        PUBLISH_1 : PUBLISH_1(ID := opc_ua[WRITE;%opcuaFolderTestWithNodeIdString1%]);
        E_CTU : E_CTU(PV := UINT#3);
        folderTest2SameFolder1String : TEST_CONDITION;
        SUBSCRIBE_1_1 : SUBSCRIBE_1(ID := opc_ua[READ;%opcuaFolderTestWithNodeIdString1%]);
        BOOL2BOOL_1_1_1_1_2 : DINT2DINT;
        folderTest2DifferentFolder1String : TEST_CONDITION;
        SUBSCRIBE_2_2 : SUBSCRIBE_2(ID := opc_ua[READ;%opcuaFolderTestWithNodeIdString2%]);
        SUBSCRIBE_2_1_1 : SUBSCRIBE_2(ID := opc_ua[READ;%opcuaFolderTestWithNodeIdString3%]);
        BOOL2BOOL_1_3 : DINT2DINT;
        BOOL2BOOL_3 : DINT2DINT;
        folderTestDirectUnderString : TEST_CONDITION;
      END_FBS
      EVENT_CONNECTIONS
        BOOL2BOOL_2.CNF TO BOOL2BOOL_1_2.REQ;
        BOOL2BOOL_1_2.CNF TO BOOL2BOOL_1_1_2.REQ;
        BOOL2BOOL_1_1_3.CNF TO F_EQ_1_2.REQ;
        F_EQ_1_2.CNF TO folderTest2SameFolder1String.REQ;
        BOOL2BOOL_3.CNF TO F_EQ_2.REQ;
        F_EQ_2.CNF TO folderTestDirectUnderString.REQ;
        PUBLISH_2_1.INITO TO PUBLISH_2.INIT;
        PUBLISH_2_1.CNF TO PUBLISH_2.REQ;
        PUBLISH_2.INITO TO PUBLISH_1.INIT;
        PUBLISH_2.CNF TO PUBLISH_1.REQ;
        F_EQ_1_1_2.CNF TO folderTest2SameFolder2String.REQ;
        F_EQ_1_1_1_1_1.CNF TO folderTest2DifferentFolder2String.REQ;
        E_CTU.CUO TO E_PERMIT.EI;
        BOOL2BOOL_1_1_1_1_2.CNF TO F_EQ_1_1_1_2.REQ;
        F_EQ_1_1_1_2.CNF TO folderTest2DifferentFolder1String.REQ;
        folderTest2DifferentFolder1String.CNF TO F_EQ_1_1_1_1_1.REQ;
        BOOL2BOOL_1_1_1_1_1.CNF TO PUBLISH_2_1.REQ;
        BOOL2BOOL_1_1_2.CNF TO BOOL2BOOL_1_1_1_2.REQ;
        BOOL2BOOL_1_1_1_2.CNF TO BOOL2BOOL_1_1_1_1_1.REQ;
        SUBSCRIBE_2_1_1.IND TO BOOL2BOOL_1_1_1_3.REQ;
        BOOL2BOOL_1_1_1_3.CNF TO BOOL2BOOL_1_1_1_1_2.REQ;
        BOOL2BOOL_1_3.CNF TO BOOL2BOOL_1_1_3.REQ;
        folderTest2SameFolder1String.CNF TO F_EQ_1_1_2.REQ;
        SUBSCRIBE_1_1.INITO TO SUBSCRIBE_2_2.INIT;
        SUBSCRIBE_1_1.IND TO BOOL2BOOL_3.REQ;
        SUBSCRIBE_2_2.INITO TO SUBSCRIBE_2_1_1.INIT;
        SUBSCRIBE_2_2.IND TO BOOL2BOOL_1_3.REQ;
        PUBLISH_1.INITO TO INITO;
        INIT TO SUBSCRIBE_1_1.INIT;
        folderTestDirectUnderString.CNF TO E_CTU.CU;
        folderTest2SameFolder2String.CNF TO E_CTU.CU;
        folderTest2DifferentFolder2String.CNF TO E_CTU.CU;
        E_PERMIT.EO TO CNF;
        REQ TO BOOL2BOOL_2.REQ;
        SUBSCRIBE_2_1_1.INITO TO PUBLISH_2_1.INIT;
      END_CONNECTIONS
      DATA_CONNECTIONS
        BOOL2BOOL_1_2.OUT TO PUBLISH_2.SD_1;
        BOOL2BOOL_1_3.OUT TO F_EQ_1_2.IN1;
        F_EQ_1_2.OUT TO folderTest2SameFolder1String.check;
        BOOL2BOOL_3.OUT TO F_EQ_2.IN1;
        F_EQ_2.OUT TO folderTestDirectUnderString.check;
        BOOL2BOOL_1_1_2.OUT TO PUBLISH_2.SD_2;
        F_EQ_1_1_2.OUT TO folderTest2SameFolder2String.check;
        F_EQ_1_1_1_1_1.OUT TO folderTest2DifferentFolder2String.check;
        E_CTU.Q TO E_PERMIT.PERMIT;
        BOOL2BOOL_1_1_1_3.OUT TO F_EQ_1_1_1_2.IN1;
        F_EQ_1_1_1_2.OUT TO folderTest2DifferentFolder1String.check;
        BOOL2BOOL_1_1_1_1_2.OUT TO F_EQ_1_1_1_1_1.IN1;
        BOOL2BOOL_1_1_1_2.OUT TO PUBLISH_2_1.SD_1;
        BOOL2BOOL_1_1_1_1_1.OUT TO PUBLISH_2_1.SD_2;
        BOOL2BOOL_2.OUT TO PUBLISH_1.SD_1;
        SUBSCRIBE_2_1_1.RD_1 TO BOOL2BOOL_1_1_1_3.IN;
        SUBSCRIBE_2_2.RD_2 TO BOOL2BOOL_1_1_3.IN;
        BOOL2BOOL_1_1_3.OUT TO F_EQ_1_1_2.IN1;
        SUBSCRIBE_1_1.RD_1 TO BOOL2BOOL_3.IN;
        SUBSCRIBE_2_1_1.RD_2 TO BOOL2BOOL_1_1_1_1_2.IN;
        SUBSCRIBE_2_2.RD_1 TO BOOL2BOOL_1_3.IN;
        QI TO SUBSCRIBE_1_1.QI;
        QI TO SUBSCRIBE_2_2.QI;
        QI TO SUBSCRIBE_2_1_1.QI;
        QI TO PUBLISH_1.QI;
        QI TO PUBLISH_2.QI;
        QI TO PUBLISH_2_1.QI;
      END_CONNECTIONS
    END_SUBAPPLICATION
    SUBAPPLICATION foldersWithNodeByteStringId_1
      EVENT_INPUT
        INIT;
        REQ;
      END_EVENT
      EVENT_OUTPUT
        INITO;
        CNF;
      END_EVENT
      VAR_INPUT
        QI : BOOL;
      END_VAR
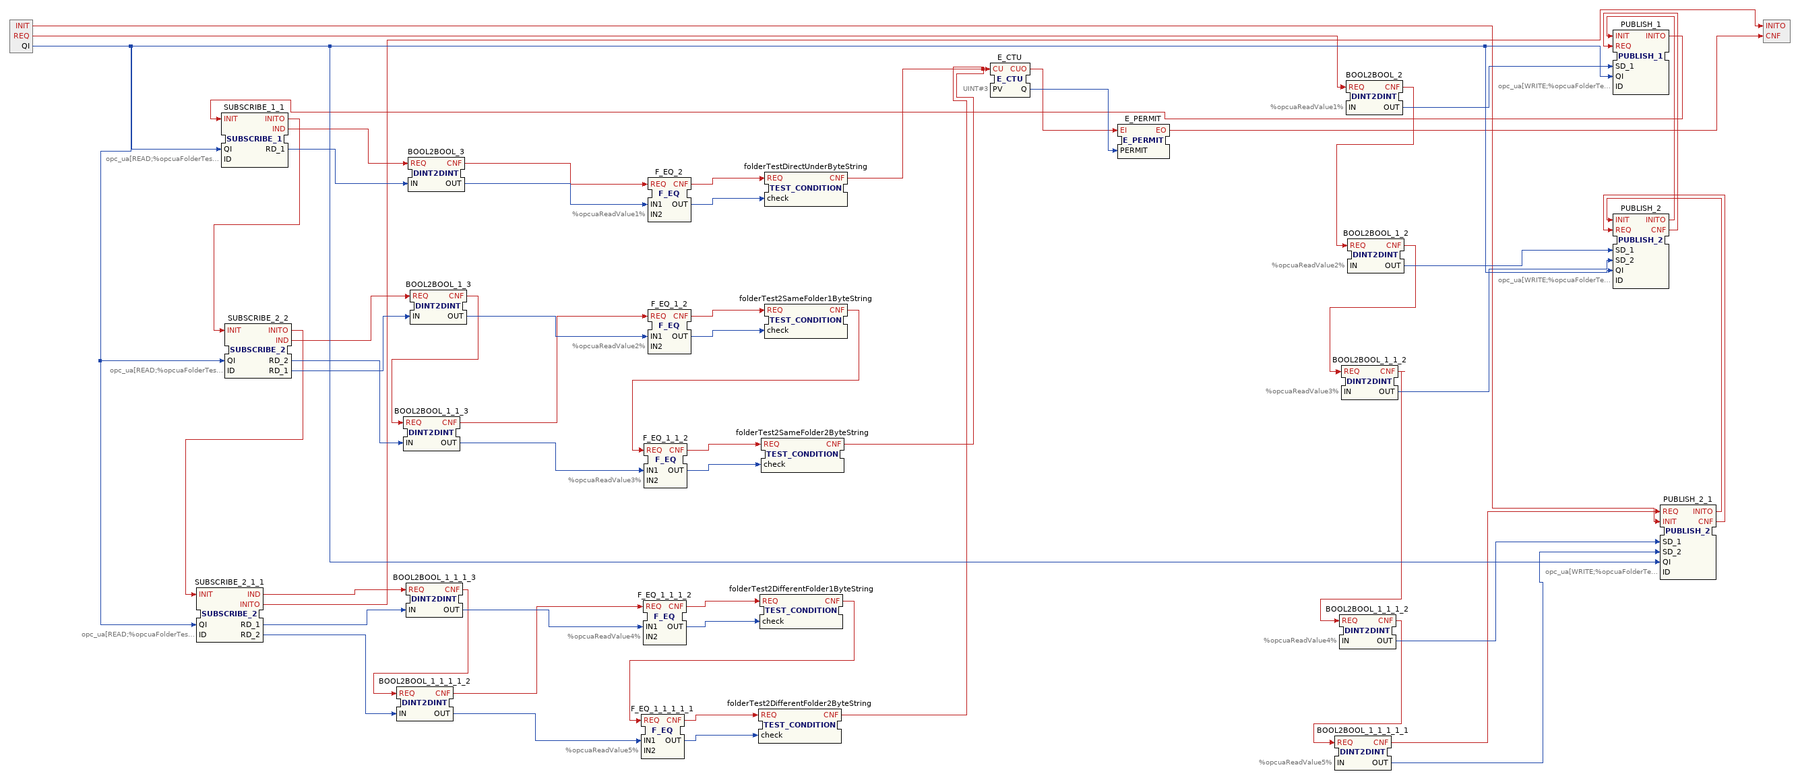
      [picture p23: application OpcUaLocalWorking.foldersWithNodeByteStringId_1]
      FBS
        BOOL2BOOL_1_2 : DINT2DINT(IN := %opcuaReadValue2%);
        F_EQ_1_2 : F_EQ(IN2 := %opcuaReadValue2%);
        F_EQ_2 : F_EQ(IN2 := %opcuaReadValue1%);
        PUBLISH_2 : PUBLISH_2(ID := opc_ua[WRITE;%opcuaFolderTestWithNodeIdByteString2%]);
        folderTest2SameFolder2ByteString : TEST_CONDITION;
        folderTest2DifferentFolder2ByteString : TEST_CONDITION;
        E_PERMIT : E_PERMIT;
        F_EQ_1_1_1_2 : F_EQ(IN2 := %opcuaReadValue4%);
        F_EQ_1_1_1_1_1 : F_EQ(IN2 := %opcuaReadValue5%);
        PUBLISH_2_1 : PUBLISH_2(ID := opc_ua[WRITE;%opcuaFolderTestWithNodeIdByteString3%]);
        BOOL2BOOL_1_1_2 : DINT2DINT(IN := %opcuaReadValue3%);
        BOOL2BOOL_1_1_1_1_1 : DINT2DINT(IN := %opcuaReadValue5%);
        BOOL2BOOL_2 : DINT2DINT(IN := %opcuaReadValue1%);
        BOOL2BOOL_1_1_1_3 : DINT2DINT;
        BOOL2BOOL_1_1_3 : DINT2DINT;
        BOOL2BOOL_1_1_1_2 : DINT2DINT(IN := %opcuaReadValue4%);
        F_EQ_1_1_2 : F_EQ(IN2 := %opcuaReadValue3%);
        PUBLISH_1 : PUBLISH_1(ID := opc_ua[WRITE;%opcuaFolderTestWithNodeIdByteString1%]);
        E_CTU : E_CTU(PV := UINT#3);
        folderTest2SameFolder1ByteString : TEST_CONDITION;
        SUBSCRIBE_1_1 : SUBSCRIBE_1(ID := opc_ua[READ;%opcuaFolderTestWithNodeIdByteString1%]);
        BOOL2BOOL_1_1_1_1_2 : DINT2DINT;
        folderTest2DifferentFolder1ByteString : TEST_CONDITION;
        SUBSCRIBE_2_2 : SUBSCRIBE_2(ID := opc_ua[READ;%opcuaFolderTestWithNodeIdByteString2%]);
        SUBSCRIBE_2_1_1 : SUBSCRIBE_2(ID := opc_ua[READ;%opcuaFolderTestWithNodeIdByteString3%]);
        BOOL2BOOL_1_3 : DINT2DINT;
        BOOL2BOOL_3 : DINT2DINT;
        folderTestDirectUnderByteString : TEST_CONDITION;
      END_FBS
      EVENT_CONNECTIONS
        BOOL2BOOL_2.CNF TO BOOL2BOOL_1_2.REQ;
        BOOL2BOOL_1_2.CNF TO BOOL2BOOL_1_1_2.REQ;
        BOOL2BOOL_1_1_3.CNF TO F_EQ_1_2.REQ;
        F_EQ_1_2.CNF TO folderTest2SameFolder1ByteString.REQ;
        BOOL2BOOL_3.CNF TO F_EQ_2.REQ;
        F_EQ_2.CNF TO folderTestDirectUnderByteString.REQ;
        PUBLISH_2_1.INITO TO PUBLISH_2.INIT;
        PUBLISH_2_1.CNF TO PUBLISH_2.REQ;
        PUBLISH_2.INITO TO PUBLISH_1.INIT;
        PUBLISH_2.CNF TO PUBLISH_1.REQ;
        F_EQ_1_1_2.CNF TO folderTest2SameFolder2ByteString.REQ;
        F_EQ_1_1_1_1_1.CNF TO folderTest2DifferentFolder2ByteString.REQ;
        E_CTU.CUO TO E_PERMIT.EI;
        BOOL2BOOL_1_1_1_1_2.CNF TO F_EQ_1_1_1_2.REQ;
        F_EQ_1_1_1_2.CNF TO folderTest2DifferentFolder1ByteString.REQ;
        folderTest2DifferentFolder1ByteString.CNF TO F_EQ_1_1_1_1_1.REQ;
        BOOL2BOOL_1_1_1_1_1.CNF TO PUBLISH_2_1.REQ;
        BOOL2BOOL_1_1_2.CNF TO BOOL2BOOL_1_1_1_2.REQ;
        BOOL2BOOL_1_1_1_2.CNF TO BOOL2BOOL_1_1_1_1_1.REQ;
        SUBSCRIBE_2_1_1.IND TO BOOL2BOOL_1_1_1_3.REQ;
        BOOL2BOOL_1_1_1_3.CNF TO BOOL2BOOL_1_1_1_1_2.REQ;
        BOOL2BOOL_1_3.CNF TO BOOL2BOOL_1_1_3.REQ;
        folderTest2SameFolder1ByteString.CNF TO F_EQ_1_1_2.REQ;
        SUBSCRIBE_1_1.INITO TO SUBSCRIBE_2_2.INIT;
        SUBSCRIBE_1_1.IND TO BOOL2BOOL_3.REQ;
        SUBSCRIBE_2_2.INITO TO SUBSCRIBE_2_1_1.INIT;
        SUBSCRIBE_2_2.IND TO BOOL2BOOL_1_3.REQ;
        folderTestDirectUnderByteString.CNF TO E_CTU.CU;
        folderTest2SameFolder2ByteString.CNF TO E_CTU.CU;
        folderTest2DifferentFolder2ByteString.CNF TO E_CTU.CU;
        E_PERMIT.EO TO CNF;
        REQ TO BOOL2BOOL_2.REQ;
        INIT TO PUBLISH_2_1.INIT;
        PUBLISH_1.INITO TO SUBSCRIBE_1_1.INIT;
        SUBSCRIBE_2_1_1.INITO TO INITO;
      END_CONNECTIONS
      DATA_CONNECTIONS
        BOOL2BOOL_1_2.OUT TO PUBLISH_2.SD_1;
        BOOL2BOOL_1_3.OUT TO F_EQ_1_2.IN1;
        F_EQ_1_2.OUT TO folderTest2SameFolder1ByteString.check;
        BOOL2BOOL_3.OUT TO F_EQ_2.IN1;
        F_EQ_2.OUT TO folderTestDirectUnderByteString.check;
        BOOL2BOOL_1_1_2.OUT TO PUBLISH_2.SD_2;
        F_EQ_1_1_2.OUT TO folderTest2SameFolder2ByteString.check;
        F_EQ_1_1_1_1_1.OUT TO folderTest2DifferentFolder2ByteString.check;
        E_CTU.Q TO E_PERMIT.PERMIT;
        BOOL2BOOL_1_1_1_3.OUT TO F_EQ_1_1_1_2.IN1;
        F_EQ_1_1_1_2.OUT TO folderTest2DifferentFolder1ByteString.check;
        BOOL2BOOL_1_1_1_1_2.OUT TO F_EQ_1_1_1_1_1.IN1;
        BOOL2BOOL_1_1_1_2.OUT TO PUBLISH_2_1.SD_1;
        BOOL2BOOL_1_1_1_1_1.OUT TO PUBLISH_2_1.SD_2;
        BOOL2BOOL_2.OUT TO PUBLISH_1.SD_1;
        SUBSCRIBE_2_1_1.RD_1 TO BOOL2BOOL_1_1_1_3.IN;
        SUBSCRIBE_2_2.RD_2 TO BOOL2BOOL_1_1_3.IN;
        BOOL2BOOL_1_1_3.OUT TO F_EQ_1_1_2.IN1;
        SUBSCRIBE_1_1.RD_1 TO BOOL2BOOL_3.IN;
        SUBSCRIBE_2_1_1.RD_2 TO BOOL2BOOL_1_1_1_1_2.IN;
        SUBSCRIBE_2_2.RD_1 TO BOOL2BOOL_1_3.IN;
        QI TO SUBSCRIBE_1_1.QI;
        QI TO SUBSCRIBE_2_2.QI;
        QI TO SUBSCRIBE_2_1_1.QI;
        QI TO PUBLISH_1.QI;
        QI TO PUBLISH_2.QI;
        QI TO PUBLISH_2_1.QI;
      END_CONNECTIONS
    END_SUBAPPLICATION
    SUBAPPLICATION foldersWithNodeNumericId_1
      EVENT_INPUT
        INIT;
        REQ;
      END_EVENT
      EVENT_OUTPUT
        INITO;
        CNF;
      END_EVENT
      VAR_INPUT
        QI : BOOL;
      END_VAR
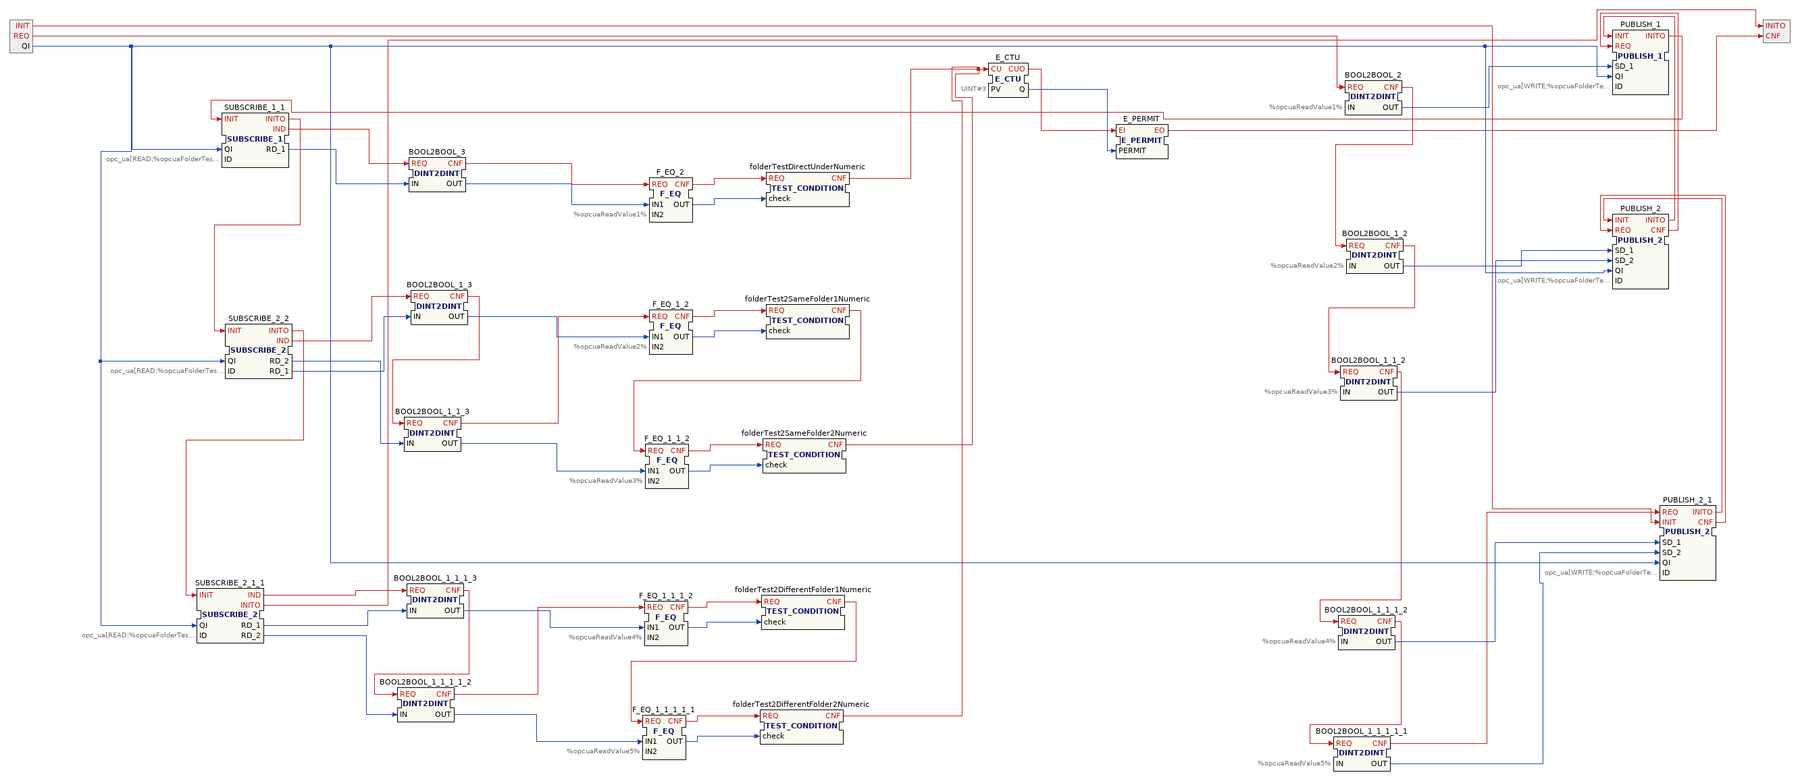
      FBS
        BOOL2BOOL_1_2 : DINT2DINT(IN := %opcuaReadValue2%);
        F_EQ_1_2 : F_EQ(IN2 := %opcuaReadValue2%);
        F_EQ_2 : F_EQ(IN2 := %opcuaReadValue1%);
        PUBLISH_2 : PUBLISH_2(ID := opc_ua[WRITE;%opcuaFolderTestWithNodeIdNumeric2%]);
        folderTest2SameFolder2Numeric : TEST_CONDITION;
        folderTest2DifferentFolder2Numeric : TEST_CONDITION;
        E_PERMIT : E_PERMIT;
        F_EQ_1_1_1_2 : F_EQ(IN2 := %opcuaReadValue4%);
        F_EQ_1_1_1_1_1 : F_EQ(IN2 := %opcuaReadValue5%);
        PUBLISH_2_1 : PUBLISH_2(ID := opc_ua[WRITE;%opcuaFolderTestWithNodeIdNumeric3%]);
        BOOL2BOOL_1_1_2 : DINT2DINT(IN := %opcuaReadValue3%);
        BOOL2BOOL_1_1_1_1_1 : DINT2DINT(IN := %opcuaReadValue5%);
        BOOL2BOOL_2 : DINT2DINT(IN := %opcuaReadValue1%);
        BOOL2BOOL_1_1_1_3 : DINT2DINT;
        BOOL2BOOL_1_1_3 : DINT2DINT;
        BOOL2BOOL_1_1_1_2 : DINT2DINT(IN := %opcuaReadValue4%);
        F_EQ_1_1_2 : F_EQ(IN2 := %opcuaReadValue3%);
        PUBLISH_1 : PUBLISH_1(ID := opc_ua[WRITE;%opcuaFolderTestWithNodeIdNumeric1%]);
        E_CTU : E_CTU(PV := UINT#3);
        folderTest2SameFolder1Numeric : TEST_CONDITION;
        SUBSCRIBE_1_1 : SUBSCRIBE_1(ID := opc_ua[READ;%opcuaFolderTestWithNodeIdNumeric1%]);
        BOOL2BOOL_1_1_1_1_2 : DINT2DINT;
        folderTest2DifferentFolder1Numeric : TEST_CONDITION;
        SUBSCRIBE_2_2 : SUBSCRIBE_2(ID := opc_ua[READ;%opcuaFolderTestWithNodeIdNumeric2%]);
        SUBSCRIBE_2_1_1 : SUBSCRIBE_2(ID := opc_ua[READ;%opcuaFolderTestWithNodeIdNumeric3%]);
        BOOL2BOOL_1_3 : DINT2DINT;
        BOOL2BOOL_3 : DINT2DINT;
        folderTestDirectUnderNumeric : TEST_CONDITION;
      END_FBS
      EVENT_CONNECTIONS
        BOOL2BOOL_2.CNF TO BOOL2BOOL_1_2.REQ;
        BOOL2BOOL_1_2.CNF TO BOOL2BOOL_1_1_2.REQ;
        BOOL2BOOL_1_1_3.CNF TO F_EQ_1_2.REQ;
        F_EQ_1_2.CNF TO folderTest2SameFolder1Numeric.REQ;
        BOOL2BOOL_3.CNF TO F_EQ_2.REQ;
        F_EQ_2.CNF TO folderTestDirectUnderNumeric.REQ;
        PUBLISH_2_1.INITO TO PUBLISH_2.INIT;
        PUBLISH_2_1.CNF TO PUBLISH_2.REQ;
        PUBLISH_2.INITO TO PUBLISH_1.INIT;
        PUBLISH_2.CNF TO PUBLISH_1.REQ;
        F_EQ_1_1_2.CNF TO folderTest2SameFolder2Numeric.REQ;
        F_EQ_1_1_1_1_1.CNF TO folderTest2DifferentFolder2Numeric.REQ;
        E_CTU.CUO TO E_PERMIT.EI;
        BOOL2BOOL_1_1_1_1_2.CNF TO F_EQ_1_1_1_2.REQ;
        F_EQ_1_1_1_2.CNF TO folderTest2DifferentFolder1Numeric.REQ;
        folderTest2DifferentFolder1Numeric.CNF TO F_EQ_1_1_1_1_1.REQ;
        BOOL2BOOL_1_1_1_1_1.CNF TO PUBLISH_2_1.REQ;
        BOOL2BOOL_1_1_2.CNF TO BOOL2BOOL_1_1_1_2.REQ;
        BOOL2BOOL_1_1_1_2.CNF TO BOOL2BOOL_1_1_1_1_1.REQ;
        SUBSCRIBE_2_1_1.IND TO BOOL2BOOL_1_1_1_3.REQ;
        BOOL2BOOL_1_1_1_3.CNF TO BOOL2BOOL_1_1_1_1_2.REQ;
        BOOL2BOOL_1_3.CNF TO BOOL2BOOL_1_1_3.REQ;
        folderTest2SameFolder1Numeric.CNF TO F_EQ_1_1_2.REQ;
        SUBSCRIBE_1_1.INITO TO SUBSCRIBE_2_2.INIT;
        SUBSCRIBE_1_1.IND TO BOOL2BOOL_3.REQ;
        SUBSCRIBE_2_2.INITO TO SUBSCRIBE_2_1_1.INIT;
        SUBSCRIBE_2_2.IND TO BOOL2BOOL_1_3.REQ;
        folderTestDirectUnderNumeric.CNF TO E_CTU.CU;
        folderTest2SameFolder2Numeric.CNF TO E_CTU.CU;
        folderTest2DifferentFolder2Numeric.CNF TO E_CTU.CU;
        E_PERMIT.EO TO CNF;
        REQ TO BOOL2BOOL_2.REQ;
        INIT TO PUBLISH_2_1.INIT;
        PUBLISH_1.INITO TO SUBSCRIBE_1_1.INIT;
        SUBSCRIBE_2_1_1.INITO TO INITO;
      END_CONNECTIONS
      DATA_CONNECTIONS
        BOOL2BOOL_1_2.OUT TO PUBLISH_2.SD_1;
        BOOL2BOOL_1_3.OUT TO F_EQ_1_2.IN1;
        F_EQ_1_2.OUT TO folderTest2SameFolder1Numeric.check;
        BOOL2BOOL_3.OUT TO F_EQ_2.IN1;
        F_EQ_2.OUT TO folderTestDirectUnderNumeric.check;
        BOOL2BOOL_1_1_2.OUT TO PUBLISH_2.SD_2;
        F_EQ_1_1_2.OUT TO folderTest2SameFolder2Numeric.check;
        F_EQ_1_1_1_1_1.OUT TO folderTest2DifferentFolder2Numeric.check;
        E_CTU.Q TO E_PERMIT.PERMIT;
        BOOL2BOOL_1_1_1_3.OUT TO F_EQ_1_1_1_2.IN1;
        F_EQ_1_1_1_2.OUT TO folderTest2DifferentFolder1Numeric.check;
        BOOL2BOOL_1_1_1_1_2.OUT TO F_EQ_1_1_1_1_1.IN1;
        BOOL2BOOL_1_1_1_2.OUT TO PUBLISH_2_1.SD_1;
        BOOL2BOOL_1_1_1_1_1.OUT TO PUBLISH_2_1.SD_2;
        BOOL2BOOL_2.OUT TO PUBLISH_1.SD_1;
        SUBSCRIBE_2_1_1.RD_1 TO BOOL2BOOL_1_1_1_3.IN;
        SUBSCRIBE_2_2.RD_2 TO BOOL2BOOL_1_1_3.IN;
        BOOL2BOOL_1_1_3.OUT TO F_EQ_1_1_2.IN1;
        SUBSCRIBE_1_1.RD_1 TO BOOL2BOOL_3.IN;
        SUBSCRIBE_2_1_1.RD_2 TO BOOL2BOOL_1_1_1_1_2.IN;
        SUBSCRIBE_2_2.RD_1 TO BOOL2BOOL_1_3.IN;
        QI TO SUBSCRIBE_1_1.QI;
        QI TO SUBSCRIBE_2_2.QI;
        QI TO SUBSCRIBE_2_1_1.QI;
        QI TO PUBLISH_1.QI;
        QI TO PUBLISH_2.QI;
        QI TO PUBLISH_2_1.QI;
      END_CONNECTIONS
    END_SUBAPPLICATION
    SUBAPPLICATION foldersWithNodeStringId_1
      EVENT_INPUT
        INIT;
        REQ;
      END_EVENT
      EVENT_OUTPUT
        INITO;
        CNF;
      END_EVENT
      VAR_INPUT
        QI : BOOL;
      END_VAR
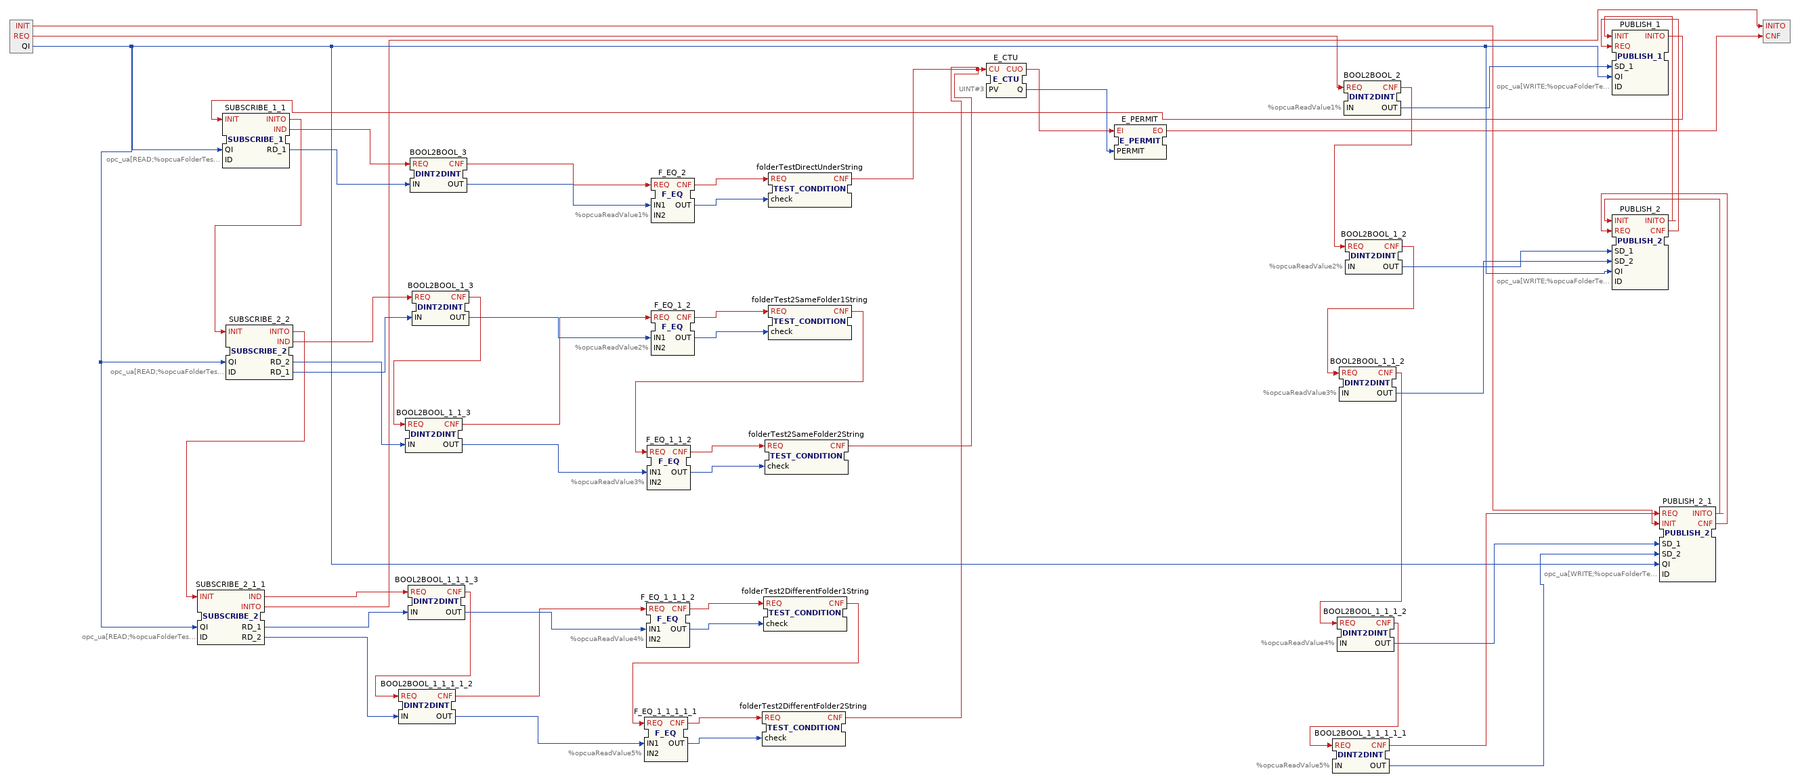
      FBS
        BOOL2BOOL_1_2 : DINT2DINT(IN := %opcuaReadValue2%);
        F_EQ_1_2 : F_EQ(IN2 := %opcuaReadValue2%);
        F_EQ_2 : F_EQ(IN2 := %opcuaReadValue1%);
        PUBLISH_2 : PUBLISH_2(ID := opc_ua[WRITE;%opcuaFolderTestWithNodeIdString2%]);
        folderTest2SameFolder2String : TEST_CONDITION;
        folderTest2DifferentFolder2String : TEST_CONDITION;
        E_PERMIT : E_PERMIT;
        F_EQ_1_1_1_2 : F_EQ(IN2 := %opcuaReadValue4%);
        F_EQ_1_1_1_1_1 : F_EQ(IN2 := %opcuaReadValue5%);
        PUBLISH_2_1 : PUBLISH_2(ID := opc_ua[WRITE;%opcuaFolderTestWithNodeIdString3%]);
        BOOL2BOOL_1_1_2 : DINT2DINT(IN := %opcuaReadValue3%);
        BOOL2BOOL_1_1_1_1_1 : DINT2DINT(IN := %opcuaReadValue5%);
        BOOL2BOOL_2 : DINT2DINT(IN := %opcuaReadValue1%);
        BOOL2BOOL_1_1_1_3 : DINT2DINT;
        BOOL2BOOL_1_1_3 : DINT2DINT;
        BOOL2BOOL_1_1_1_2 : DINT2DINT(IN := %opcuaReadValue4%);
        F_EQ_1_1_2 : F_EQ(IN2 := %opcuaReadValue3%);
        PUBLISH_1 : PUBLISH_1(ID := opc_ua[WRITE;%opcuaFolderTestWithNodeIdString1%]);
        E_CTU : E_CTU(PV := UINT#3);
        folderTest2SameFolder1String : TEST_CONDITION;
        SUBSCRIBE_1_1 : SUBSCRIBE_1(ID := opc_ua[READ;%opcuaFolderTestWithNodeIdString1%]);
        BOOL2BOOL_1_1_1_1_2 : DINT2DINT;
        folderTest2DifferentFolder1String : TEST_CONDITION;
        SUBSCRIBE_2_2 : SUBSCRIBE_2(ID := opc_ua[READ;%opcuaFolderTestWithNodeIdString2%]);
        SUBSCRIBE_2_1_1 : SUBSCRIBE_2(ID := opc_ua[READ;%opcuaFolderTestWithNodeIdString3%]);
        BOOL2BOOL_1_3 : DINT2DINT;
        BOOL2BOOL_3 : DINT2DINT;
        folderTestDirectUnderString : TEST_CONDITION;
      END_FBS
      EVENT_CONNECTIONS
        BOOL2BOOL_2.CNF TO BOOL2BOOL_1_2.REQ;
        BOOL2BOOL_1_2.CNF TO BOOL2BOOL_1_1_2.REQ;
        BOOL2BOOL_1_1_3.CNF TO F_EQ_1_2.REQ;
        F_EQ_1_2.CNF TO folderTest2SameFolder1String.REQ;
        BOOL2BOOL_3.CNF TO F_EQ_2.REQ;
        F_EQ_2.CNF TO folderTestDirectUnderString.REQ;
        PUBLISH_2_1.INITO TO PUBLISH_2.INIT;
        PUBLISH_2_1.CNF TO PUBLISH_2.REQ;
        PUBLISH_2.INITO TO PUBLISH_1.INIT;
        PUBLISH_2.CNF TO PUBLISH_1.REQ;
        F_EQ_1_1_2.CNF TO folderTest2SameFolder2String.REQ;
        F_EQ_1_1_1_1_1.CNF TO folderTest2DifferentFolder2String.REQ;
        E_CTU.CUO TO E_PERMIT.EI;
        BOOL2BOOL_1_1_1_1_2.CNF TO F_EQ_1_1_1_2.REQ;
        F_EQ_1_1_1_2.CNF TO folderTest2DifferentFolder1String.REQ;
        folderTest2DifferentFolder1String.CNF TO F_EQ_1_1_1_1_1.REQ;
        BOOL2BOOL_1_1_1_1_1.CNF TO PUBLISH_2_1.REQ;
        BOOL2BOOL_1_1_2.CNF TO BOOL2BOOL_1_1_1_2.REQ;
        BOOL2BOOL_1_1_1_2.CNF TO BOOL2BOOL_1_1_1_1_1.REQ;
        SUBSCRIBE_2_1_1.IND TO BOOL2BOOL_1_1_1_3.REQ;
        BOOL2BOOL_1_1_1_3.CNF TO BOOL2BOOL_1_1_1_1_2.REQ;
        BOOL2BOOL_1_3.CNF TO BOOL2BOOL_1_1_3.REQ;
        folderTest2SameFolder1String.CNF TO F_EQ_1_1_2.REQ;
        SUBSCRIBE_1_1.INITO TO SUBSCRIBE_2_2.INIT;
        SUBSCRIBE_1_1.IND TO BOOL2BOOL_3.REQ;
        SUBSCRIBE_2_2.INITO TO SUBSCRIBE_2_1_1.INIT;
        SUBSCRIBE_2_2.IND TO BOOL2BOOL_1_3.REQ;
        folderTestDirectUnderString.CNF TO E_CTU.CU;
        folderTest2SameFolder2String.CNF TO E_CTU.CU;
        folderTest2DifferentFolder2String.CNF TO E_CTU.CU;
        E_PERMIT.EO TO CNF;
        REQ TO BOOL2BOOL_2.REQ;
        INIT TO PUBLISH_2_1.INIT;
        PUBLISH_1.INITO TO SUBSCRIBE_1_1.INIT;
        SUBSCRIBE_2_1_1.INITO TO INITO;
      END_CONNECTIONS
      DATA_CONNECTIONS
        BOOL2BOOL_1_2.OUT TO PUBLISH_2.SD_1;
        BOOL2BOOL_1_3.OUT TO F_EQ_1_2.IN1;
        F_EQ_1_2.OUT TO folderTest2SameFolder1String.check;
        BOOL2BOOL_3.OUT TO F_EQ_2.IN1;
        F_EQ_2.OUT TO folderTestDirectUnderString.check;
        BOOL2BOOL_1_1_2.OUT TO PUBLISH_2.SD_2;
        F_EQ_1_1_2.OUT TO folderTest2SameFolder2String.check;
        F_EQ_1_1_1_1_1.OUT TO folderTest2DifferentFolder2String.check;
        E_CTU.Q TO E_PERMIT.PERMIT;
        BOOL2BOOL_1_1_1_3.OUT TO F_EQ_1_1_1_2.IN1;
        F_EQ_1_1_1_2.OUT TO folderTest2DifferentFolder1String.check;
        BOOL2BOOL_1_1_1_1_2.OUT TO F_EQ_1_1_1_1_1.IN1;
        BOOL2BOOL_1_1_1_2.OUT TO PUBLISH_2_1.SD_1;
        BOOL2BOOL_1_1_1_1_1.OUT TO PUBLISH_2_1.SD_2;
        BOOL2BOOL_2.OUT TO PUBLISH_1.SD_1;
        SUBSCRIBE_2_1_1.RD_1 TO BOOL2BOOL_1_1_1_3.IN;
        SUBSCRIBE_2_2.RD_2 TO BOOL2BOOL_1_1_3.IN;
        BOOL2BOOL_1_1_3.OUT TO F_EQ_1_1_2.IN1;
        SUBSCRIBE_1_1.RD_1 TO BOOL2BOOL_3.IN;
        SUBSCRIBE_2_1_1.RD_2 TO BOOL2BOOL_1_1_1_1_2.IN;
        SUBSCRIBE_2_2.RD_1 TO BOOL2BOOL_1_3.IN;
        QI TO SUBSCRIBE_1_1.QI;
        QI TO SUBSCRIBE_2_2.QI;
        QI TO SUBSCRIBE_2_1_1.QI;
        QI TO PUBLISH_1.QI;
        QI TO PUBLISH_2.QI;
        QI TO PUBLISH_2_1.QI;
      END_CONNECTIONS
    END_SUBAPPLICATION
    SUBAPPLICATION FoldersNoBrowseName_1
      EVENT_INPUT
        INIT;
        REQ;
      END_EVENT
      EVENT_OUTPUT
        INITO;
        CNF;
      END_EVENT
      VAR_INPUT
        QI : BOOL;
      END_VAR
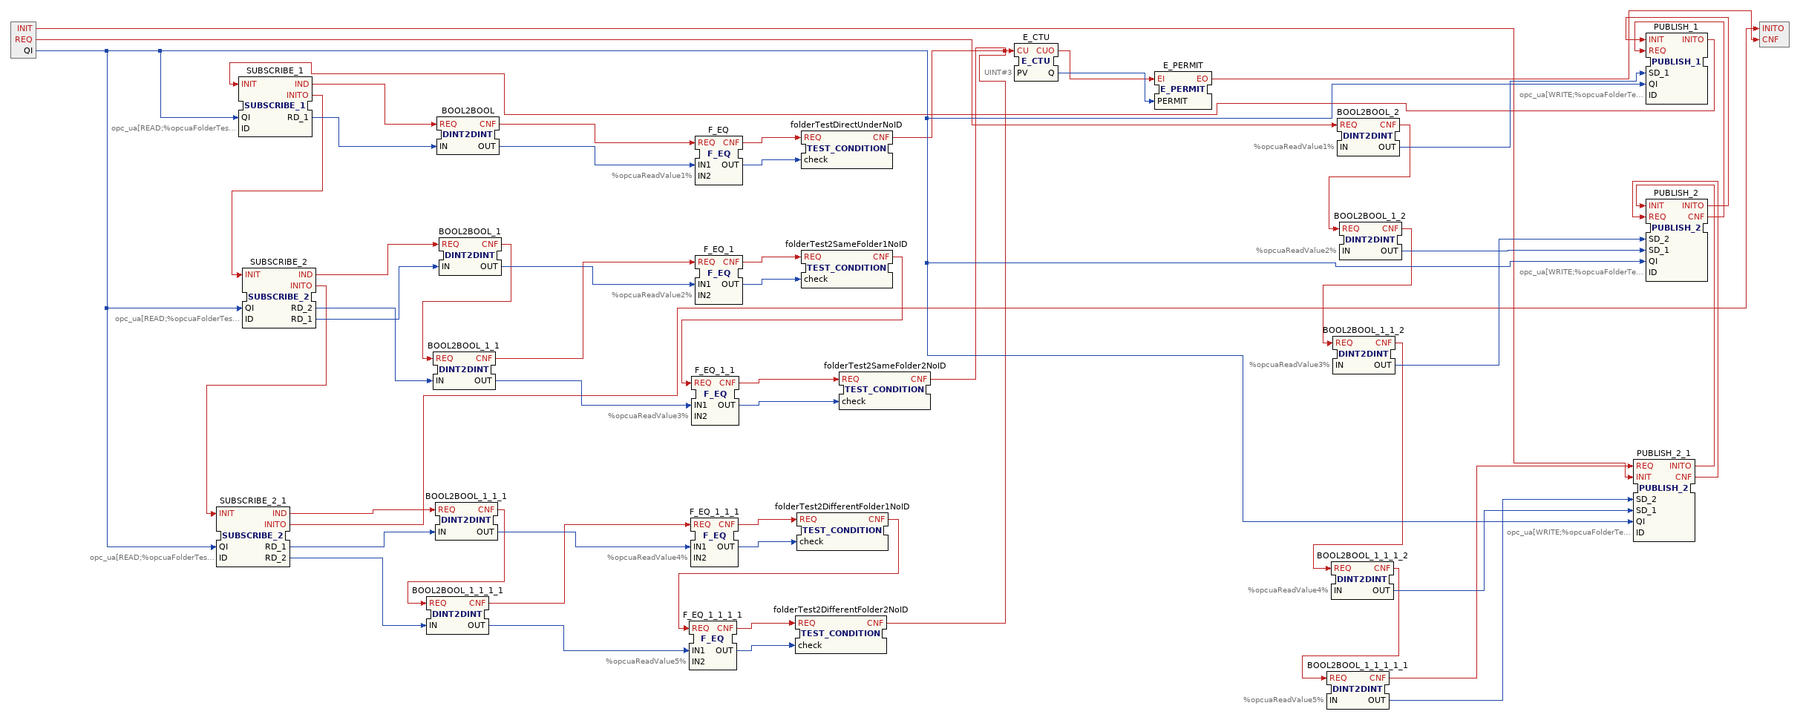
      FBS
        F_EQ_1_1_1 : F_EQ(IN2 := %opcuaReadValue4%);
        BOOL2BOOL_1_1 : DINT2DINT;
        SUBSCRIBE_2 : SUBSCRIBE_2(ID := opc_ua[READ;%opcuaFolderTestOnlyBroseName2%]);
        folderTestDirectUnderNoID : TEST_CONDITION;
        BOOL2BOOL_1 : DINT2DINT;
        BOOL2BOOL_1_1_1 : DINT2DINT;
        BOOL2BOOL_1_1_1_1_1 : DINT2DINT(IN := %opcuaReadValue5%);
        SUBSCRIBE_2_1 : SUBSCRIBE_2(ID := opc_ua[READ;%opcuaFolderTestOnlyBroseName3%]);
        SUBSCRIBE_1 : SUBSCRIBE_1(ID := opc_ua[READ;%opcuaFolderTestOnlyBroseName1%]);
        BOOL2BOOL_1_1_1_2 : DINT2DINT(IN := %opcuaReadValue4%);
        PUBLISH_2_1 : PUBLISH_2(ID := opc_ua[WRITE;%opcuaFolderTestOnlyBroseName3%]);
        BOOL2BOOL : DINT2DINT;
        F_EQ_1_1_1_1 : F_EQ(IN2 := %opcuaReadValue5%);
        BOOL2BOOL_1_1_2 : DINT2DINT(IN := %opcuaReadValue3%);
        E_PERMIT : E_PERMIT;
        folderTest2SameFolder1NoID : TEST_CONDITION;
        BOOL2BOOL_1_2 : DINT2DINT(IN := %opcuaReadValue2%);
        folderTest2DifferentFolder2NoID : TEST_CONDITION;
        BOOL2BOOL_1_1_1_1 : DINT2DINT;
        PUBLISH_1 : PUBLISH_1(ID := opc_ua[WRITE;%opcuaFolderTestOnlyBroseName1%]);
        BOOL2BOOL_2 : DINT2DINT(IN := %opcuaReadValue1%);
        F_EQ_1 : F_EQ(IN2 := %opcuaReadValue2%);
        E_CTU : E_CTU(PV := UINT#3);
        F_EQ : F_EQ(IN2 := %opcuaReadValue1%);
        PUBLISH_2 : PUBLISH_2(ID := opc_ua[WRITE;%opcuaFolderTestOnlyBroseName2%]);
        folderTest2SameFolder2NoID : TEST_CONDITION;
        folderTest2DifferentFolder1NoID : TEST_CONDITION;
        F_EQ_1_1 : F_EQ(IN2 := %opcuaReadValue3%);
      END_FBS
      EVENT_CONNECTIONS
        BOOL2BOOL_1_1_1_1.CNF TO F_EQ_1_1_1.REQ;
        F_EQ_1_1_1.CNF TO folderTest2DifferentFolder1NoID.REQ;
        BOOL2BOOL_1.CNF TO BOOL2BOOL_1_1.REQ;
        BOOL2BOOL_1_1.CNF TO F_EQ_1.REQ;
        SUBSCRIBE_2.IND TO BOOL2BOOL_1.REQ;
        F_EQ.CNF TO folderTestDirectUnderNoID.REQ;
        folderTestDirectUnderNoID.CNF TO E_CTU.CU;
        SUBSCRIBE_2_1.IND TO BOOL2BOOL_1_1_1.REQ;
        BOOL2BOOL_1_1_1.CNF TO BOOL2BOOL_1_1_1_1.REQ;
        BOOL2BOOL_1_1_1_2.CNF TO BOOL2BOOL_1_1_1_1_1.REQ;
        SUBSCRIBE_1.IND TO BOOL2BOOL.REQ;
        BOOL2BOOL_1_1_2.CNF TO BOOL2BOOL_1_1_1_2.REQ;
        PUBLISH_2_1.INITO TO PUBLISH_2.INIT;
        PUBLISH_2_1.CNF TO PUBLISH_2.REQ;
        BOOL2BOOL.CNF TO F_EQ.REQ;
        folderTest2DifferentFolder1NoID.CNF TO F_EQ_1_1_1_1.REQ;
        F_EQ_1_1_1_1.CNF TO folderTest2DifferentFolder2NoID.REQ;
        BOOL2BOOL_1_2.CNF TO BOOL2BOOL_1_1_2.REQ;
        E_CTU.CUO TO E_PERMIT.EI;
        F_EQ_1.CNF TO folderTest2SameFolder1NoID.REQ;
        folderTest2SameFolder1NoID.CNF TO F_EQ_1_1.REQ;
        BOOL2BOOL_2.CNF TO BOOL2BOOL_1_2.REQ;
        folderTest2DifferentFolder2NoID.CNF TO E_CTU.CU;
        PUBLISH_2.INITO TO PUBLISH_1.INIT;
        PUBLISH_2.CNF TO PUBLISH_1.REQ;
        folderTest2SameFolder2NoID.CNF TO E_CTU.CU;
        F_EQ_1_1.CNF TO folderTest2SameFolder2NoID.REQ;
        E_PERMIT.EO TO CNF;
        REQ TO BOOL2BOOL_2.REQ;
        BOOL2BOOL_1_1_1_1_1.CNF TO PUBLISH_2_1.REQ;
        SUBSCRIBE_1.INITO TO SUBSCRIBE_2.INIT;
        SUBSCRIBE_2.INITO TO SUBSCRIBE_2_1.INIT;
        INIT TO PUBLISH_2_1.INIT;
        PUBLISH_1.INITO TO SUBSCRIBE_1.INIT;
        SUBSCRIBE_2_1.INITO TO INITO;
      END_CONNECTIONS
      DATA_CONNECTIONS
        BOOL2BOOL_1_1_1.OUT TO F_EQ_1_1_1.IN1;
        F_EQ_1_1_1.OUT TO folderTest2DifferentFolder1NoID.check;
        SUBSCRIBE_2.RD_2 TO BOOL2BOOL_1_1.IN;
        BOOL2BOOL_1_1.OUT TO F_EQ_1_1.IN1;
        SUBSCRIBE_2.RD_1 TO BOOL2BOOL_1.IN;
        F_EQ.OUT TO folderTestDirectUnderNoID.check;
        BOOL2BOOL_1.OUT TO F_EQ_1.IN1;
        SUBSCRIBE_2_1.RD_1 TO BOOL2BOOL_1_1_1.IN;
        BOOL2BOOL_1_1_1_1_1.OUT TO PUBLISH_2_1.SD_2;
        SUBSCRIBE_2_1.RD_2 TO BOOL2BOOL_1_1_1_1.IN;
        SUBSCRIBE_1.RD_1 TO BOOL2BOOL.IN;
        BOOL2BOOL_1_1_1_2.OUT TO PUBLISH_2_1.SD_1;
        BOOL2BOOL.OUT TO F_EQ.IN1;
        BOOL2BOOL_1_1_1_1.OUT TO F_EQ_1_1_1_1.IN1;
        F_EQ_1_1_1_1.OUT TO folderTest2DifferentFolder2NoID.check;
        BOOL2BOOL_1_1_2.OUT TO PUBLISH_2.SD_2;
        E_CTU.Q TO E_PERMIT.PERMIT;
        F_EQ_1.OUT TO folderTest2SameFolder1NoID.check;
        BOOL2BOOL_1_2.OUT TO PUBLISH_2.SD_1;
        BOOL2BOOL_2.OUT TO PUBLISH_1.SD_1;
        F_EQ_1_1.OUT TO folderTest2SameFolder2NoID.check;
        QI TO SUBSCRIBE_2.QI;
        QI TO SUBSCRIBE_2_1.QI;
        QI TO SUBSCRIBE_1.QI;
        QI TO PUBLISH_2_1.QI;
        QI TO PUBLISH_1.QI;
        QI TO PUBLISH_2.QI;
      END_CONNECTIONS
    END_SUBAPPLICATION
    SUBAPPLICATION MethodOnlyBrowseName
      EVENT_INPUT
        INIT;
      END_EVENT
      EVENT_OUTPUT
        INITO;
      END_EVENT
      VAR_INPUT
        QI : BOOL;
      END_VAR
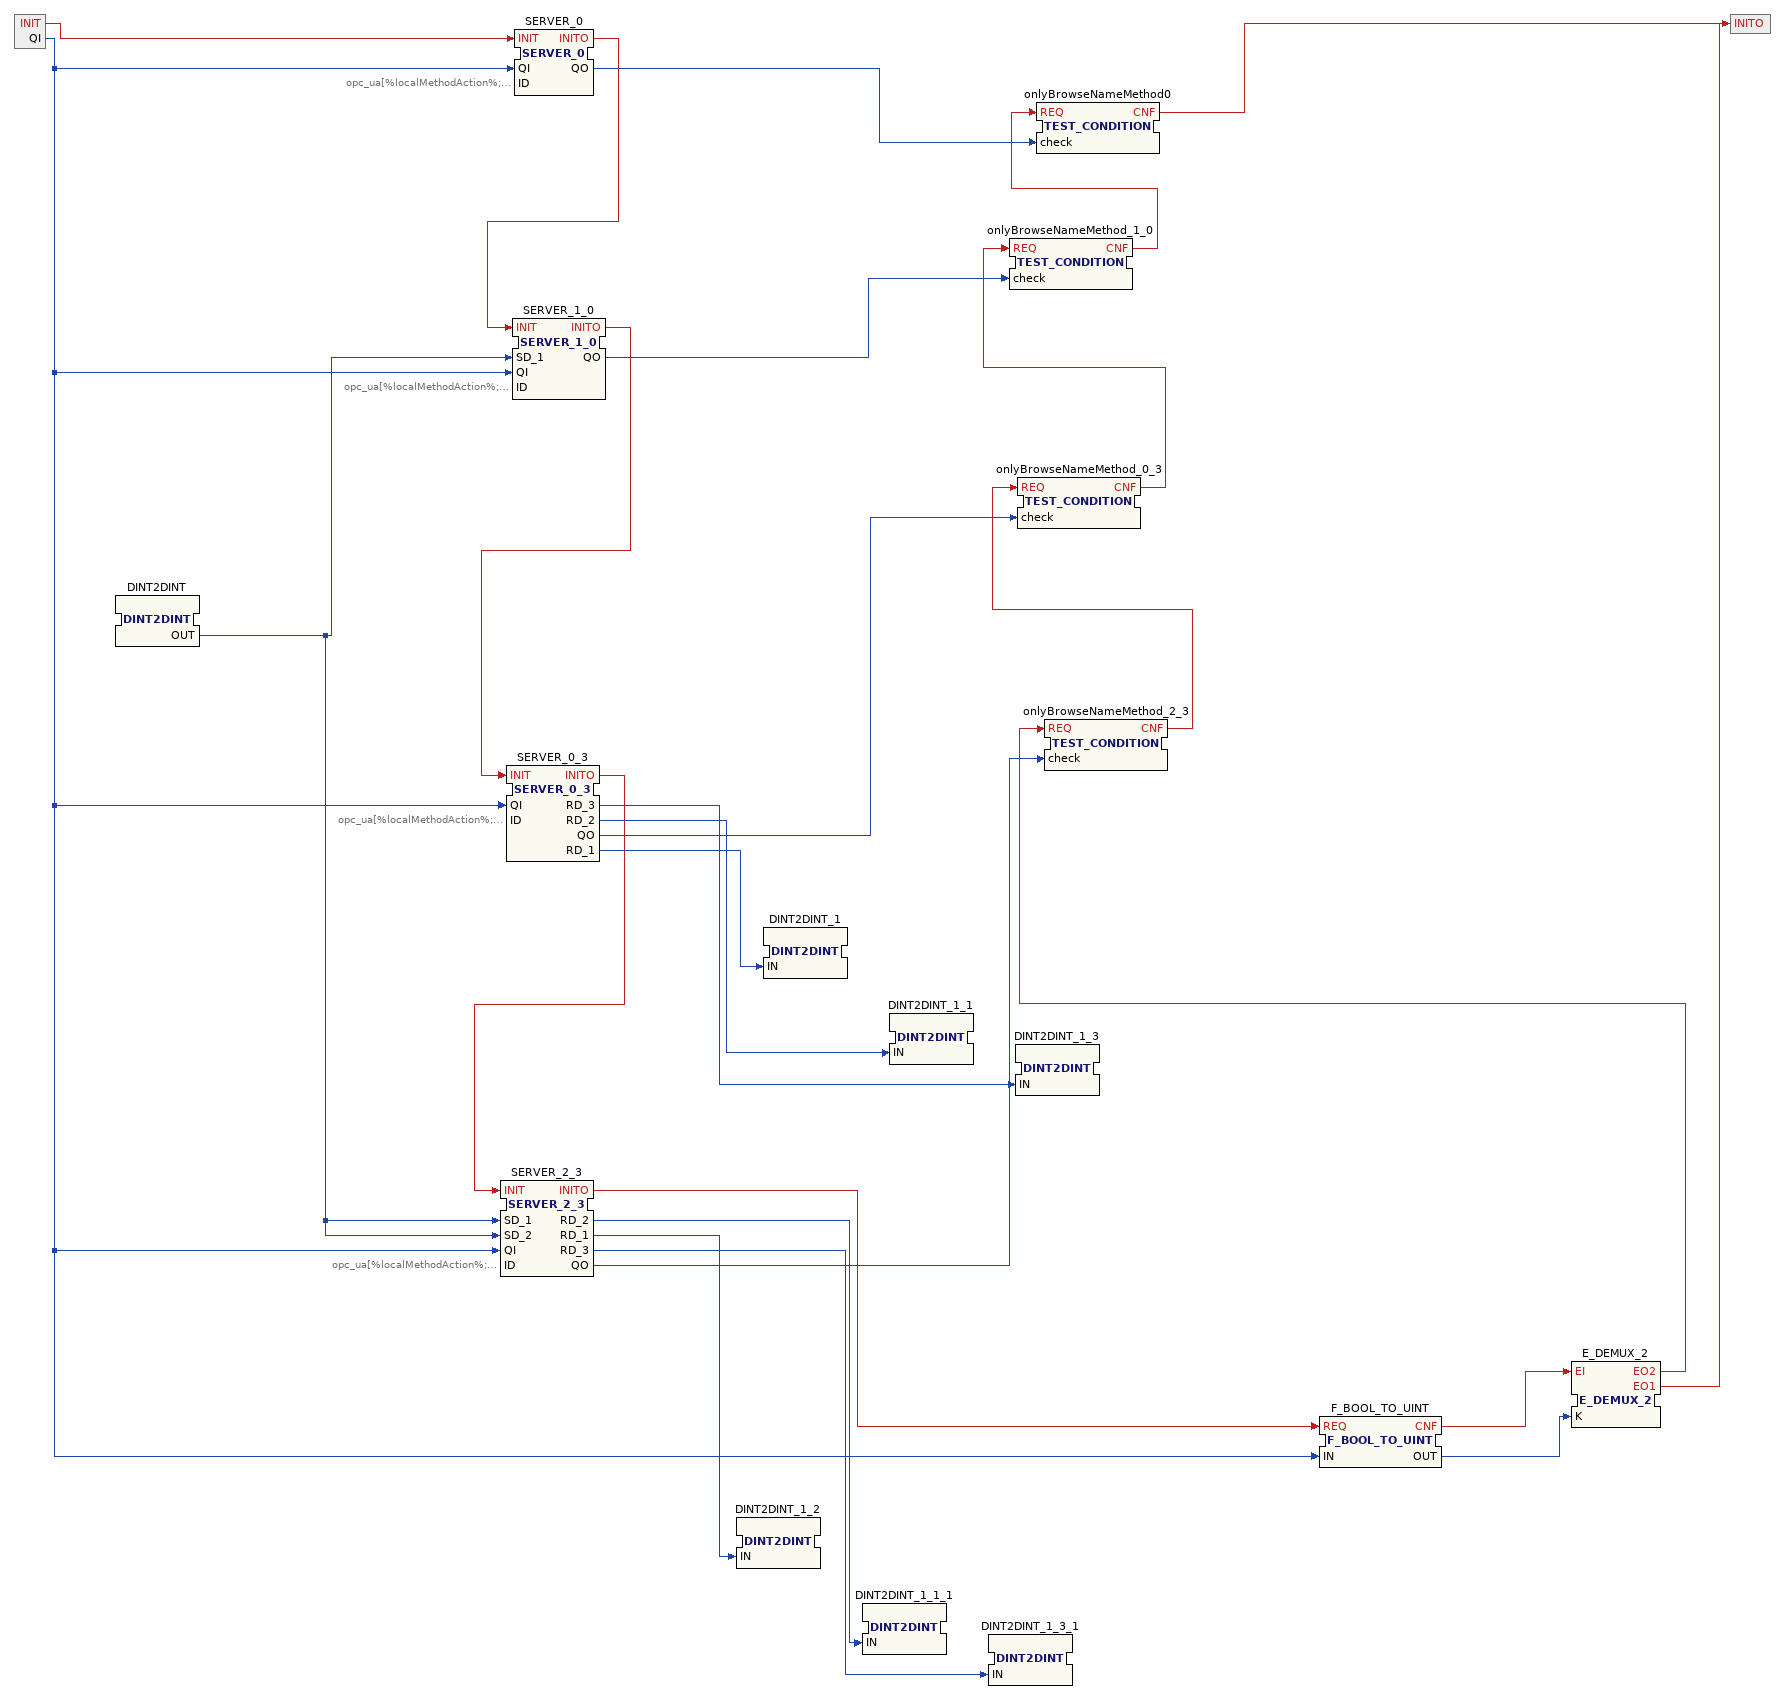
      FBS
        DINT2DINT_1_1_1 : DINT2DINT;
        DINT2DINT_1_2 : DINT2DINT;
        SERVER_0 : SERVER_0(ID := opc_ua[%localMethodAction%;%opcuaMethodCreation1%]);
        DINT2DINT_1_3 : DINT2DINT;
        DINT2DINT_1_1 : DINT2DINT;
        SERVER_0_3 : SERVER_0_3(ID := opc_ua[%localMethodAction%;%opcuaMethodCreation3%]);
        DINT2DINT_1_3_1 : DINT2DINT;
        SERVER_2_3 : SERVER_2_3(ID := opc_ua[%localMethodAction%;%opcuaMethodCreation4%]);
        onlyBrowseNameMethod_2_3 : TEST_CONDITION;
        onlyBrowseNameMethod_0_3 : TEST_CONDITION;
        SERVER_1_0 : SERVER_1_0(ID := opc_ua[%localMethodAction%;%opcuaMethodCreation2%]);
        onlyBrowseNameMethod0 : TEST_CONDITION;
        onlyBrowseNameMethod_1_0 : TEST_CONDITION;
        DINT2DINT : DINT2DINT;
        DINT2DINT_1 : DINT2DINT;
        E_DEMUX_2 : E_DEMUX_2;
        F_BOOL_TO_UINT : F_BOOL_TO_UINT;
      END_FBS
      EVENT_CONNECTIONS
        INIT TO SERVER_0.INIT;
        F_BOOL_TO_UINT.CNF TO E_DEMUX_2.EI;
        SERVER_2_3.INITO TO F_BOOL_TO_UINT.REQ;
        E_DEMUX_2.EO2 TO onlyBrowseNameMethod_2_3.REQ;
        SERVER_0.INITO TO SERVER_1_0.INIT;
        SERVER_1_0.INITO TO SERVER_0_3.INIT;
        SERVER_0_3.INITO TO SERVER_2_3.INIT;
        onlyBrowseNameMethod_2_3.CNF TO onlyBrowseNameMethod_0_3.REQ;
        onlyBrowseNameMethod_0_3.CNF TO onlyBrowseNameMethod_1_0.REQ;
        onlyBrowseNameMethod_1_0.CNF TO onlyBrowseNameMethod0.REQ;
        onlyBrowseNameMethod0.CNF TO INITO;
        E_DEMUX_2.EO1 TO INITO;
      END_CONNECTIONS
      DATA_CONNECTIONS
        SERVER_2_3.RD_2 TO DINT2DINT_1_1_1.IN;
        SERVER_2_3.RD_1 TO DINT2DINT_1_2.IN;
        SERVER_0.QO TO onlyBrowseNameMethod0.check;
        SERVER_0_3.RD_3 TO DINT2DINT_1_3.IN;
        SERVER_0_3.RD_2 TO DINT2DINT_1_1.IN;
        SERVER_0_3.QO TO onlyBrowseNameMethod_0_3.check;
        SERVER_0_3.RD_1 TO DINT2DINT_1.IN;
        SERVER_2_3.RD_3 TO DINT2DINT_1_3_1.IN;
        DINT2DINT.OUT TO SERVER_2_3.SD_1;
        DINT2DINT.OUT TO SERVER_2_3.SD_2;
        SERVER_2_3.QO TO onlyBrowseNameMethod_2_3.check;
        DINT2DINT.OUT TO SERVER_1_0.SD_1;
        SERVER_1_0.QO TO onlyBrowseNameMethod_1_0.check;
        QI TO SERVER_0.QI;
        QI TO SERVER_1_0.QI;
        QI TO SERVER_0_3.QI;
        QI TO SERVER_2_3.QI;
        F_BOOL_TO_UINT.OUT TO E_DEMUX_2.K;
        QI TO F_BOOL_TO_UINT.IN;
      END_CONNECTIONS
    END_SUBAPPLICATION
    SUBAPPLICATION MethodNumericNodeId
      EVENT_INPUT
        INIT;
      END_EVENT
      EVENT_OUTPUT
        INITO;
      END_EVENT
      VAR_INPUT
        QI : BOOL;
      END_VAR
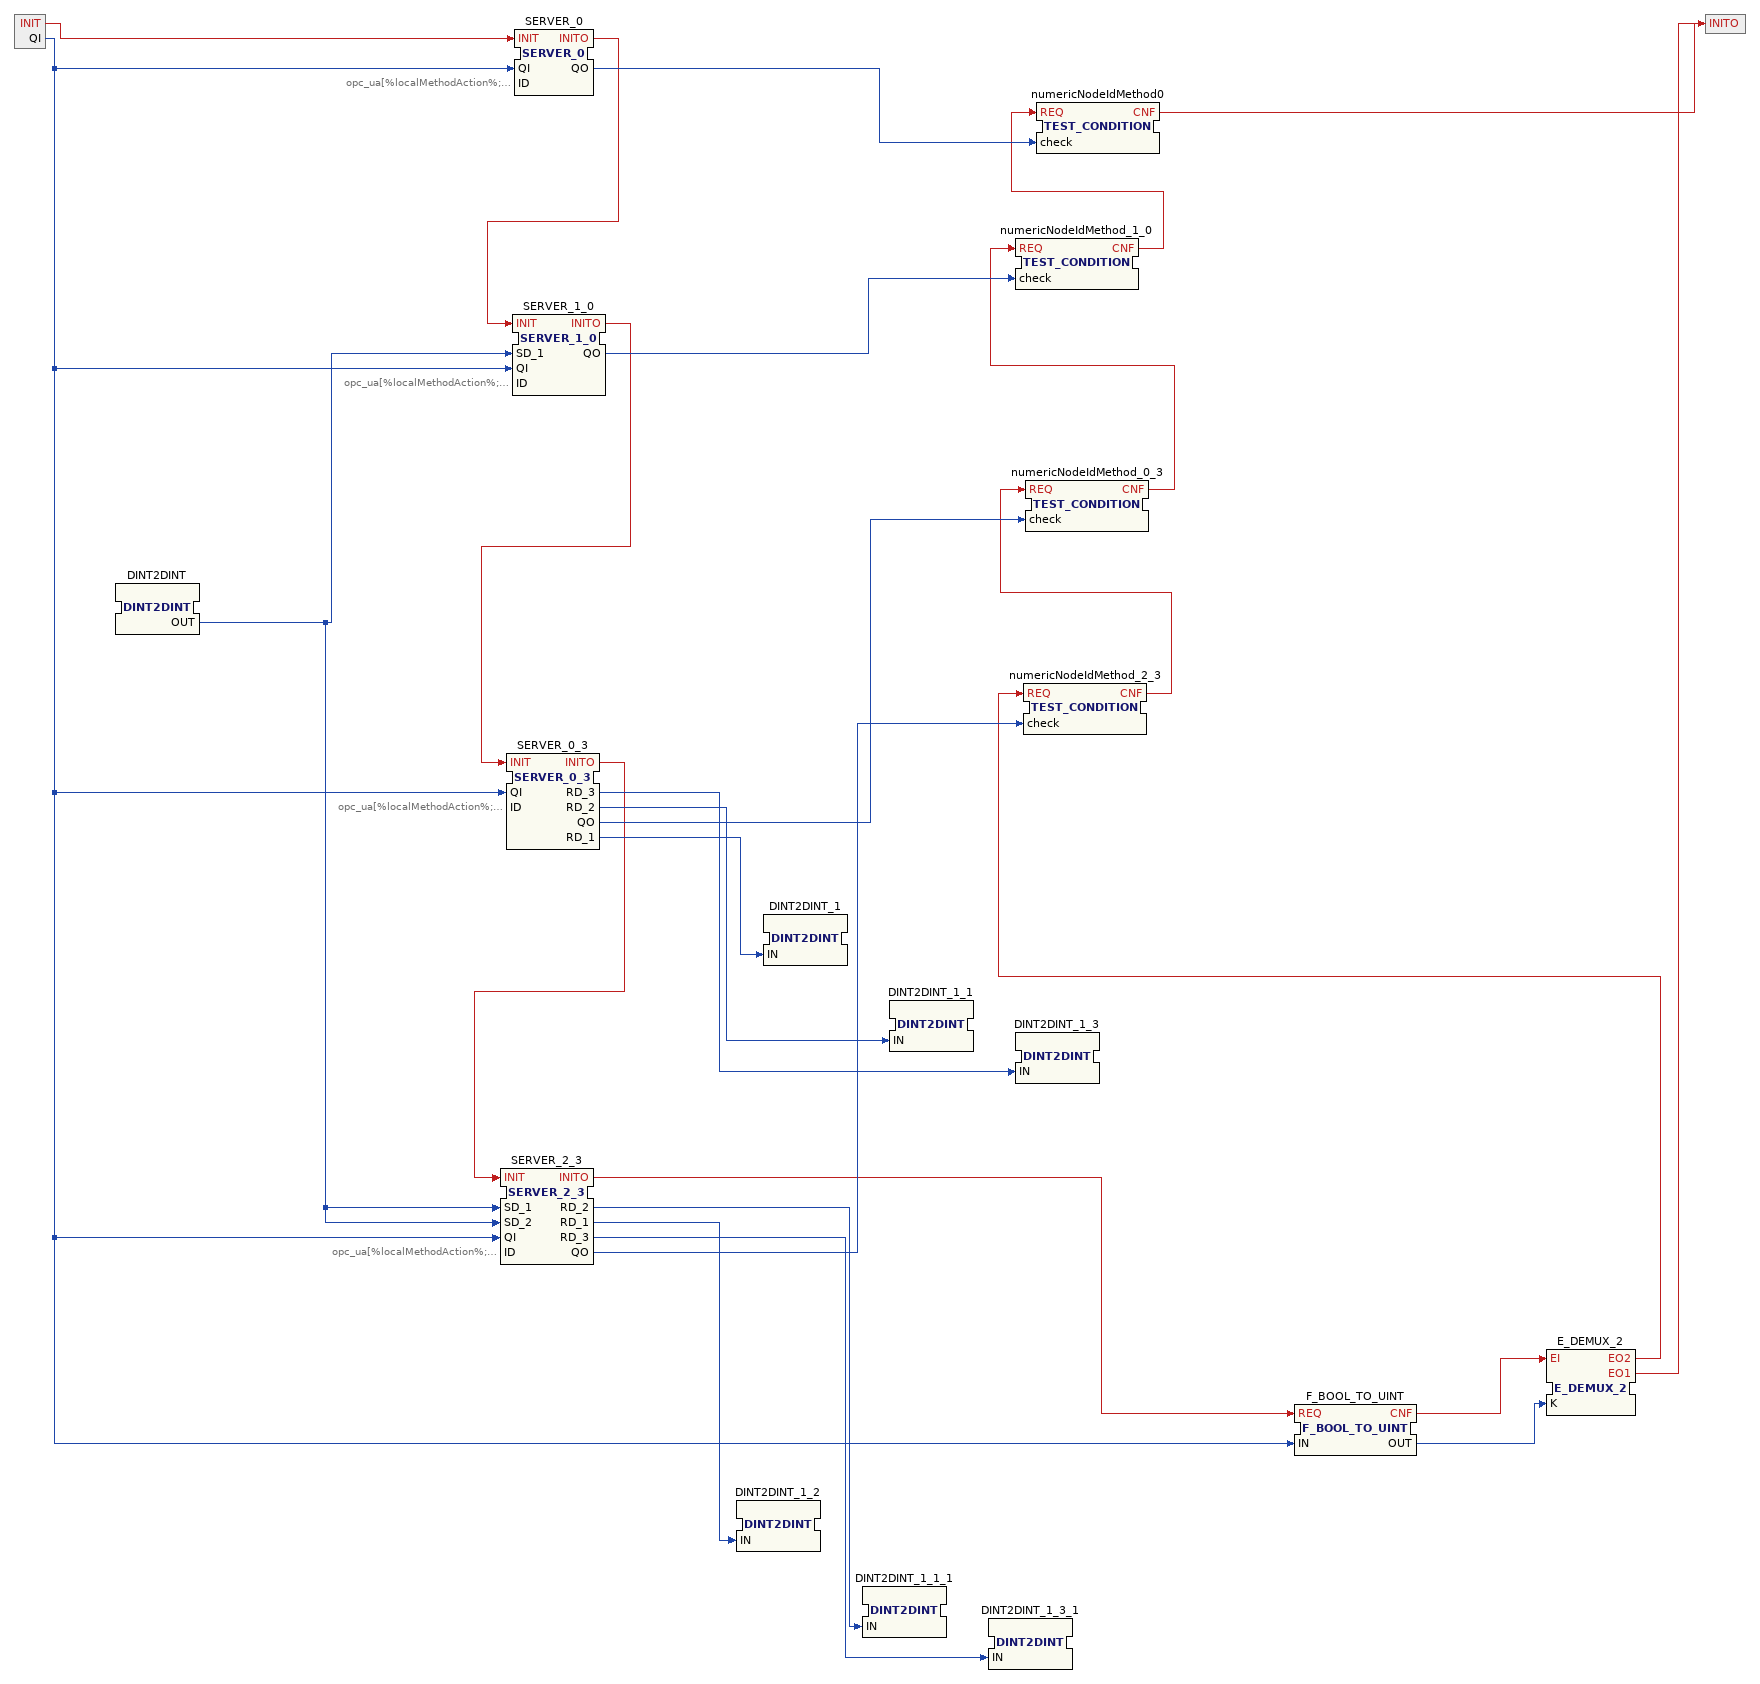
      FBS
        DINT2DINT_1_1_1 : DINT2DINT;
        DINT2DINT_1_2 : DINT2DINT;
        SERVER_0 : SERVER_0(ID := opc_ua[%localMethodAction%;%opcuaMethodCreation5%]);
        DINT2DINT_1_3 : DINT2DINT;
        DINT2DINT_1_1 : DINT2DINT;
        SERVER_0_3 : SERVER_0_3(ID := opc_ua[%localMethodAction%;%opcuaMethodCreation7%]);
        DINT2DINT_1_3_1 : DINT2DINT;
        SERVER_2_3 : SERVER_2_3(ID := opc_ua[%localMethodAction%;%opcuaMethodCreation8%]);
        numericNodeIdMethod_2_3 : TEST_CONDITION;
        numericNodeIdMethod_0_3 : TEST_CONDITION;
        SERVER_1_0 : SERVER_1_0(ID := opc_ua[%localMethodAction%;%opcuaMethodCreation6%]);
        numericNodeIdMethod0 : TEST_CONDITION;
        numericNodeIdMethod_1_0 : TEST_CONDITION;
        DINT2DINT : DINT2DINT;
        DINT2DINT_1 : DINT2DINT;
        E_DEMUX_2 : E_DEMUX_2;
        F_BOOL_TO_UINT : F_BOOL_TO_UINT;
      END_FBS
      EVENT_CONNECTIONS
        INIT TO SERVER_0.INIT;
        F_BOOL_TO_UINT.CNF TO E_DEMUX_2.EI;
        SERVER_2_3.INITO TO F_BOOL_TO_UINT.REQ;
        E_DEMUX_2.EO2 TO numericNodeIdMethod_2_3.REQ;
        E_DEMUX_2.EO1 TO INITO;
        SERVER_0_3.INITO TO SERVER_2_3.INIT;
        SERVER_0.INITO TO SERVER_1_0.INIT;
        SERVER_1_0.INITO TO SERVER_0_3.INIT;
        numericNodeIdMethod_0_3.CNF TO numericNodeIdMethod_1_0.REQ;
        numericNodeIdMethod0.CNF TO INITO;
        numericNodeIdMethod_1_0.CNF TO numericNodeIdMethod0.REQ;
        numericNodeIdMethod_2_3.CNF TO numericNodeIdMethod_0_3.REQ;
      END_CONNECTIONS
      DATA_CONNECTIONS
        SERVER_2_3.RD_2 TO DINT2DINT_1_1_1.IN;
        SERVER_2_3.RD_1 TO DINT2DINT_1_2.IN;
        SERVER_0.QO TO numericNodeIdMethod0.check;
        SERVER_0_3.RD_3 TO DINT2DINT_1_3.IN;
        SERVER_0_3.RD_2 TO DINT2DINT_1_1.IN;
        SERVER_0_3.QO TO numericNodeIdMethod_0_3.check;
        SERVER_0_3.RD_1 TO DINT2DINT_1.IN;
        SERVER_2_3.RD_3 TO DINT2DINT_1_3_1.IN;
        DINT2DINT.OUT TO SERVER_2_3.SD_1;
        DINT2DINT.OUT TO SERVER_2_3.SD_2;
        SERVER_2_3.QO TO numericNodeIdMethod_2_3.check;
        DINT2DINT.OUT TO SERVER_1_0.SD_1;
        SERVER_1_0.QO TO numericNodeIdMethod_1_0.check;
        QI TO SERVER_0.QI;
        QI TO SERVER_1_0.QI;
        QI TO SERVER_0_3.QI;
        QI TO SERVER_2_3.QI;
        F_BOOL_TO_UINT.OUT TO E_DEMUX_2.K;
        QI TO F_BOOL_TO_UINT.IN;
      END_CONNECTIONS
    END_SUBAPPLICATION
    SUBAPPLICATION MethodStringNodeId
      EVENT_INPUT
        INIT;
      END_EVENT
      EVENT_OUTPUT
        INITO;
      END_EVENT
      VAR_INPUT
        QI : BOOL;
      END_VAR
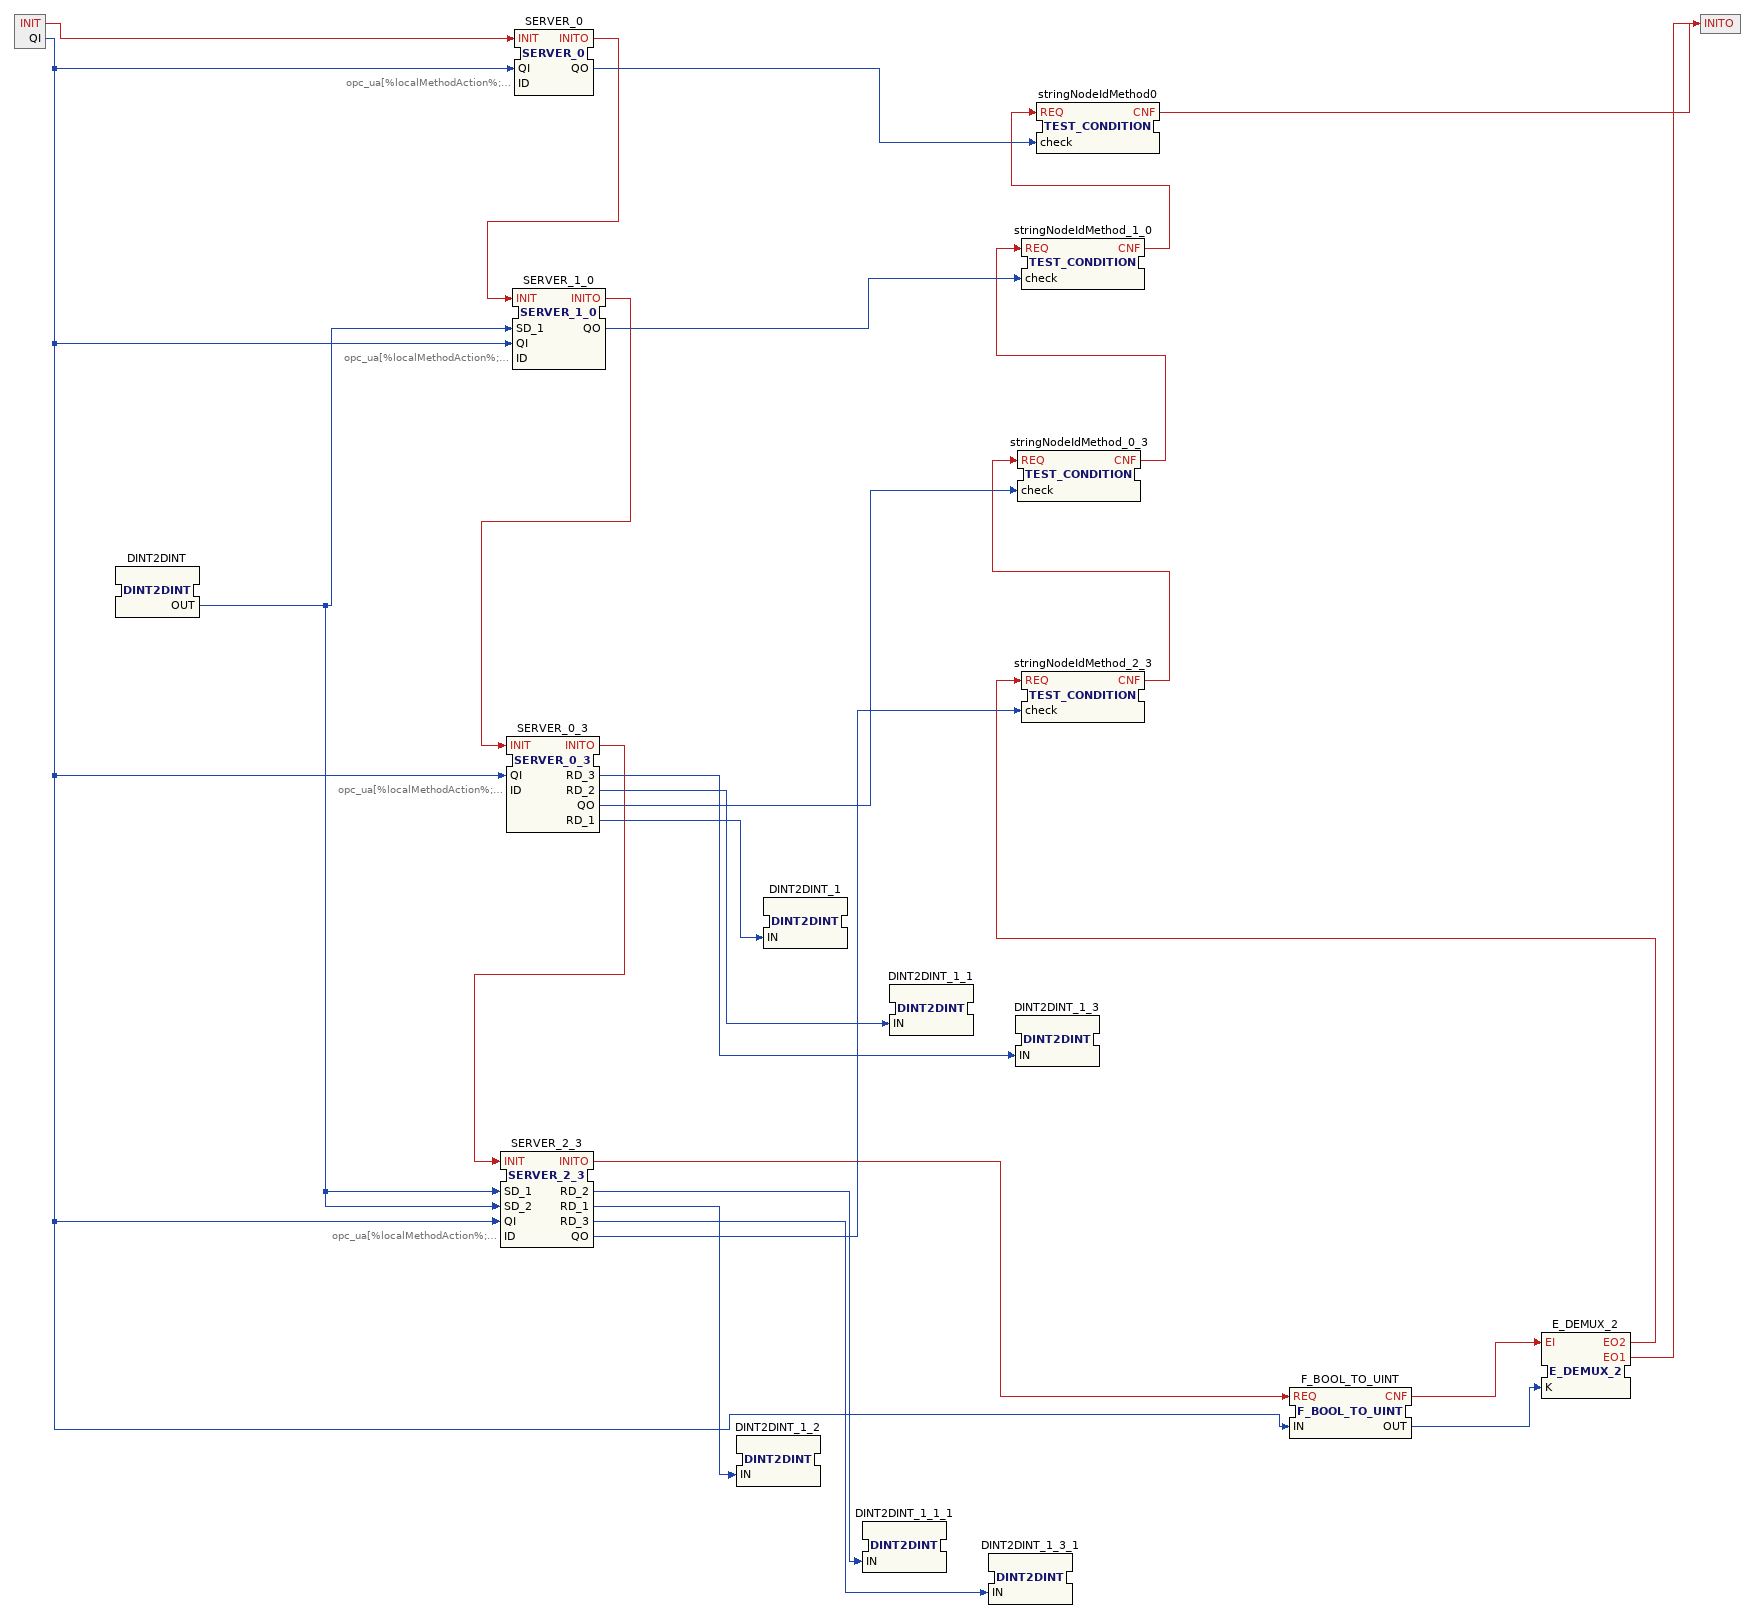
      FBS
        DINT2DINT_1_1_1 : DINT2DINT;
        DINT2DINT_1_2 : DINT2DINT;
        SERVER_0 : SERVER_0(ID := opc_ua[%localMethodAction%;%opcuaMethodCreation9%]);
        DINT2DINT_1_3 : DINT2DINT;
        DINT2DINT_1_1 : DINT2DINT;
        SERVER_0_3 : SERVER_0_3(ID := opc_ua[%localMethodAction%;%opcuaMethodCreation11%]);
        DINT2DINT_1_3_1 : DINT2DINT;
        SERVER_2_3 : SERVER_2_3(ID := opc_ua[%localMethodAction%;%opcuaMethodCreation12%]);
        stringNodeIdMethod_2_3 : TEST_CONDITION;
        stringNodeIdMethod_0_3 : TEST_CONDITION;
        SERVER_1_0 : SERVER_1_0(ID := opc_ua[%localMethodAction%;%opcuaMethodCreation10%]);
        stringNodeIdMethod0 : TEST_CONDITION;
        stringNodeIdMethod_1_0 : TEST_CONDITION;
        DINT2DINT : DINT2DINT;
        DINT2DINT_1 : DINT2DINT;
        E_DEMUX_2 : E_DEMUX_2;
        F_BOOL_TO_UINT : F_BOOL_TO_UINT;
      END_FBS
      EVENT_CONNECTIONS
        INIT TO SERVER_0.INIT;
        F_BOOL_TO_UINT.CNF TO E_DEMUX_2.EI;
        SERVER_2_3.INITO TO F_BOOL_TO_UINT.REQ;
        E_DEMUX_2.EO2 TO stringNodeIdMethod_2_3.REQ;
        E_DEMUX_2.EO1 TO INITO;
        stringNodeIdMethod_1_0.CNF TO stringNodeIdMethod0.REQ;
        stringNodeIdMethod0.CNF TO INITO;
        stringNodeIdMethod_2_3.CNF TO stringNodeIdMethod_0_3.REQ;
        stringNodeIdMethod_0_3.CNF TO stringNodeIdMethod_1_0.REQ;
        SERVER_0_3.INITO TO SERVER_2_3.INIT;
        SERVER_1_0.INITO TO SERVER_0_3.INIT;
        SERVER_0.INITO TO SERVER_1_0.INIT;
      END_CONNECTIONS
      DATA_CONNECTIONS
        SERVER_2_3.RD_2 TO DINT2DINT_1_1_1.IN;
        SERVER_2_3.RD_1 TO DINT2DINT_1_2.IN;
        SERVER_0.QO TO stringNodeIdMethod0.check;
        SERVER_0_3.RD_3 TO DINT2DINT_1_3.IN;
        SERVER_0_3.RD_2 TO DINT2DINT_1_1.IN;
        SERVER_0_3.QO TO stringNodeIdMethod_0_3.check;
        SERVER_0_3.RD_1 TO DINT2DINT_1.IN;
        SERVER_2_3.RD_3 TO DINT2DINT_1_3_1.IN;
        DINT2DINT.OUT TO SERVER_2_3.SD_1;
        DINT2DINT.OUT TO SERVER_2_3.SD_2;
        SERVER_2_3.QO TO stringNodeIdMethod_2_3.check;
        DINT2DINT.OUT TO SERVER_1_0.SD_1;
        SERVER_1_0.QO TO stringNodeIdMethod_1_0.check;
        QI TO SERVER_0.QI;
        QI TO SERVER_1_0.QI;
        QI TO SERVER_0_3.QI;
        QI TO SERVER_2_3.QI;
        F_BOOL_TO_UINT.OUT TO E_DEMUX_2.K;
        QI TO F_BOOL_TO_UINT.IN;
      END_CONNECTIONS
    END_SUBAPPLICATION
    SUBAPPLICATION MethodBytestringNodeId
      EVENT_INPUT
        INIT;
      END_EVENT
      EVENT_OUTPUT
        INITO;
      END_EVENT
      VAR_INPUT
        QI : BOOL;
      END_VAR
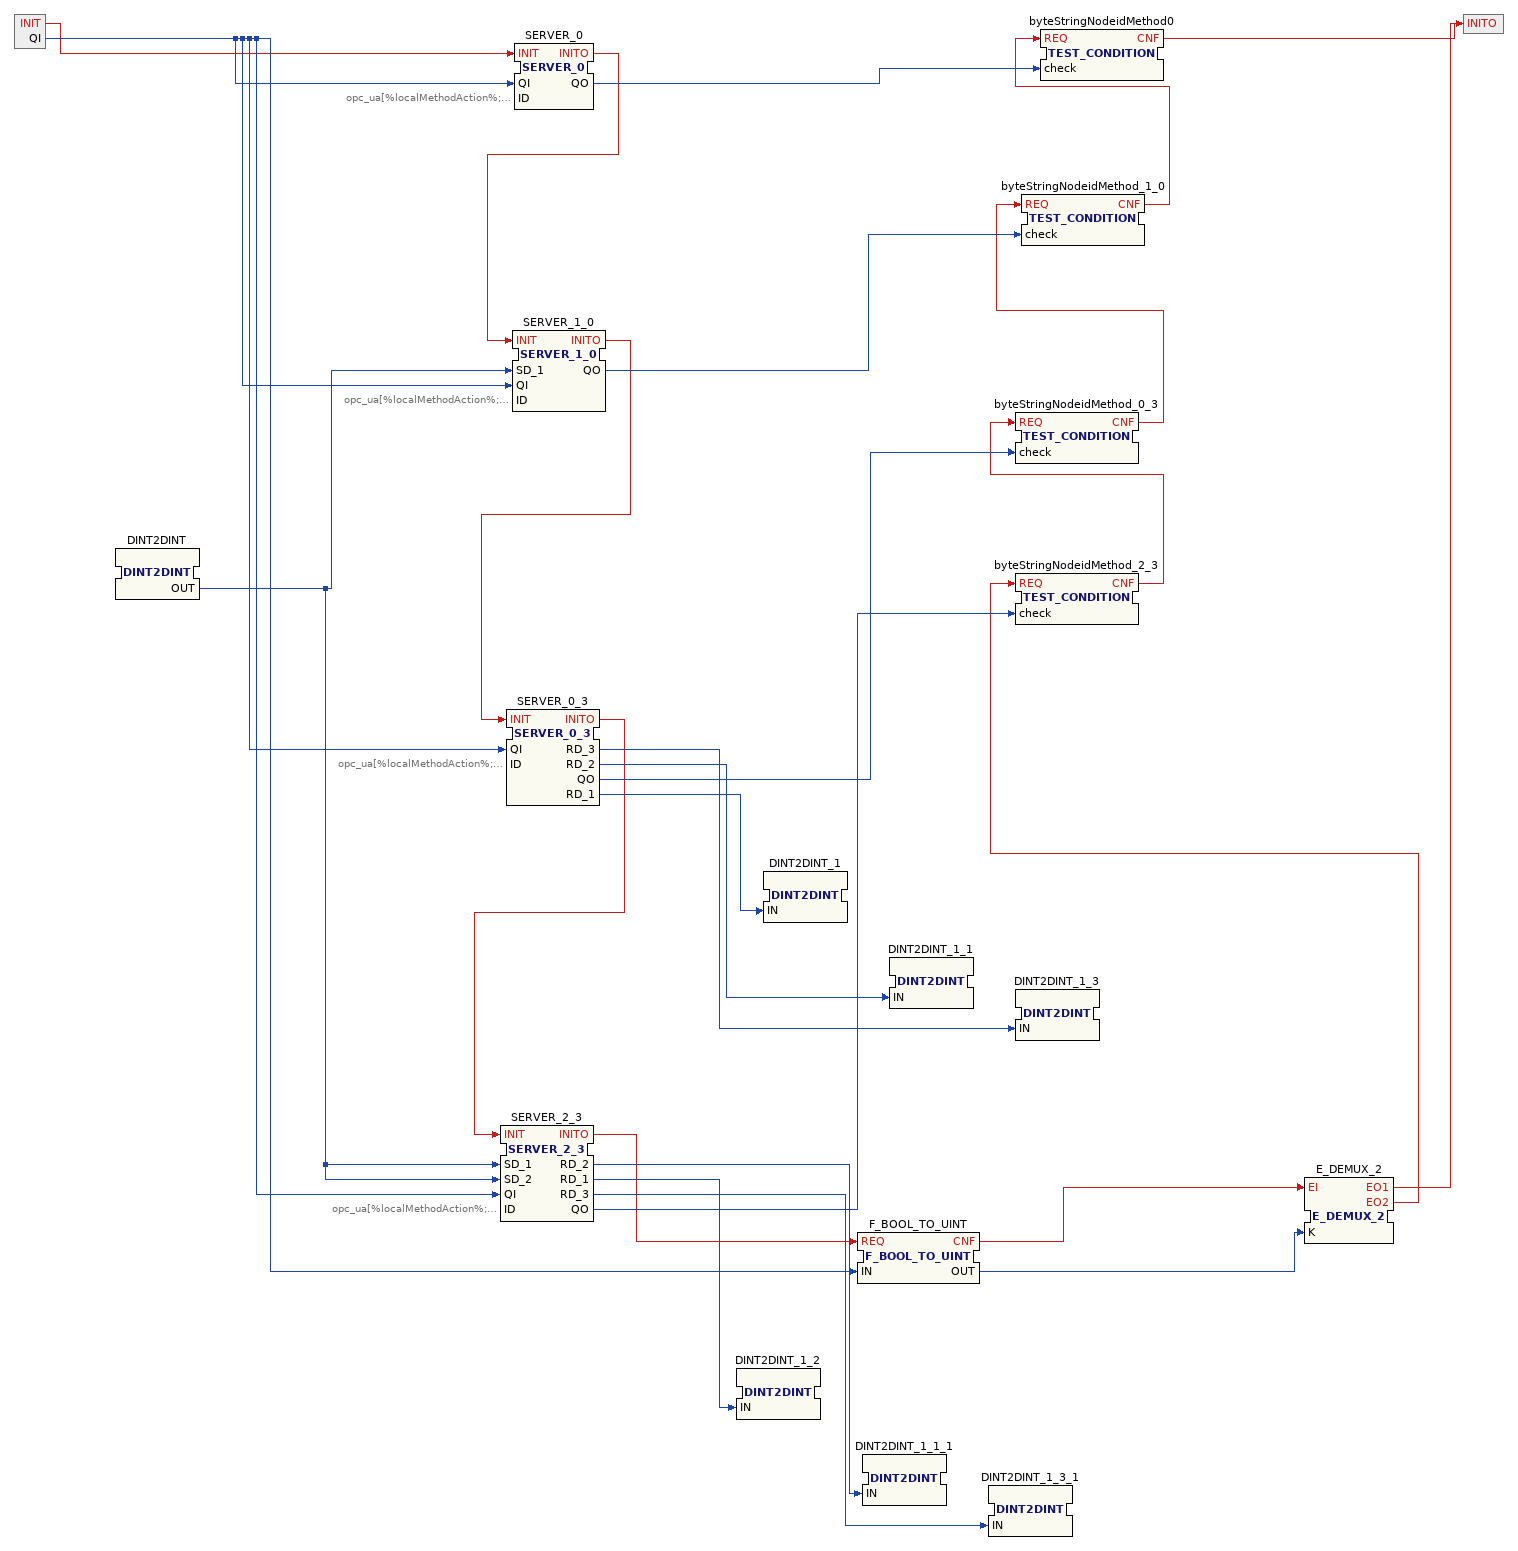
      FBS
        DINT2DINT_1_1_1 : DINT2DINT;
        DINT2DINT_1_2 : DINT2DINT;
        SERVER_0 : SERVER_0(ID := opc_ua[%localMethodAction%;%opcuaMethodCreation13%]);
        DINT2DINT_1_3 : DINT2DINT;
        DINT2DINT_1_1 : DINT2DINT;
        SERVER_0_3 : SERVER_0_3(ID := opc_ua[%localMethodAction%;%opcuaMethodCreation15%]);
        DINT2DINT_1_3_1 : DINT2DINT;
        SERVER_2_3 : SERVER_2_3(ID := opc_ua[%localMethodAction%;%opcuaMethodCreation16%]);
        byteStringNodeidMethod_2_3 : TEST_CONDITION;
        byteStringNodeidMethod_0_3 : TEST_CONDITION;
        SERVER_1_0 : SERVER_1_0(ID := opc_ua[%localMethodAction%;%opcuaMethodCreation14%]);
        byteStringNodeidMethod0 : TEST_CONDITION;
        byteStringNodeidMethod_1_0 : TEST_CONDITION;
        DINT2DINT : DINT2DINT;
        DINT2DINT_1 : DINT2DINT;
        E_DEMUX_2 : E_DEMUX_2;
        F_BOOL_TO_UINT : F_BOOL_TO_UINT;
      END_FBS
      EVENT_CONNECTIONS
        INIT TO SERVER_0.INIT;
        SERVER_0.INITO TO SERVER_1_0.INIT;
        SERVER_1_0.INITO TO SERVER_0_3.INIT;
        SERVER_0_3.INITO TO SERVER_2_3.INIT;
        SERVER_2_3.INITO TO F_BOOL_TO_UINT.REQ;
        F_BOOL_TO_UINT.CNF TO E_DEMUX_2.EI;
        E_DEMUX_2.EO1 TO INITO;
        E_DEMUX_2.EO2 TO byteStringNodeidMethod_2_3.REQ;
        byteStringNodeidMethod_2_3.CNF TO byteStringNodeidMethod_0_3.REQ;
        byteStringNodeidMethod_0_3.CNF TO byteStringNodeidMethod_1_0.REQ;
        byteStringNodeidMethod_1_0.CNF TO byteStringNodeidMethod0.REQ;
        byteStringNodeidMethod0.CNF TO INITO;
      END_CONNECTIONS
      DATA_CONNECTIONS
        SERVER_2_3.RD_2 TO DINT2DINT_1_1_1.IN;
        SERVER_2_3.RD_1 TO DINT2DINT_1_2.IN;
        SERVER_0.QO TO byteStringNodeidMethod0.check;
        SERVER_0_3.RD_3 TO DINT2DINT_1_3.IN;
        SERVER_0_3.RD_2 TO DINT2DINT_1_1.IN;
        SERVER_0_3.QO TO byteStringNodeidMethod_0_3.check;
        SERVER_0_3.RD_1 TO DINT2DINT_1.IN;
        SERVER_2_3.RD_3 TO DINT2DINT_1_3_1.IN;
        DINT2DINT.OUT TO SERVER_2_3.SD_1;
        DINT2DINT.OUT TO SERVER_2_3.SD_2;
        SERVER_2_3.QO TO byteStringNodeidMethod_2_3.check;
        DINT2DINT.OUT TO SERVER_1_0.SD_1;
        SERVER_1_0.QO TO byteStringNodeidMethod_1_0.check;
        QI TO SERVER_0.QI;
        QI TO SERVER_1_0.QI;
        QI TO SERVER_0_3.QI;
        QI TO SERVER_2_3.QI;
        F_BOOL_TO_UINT.OUT TO E_DEMUX_2.K;
        QI TO F_BOOL_TO_UINT.IN;
      END_CONNECTIONS
    END_SUBAPPLICATION
    EVENT_CONNECTIONS
      E_SR.EO TO FoldersNoBrowseName.INIT;
      foldersWithNodeStringId.INITO TO foldersWithNodeByteStringId.INIT;
      foldersWithNodeStringId.CNF TO foldersWithNodeByteStringId.REQ;
      F_BOOL_TO_UINT.CNF TO E_DEMUX_2.EI;
      E_DEMUX_2.EO2 TO FoldersNoBrowseName.REQ;
      foldersWithNodeByteStringId.INITO TO F_BOOL_TO_UINT.REQ;
      foldersWithNodeNumericId.CNF TO foldersWithNodeStringId.REQ;
      foldersWithNodeByteStringId.CNF TO E_SR.R;
      foldersWithNodeNumericId.INITO TO foldersWithNodeStringId.INIT;
      FoldersNoBrowseName.INITO TO foldersWithNodeNumericId.INIT;
      FoldersNoBrowseName.CNF TO foldersWithNodeNumericId.REQ;
      FoldersNoBrowseName_1.CNF TO foldersWithNodeNumericId_1.REQ;
      foldersWithNodeByteStringId_1.INITO TO F_BOOL_TO_UINT_1.REQ;
      E_DEMUX_2_1.EO1 TO STEST_END_1.REQ;
      F_BOOL_TO_UINT_1.CNF TO E_DEMUX_2_1.EI;
      foldersWithNodeStringId_1.INITO TO foldersWithNodeByteStringId_1.INIT;
      E_SR_1.EO TO FoldersNoBrowseName_1.INIT;
      E_DEMUX_2_1.EO2 TO FoldersNoBrowseName_1.REQ;
      FoldersNoBrowseName_1.INITO TO foldersWithNodeNumericId_1.INIT;
      foldersWithNodeStringId_1.CNF TO foldersWithNodeByteStringId_1.REQ;
      foldersWithNodeByteStringId_1.CNF TO E_SR_1.R;
      foldersWithNodeNumericId_1.INITO TO foldersWithNodeStringId_1.INIT;
      foldersWithNodeNumericId_1.CNF TO foldersWithNodeStringId_1.REQ;
      MethodOnlyBrowseName.INITO TO MethodNumericNodeId.INIT;
      MethodNumericNodeId.INITO TO MethodStringNodeId.INIT;
      MethodStringNodeId.INITO TO MethodBytestringNodeId.INIT;
      E_SR_2.EO TO MethodOnlyBrowseName.INIT;
      F_BOOL_TO_UINT_2.CNF TO E_DEMUX_2_2.EI;
      E_DEMUX_2_2.EO2 TO E_SR_2.R;
      E_DEMUX_2.EO1 TO STEST_END.REQ;
      E_DEMUX_2_2.EO1 TO STEST_END_2.REQ;
      MethodBytestringNodeId.INITO TO F_BOOL_TO_UINT_2.REQ;
    END_CONNECTIONS
    DATA_CONNECTIONS
      E_SR.Q TO FoldersNoBrowseName.QI;
      E_SR.Q TO FoldersNoBrowseName.QI;
      E_SR.Q TO foldersWithNodeNumericId.QI;
      E_SR.Q TO foldersWithNodeStringId.QI;
      E_SR.Q TO foldersWithNodeByteStringId.QI;
      E_SR.Q TO foldersWithNodeStringId.QI;
      E_SR.Q TO foldersWithNodeNumericId.QI;
      E_SR.Q TO foldersWithNodeByteStringId.QI;
      F_BOOL_TO_UINT.OUT TO E_DEMUX_2.K;
      E_SR.Q TO F_BOOL_TO_UINT.IN;
      E_SR_1.Q TO foldersWithNodeByteStringId_1.QI;
      E_SR_1.Q TO foldersWithNodeNumericId_1.QI;
      F_BOOL_TO_UINT_1.OUT TO E_DEMUX_2_1.K;
      E_SR_1.Q TO foldersWithNodeStringId_1.QI;
      E_SR_1.Q TO foldersWithNodeStringId_1.QI;
      E_SR_1.Q TO foldersWithNodeNumericId_1.QI;
      E_SR_1.Q TO FoldersNoBrowseName_1.QI;
      E_SR_1.Q TO foldersWithNodeByteStringId_1.QI;
      E_SR_1.Q TO foldersWithNodeByteStringId_1.QI;
      E_SR_1.Q TO foldersWithNodeNumericId_1.QI;
      E_SR_1.Q TO FoldersNoBrowseName_1.QI;
      E_SR_1.Q TO foldersWithNodeStringId_1.QI;
      E_SR_1.Q TO FoldersNoBrowseName_1.QI;
      E_SR_1.Q TO F_BOOL_TO_UINT_1.IN;
      E_SR_2.Q TO MethodOnlyBrowseName.QI;
      E_SR_2.Q TO MethodNumericNodeId.QI;
      E_SR_2.Q TO MethodBytestringNodeId.QI;
      E_SR_2.Q TO F_BOOL_TO_UINT_2.IN;
      F_BOOL_TO_UINT_2.OUT TO E_DEMUX_2_2.K;
      E_SR_2.Q TO MethodOnlyBrowseName.QI;
      E_SR_2.Q TO MethodBytestringNodeId.QI;
      E_SR_2.Q TO MethodNumericNodeId.QI;
      E_SR_2.Q TO MethodStringNodeId.QI;
    END_CONNECTIONS
  END_APPLICATION
  APPLICATION OpcUaBothWorking
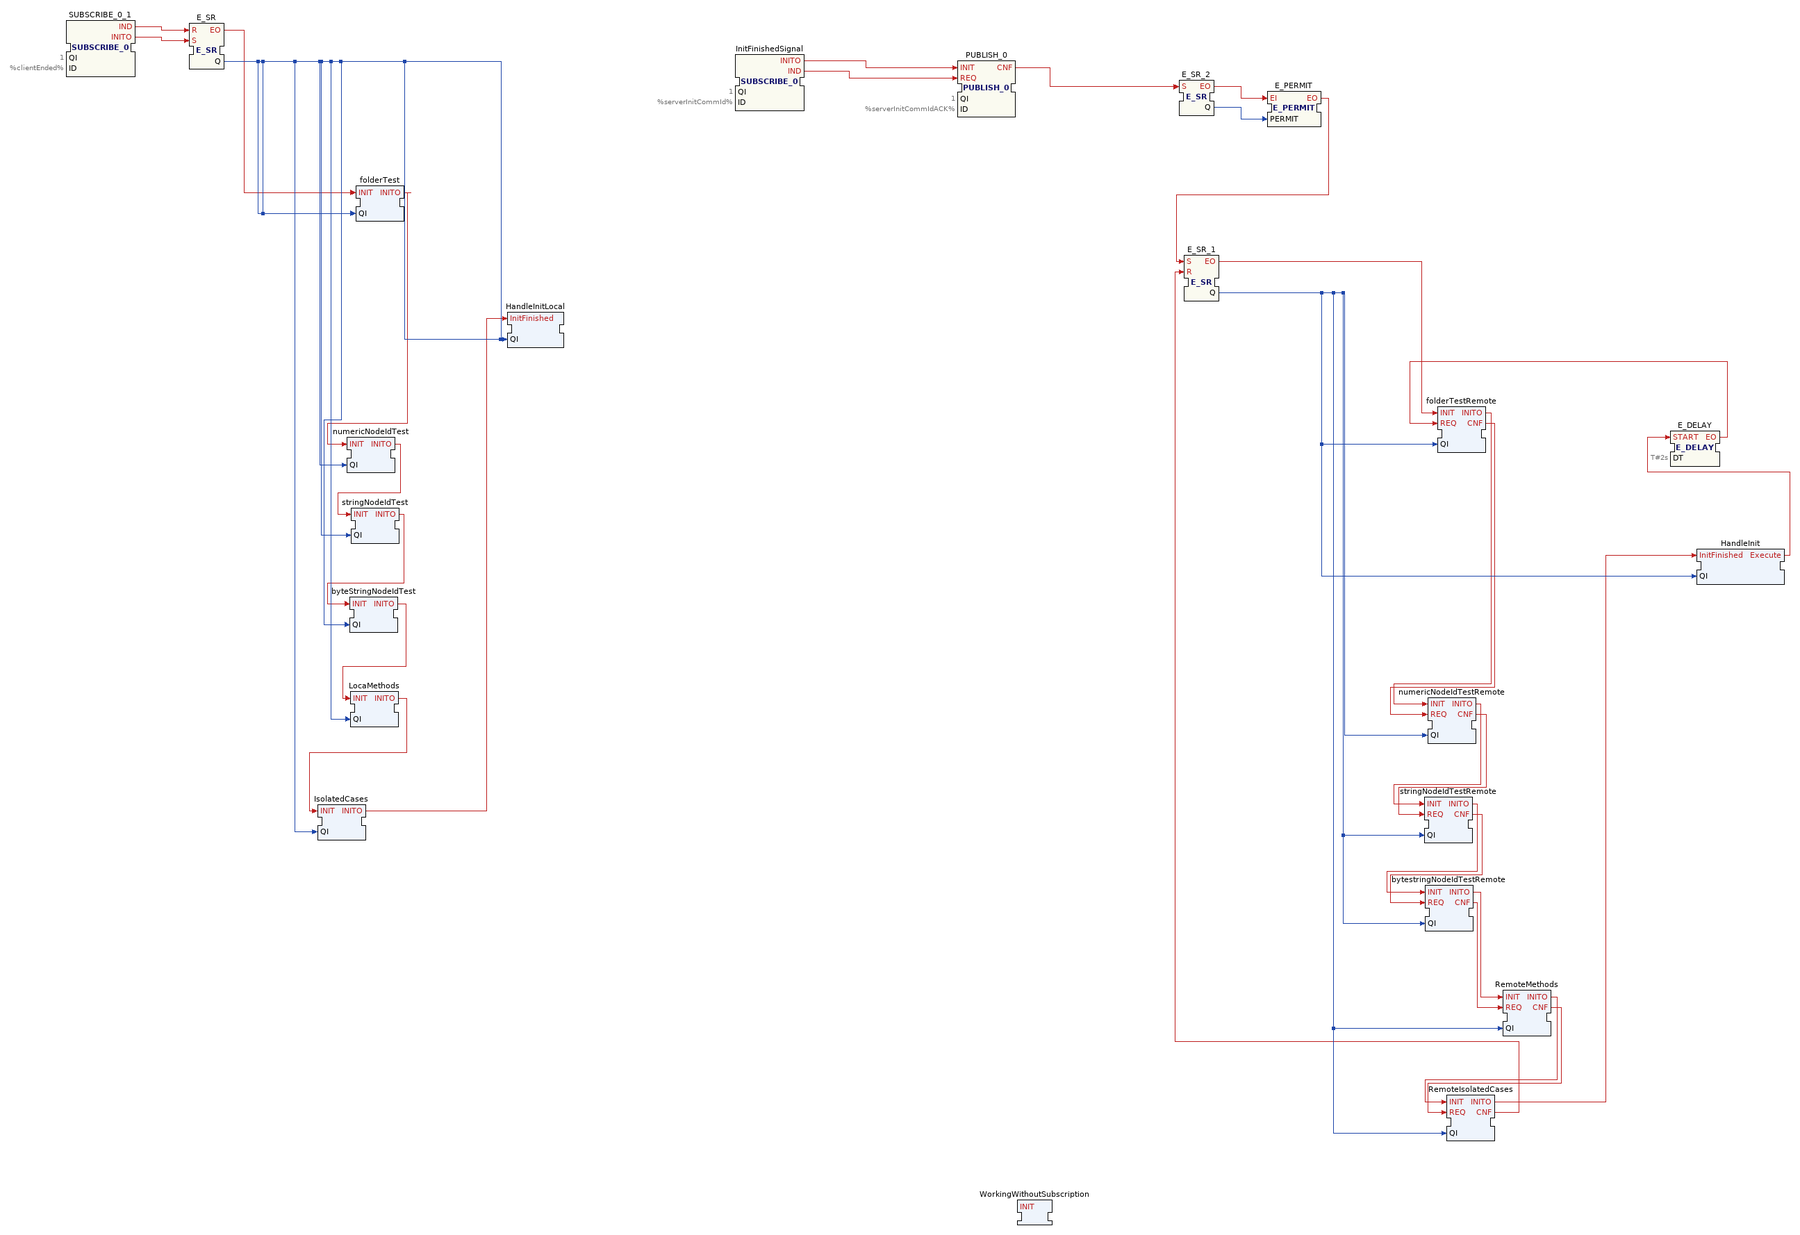
    FBS
      E_SR : E_SR;
      E_SR_1 : E_SR;
      InitFinishedSignal : SUBSCRIBE_0(QI := 1, ID := %serverInitCommId%);
      SUBSCRIBE_0_1 : SUBSCRIBE_0(QI := 1, ID := %clientEnded%);
      PUBLISH_0 : PUBLISH_0(QI := 1, ID := %serverInitCommIdACK%);
      E_SR_2 : E_SR;
      E_PERMIT : E_PERMIT;
      E_DELAY : E_DELAY(DT := T#2s);
    END_FBS
    SUBAPPLICATION folderTest
      EVENT_INPUT
        INIT;
      END_EVENT
      EVENT_OUTPUT
        INITO;
      END_EVENT
      VAR_INPUT
        QI : BOOL;
      END_VAR
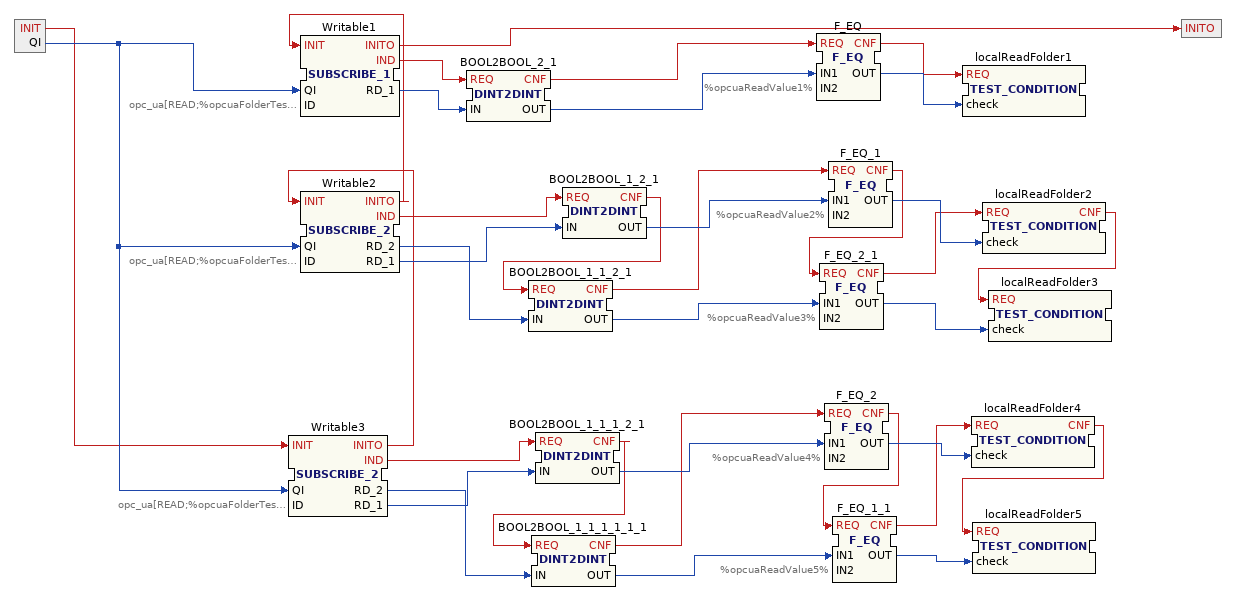
      FBS
        BOOL2BOOL_1_2_1 : DINT2DINT;
        BOOL2BOOL_2_1 : DINT2DINT;
        BOOL2BOOL_1_1_2_1 : DINT2DINT;
        BOOL2BOOL_1_1_1_2_1 : DINT2DINT;
        BOOL2BOOL_1_1_1_1_1_1 : DINT2DINT;
        Writable1 : SUBSCRIBE_1(ID := opc_ua[READ;%opcuaFolderTestOnlyBroseName1%]);
        Writable2 : SUBSCRIBE_2(ID := opc_ua[READ;%opcuaFolderTestOnlyBroseName2%]);
        Writable3 : SUBSCRIBE_2(ID := opc_ua[READ;%opcuaFolderTestOnlyBroseName3%]);
        localReadFolder1 : TEST_CONDITION;
        localReadFolder2 : TEST_CONDITION;
        localReadFolder3 : TEST_CONDITION;
        localReadFolder4 : TEST_CONDITION;
        localReadFolder5 : TEST_CONDITION;
        F_EQ : F_EQ(IN2 := %opcuaReadValue1%);
        F_EQ_1 : F_EQ(IN2 := %opcuaReadValue2%);
        F_EQ_2 : F_EQ(IN2 := %opcuaReadValue4%);
        F_EQ_1_1 : F_EQ(IN2 := %opcuaReadValue5%);
        F_EQ_2_1 : F_EQ(IN2 := %opcuaReadValue3%);
      END_FBS
      EVENT_CONNECTIONS
        Writable1.INITO TO INITO;
        Writable2.INITO TO Writable1.INIT;
        INIT TO Writable3.INIT;
        Writable3.INITO TO Writable2.INIT;
        Writable1.IND TO BOOL2BOOL_2_1.REQ;
        Writable2.IND TO BOOL2BOOL_1_2_1.REQ;
        BOOL2BOOL_1_2_1.CNF TO BOOL2BOOL_1_1_2_1.REQ;
        Writable3.IND TO BOOL2BOOL_1_1_1_2_1.REQ;
        BOOL2BOOL_1_1_1_2_1.CNF TO BOOL2BOOL_1_1_1_1_1_1.REQ;
        BOOL2BOOL_2_1.CNF TO F_EQ.REQ;
        F_EQ.CNF TO localReadFolder1.REQ;
        BOOL2BOOL_1_1_2_1.CNF TO F_EQ_1.REQ;
        F_EQ_1.CNF TO F_EQ_2_1.REQ;
        F_EQ_2_1.CNF TO localReadFolder2.REQ;
        BOOL2BOOL_1_1_1_1_1_1.CNF TO F_EQ_2.REQ;
        F_EQ_2.CNF TO F_EQ_1_1.REQ;
        F_EQ_1_1.CNF TO localReadFolder4.REQ;
        localReadFolder4.CNF TO localReadFolder5.REQ;
        localReadFolder2.CNF TO localReadFolder3.REQ;
      END_CONNECTIONS
      DATA_CONNECTIONS
        QI TO Writable1.QI;
        QI TO Writable2.QI;
        QI TO Writable3.QI;
        Writable1.RD_1 TO BOOL2BOOL_2_1.IN;
        Writable3.RD_2 TO BOOL2BOOL_1_1_1_1_1_1.IN;
        Writable3.RD_1 TO BOOL2BOOL_1_1_1_2_1.IN;
        Writable2.RD_2 TO BOOL2BOOL_1_1_2_1.IN;
        Writable2.RD_1 TO BOOL2BOOL_1_2_1.IN;
        BOOL2BOOL_2_1.OUT TO F_EQ.IN1;
        F_EQ.OUT TO localReadFolder1.check;
        BOOL2BOOL_1_1_2_1.OUT TO F_EQ_2_1.IN1;
        BOOL2BOOL_1_2_1.OUT TO F_EQ_1.IN1;
        BOOL2BOOL_1_1_1_2_1.OUT TO F_EQ_2.IN1;
        BOOL2BOOL_1_1_1_1_1_1.OUT TO F_EQ_1_1.IN1;
        F_EQ_1_1.OUT TO localReadFolder5.check;
        F_EQ_2.OUT TO localReadFolder4.check;
        F_EQ_2_1.OUT TO localReadFolder3.check;
        F_EQ_1.OUT TO localReadFolder2.check;
      END_CONNECTIONS
    END_SUBAPPLICATION
    SUBAPPLICATION folderTestRemote
      EVENT_INPUT
        INIT;
        REQ;
      END_EVENT
      EVENT_OUTPUT
        INITO;
        CNF;
      END_EVENT
      VAR_INPUT
        QI : BOOL;
      END_VAR
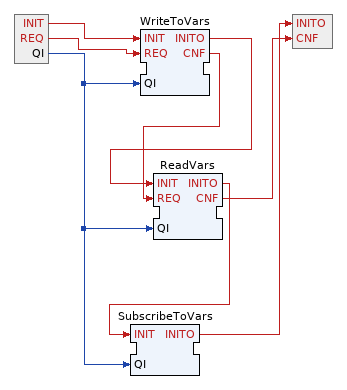
      SUBAPPLICATION SubscribeToVars
        EVENT_INPUT
          INIT;
        END_EVENT
        EVENT_OUTPUT
          INITO;
        END_EVENT
        VAR_INPUT
          QI : BOOL;
        END_VAR
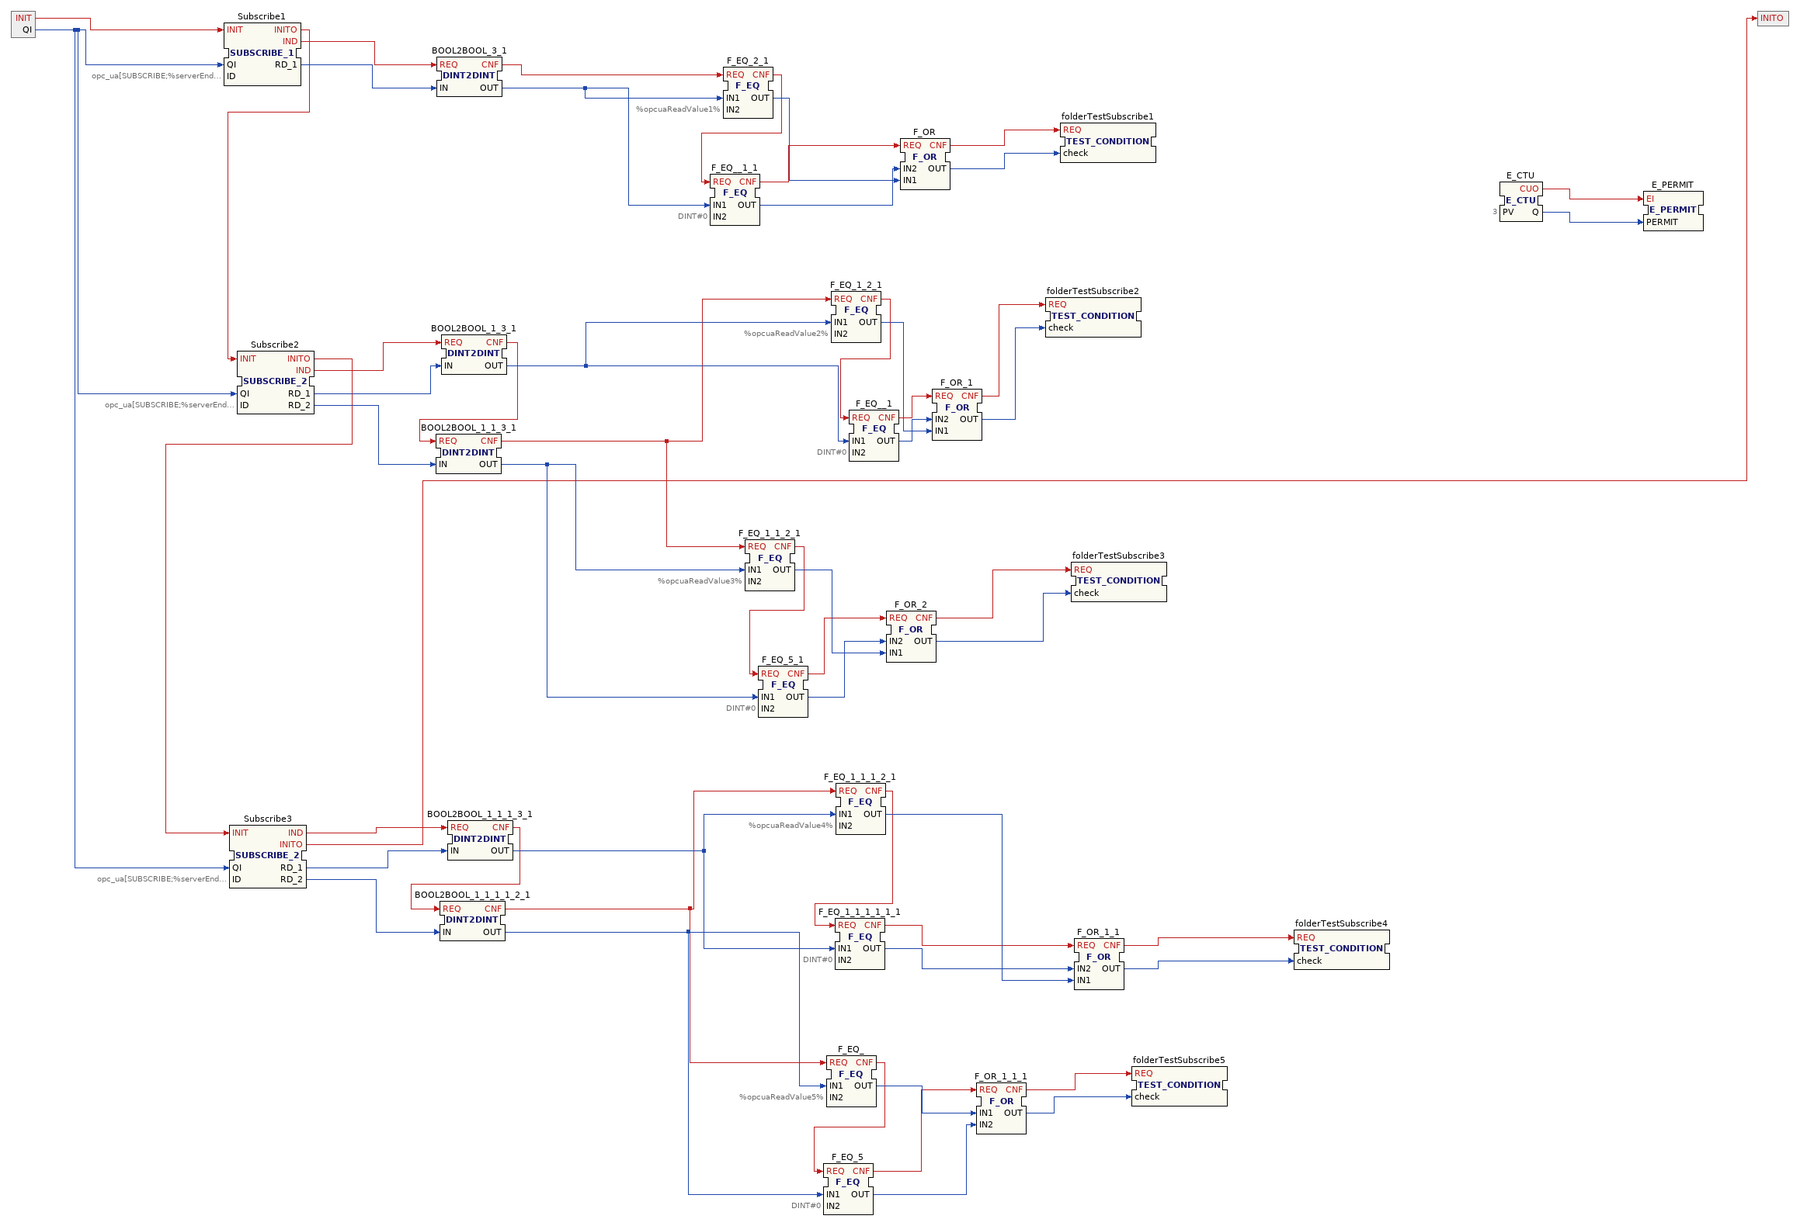
        FBS
          F_EQ_2_1 : F_EQ(IN2 := %opcuaReadValue1%);
          folderTestSubscribe4 : TEST_CONDITION;
          Subscribe3 : SUBSCRIBE_2(ID := opc_ua[SUBSCRIBE;%serverEndpoint%;%opcuaFolderTestOnlyBroseName3%]);
          F_EQ_1_1_1_2_1 : F_EQ(IN2 := %opcuaReadValue4%);
          folderTestSubscribe3 : TEST_CONDITION;
          F_EQ_1_1_1_1_1_1 : F_EQ(IN2 := DINT#0);
          F_EQ_1_1_2_1 : F_EQ(IN2 := %opcuaReadValue3%);
          folderTestSubscribe1 : TEST_CONDITION;
          folderTestSubscribe2 : TEST_CONDITION;
          Subscribe1 : SUBSCRIBE_1(ID := opc_ua[SUBSCRIBE;%serverEndpoint%;%opcuaFolderTestOnlyBroseName1%]);
          Subscribe2 : SUBSCRIBE_2(ID := opc_ua[SUBSCRIBE;%serverEndpoint%;%opcuaFolderTestOnlyBroseName2%]);
          BOOL2BOOL_1_1_3_1 : DINT2DINT;
          F_EQ_1_2_1 : F_EQ(IN2 := %opcuaReadValue2%);
          BOOL2BOOL_3_1 : DINT2DINT;
          BOOL2BOOL_1_1_1_3_1 : DINT2DINT;
          BOOL2BOOL_1_1_1_1_2_1 : DINT2DINT;
          BOOL2BOOL_1_3_1 : DINT2DINT;
          E_CTU : E_CTU(PV := 3);
          E_PERMIT : E_PERMIT;
          F_EQ_ : F_EQ(IN2 := %opcuaReadValue5%);
          folderTestSubscribe5 : TEST_CONDITION;
          F_EQ_5 : F_EQ(IN2 := DINT#0);
          F_EQ_5_1 : F_EQ(IN2 := DINT#0);
          F_EQ__1 : F_EQ(IN2 := DINT#0);
          F_EQ__1_1 : F_EQ(IN2 := DINT#0);
          F_OR : F_OR;
          F_OR_1 : F_OR;
          F_OR_2 : F_OR;
          F_OR_1_1 : F_OR;
          F_OR_1_1_1 : F_OR;
        END_FBS
        EVENT_CONNECTIONS
          Subscribe2.INITO TO Subscribe3.INIT;
          Subscribe3.IND TO BOOL2BOOL_1_1_1_3_1.REQ;
          Subscribe1.INITO TO Subscribe2.INIT;
          Subscribe1.IND TO BOOL2BOOL_3_1.REQ;
          Subscribe2.IND TO BOOL2BOOL_1_3_1.REQ;
          BOOL2BOOL_1_3_1.CNF TO BOOL2BOOL_1_1_3_1.REQ;
          BOOL2BOOL_1_1_1_3_1.CNF TO BOOL2BOOL_1_1_1_1_2_1.REQ;
          Subscribe3.INITO TO INITO;
          INIT TO Subscribe1.INIT;
          E_CTU.CUO TO E_PERMIT.EI;
          F_EQ__1_1.CNF TO F_OR.REQ;
          BOOL2BOOL_3_1.CNF TO F_EQ_2_1.REQ;
          F_EQ_2_1.CNF TO F_EQ__1_1.REQ;
          F_OR.CNF TO folderTestSubscribe1.REQ;
          F_OR_2.CNF TO folderTestSubscribe3.REQ;
          F_OR_1.CNF TO folderTestSubscribe2.REQ;
          F_EQ__1.CNF TO F_OR_1.REQ;
          F_EQ_1_2_1.CNF TO F_EQ__1.REQ;
          BOOL2BOOL_1_1_3_1.CNF TO F_EQ_1_2_1.REQ;
          BOOL2BOOL_1_1_3_1.CNF TO F_EQ_1_1_2_1.REQ;
          F_EQ_1_1_2_1.CNF TO F_EQ_5_1.REQ;
          F_EQ_5_1.CNF TO F_OR_2.REQ;
          F_OR_1_1.CNF TO folderTestSubscribe4.REQ;
          F_EQ_1_1_1_1_1_1.CNF TO F_OR_1_1.REQ;
          F_EQ_1_1_1_2_1.CNF TO F_EQ_1_1_1_1_1_1.REQ;
          BOOL2BOOL_1_1_1_1_2_1.CNF TO F_EQ_1_1_1_2_1.REQ;
          F_OR_1_1_1.CNF TO folderTestSubscribe5.REQ;
          BOOL2BOOL_1_1_1_1_2_1.CNF TO F_EQ_.REQ;
          F_EQ_.CNF TO F_EQ_5.REQ;
          F_EQ_5.CNF TO F_OR_1_1_1.REQ;
        END_CONNECTIONS
        DATA_CONNECTIONS
          BOOL2BOOL_3_1.OUT TO F_EQ_2_1.IN1;
          Subscribe3.RD_1 TO BOOL2BOOL_1_1_1_3_1.IN;
          Subscribe3.RD_2 TO BOOL2BOOL_1_1_1_1_2_1.IN;
          BOOL2BOOL_1_1_3_1.OUT TO F_EQ_1_1_2_1.IN1;
          Subscribe1.RD_1 TO BOOL2BOOL_3_1.IN;
          Subscribe2.RD_1 TO BOOL2BOOL_1_3_1.IN;
          Subscribe2.RD_2 TO BOOL2BOOL_1_1_3_1.IN;
          BOOL2BOOL_1_3_1.OUT TO F_EQ_1_2_1.IN1;
          QI TO Subscribe3.QI;
          QI TO Subscribe1.QI;
          QI TO Subscribe2.QI;
          E_CTU.Q TO E_PERMIT.PERMIT;
          BOOL2BOOL_1_1_1_1_2_1.OUT TO F_EQ_5.IN1;
          BOOL2BOOL_1_3_1.OUT TO F_EQ__1.IN1;
          BOOL2BOOL_1_1_3_1.OUT TO F_EQ_5_1.IN1;
          BOOL2BOOL_3_1.OUT TO F_EQ__1_1.IN1;
          BOOL2BOOL_1_1_1_3_1.OUT TO F_EQ_1_1_1_2_1.IN1;
          F_EQ__1_1.OUT TO F_OR.IN2;
          F_EQ_2_1.OUT TO F_OR.IN1;
          F_OR.OUT TO folderTestSubscribe1.check;
          F_EQ_5_1.OUT TO F_OR_2.IN2;
          F_EQ__1.OUT TO F_OR_1.IN2;
          F_EQ_1_2_1.OUT TO F_OR_1.IN1;
          F_OR_1.OUT TO folderTestSubscribe2.check;
          F_OR_2.OUT TO folderTestSubscribe3.check;
          F_OR_1_1.OUT TO folderTestSubscribe4.check;
          F_EQ_1_1_1_1_1_1.OUT TO F_OR_1_1.IN2;
          F_EQ_1_1_1_2_1.OUT TO F_OR_1_1.IN1;
          F_OR_1_1_1.OUT TO folderTestSubscribe5.check;
          F_EQ_.OUT TO F_OR_1_1_1.IN1;
          F_EQ_5.OUT TO F_OR_1_1_1.IN2;
          BOOL2BOOL_1_1_1_1_2_1.OUT TO F_EQ_.IN1;
          F_EQ_1_1_2_1.OUT TO F_OR_2.IN1;
          BOOL2BOOL_1_1_1_3_1.OUT TO F_EQ_1_1_1_1_1_1.IN1;
        END_CONNECTIONS
      END_SUBAPPLICATION
      SUBAPPLICATION WriteToVars
        EVENT_INPUT
          INIT;
          REQ;
        END_EVENT
        EVENT_OUTPUT
          INITO;
          CNF;
        END_EVENT
        VAR_INPUT
          QI : BOOL;
        END_VAR
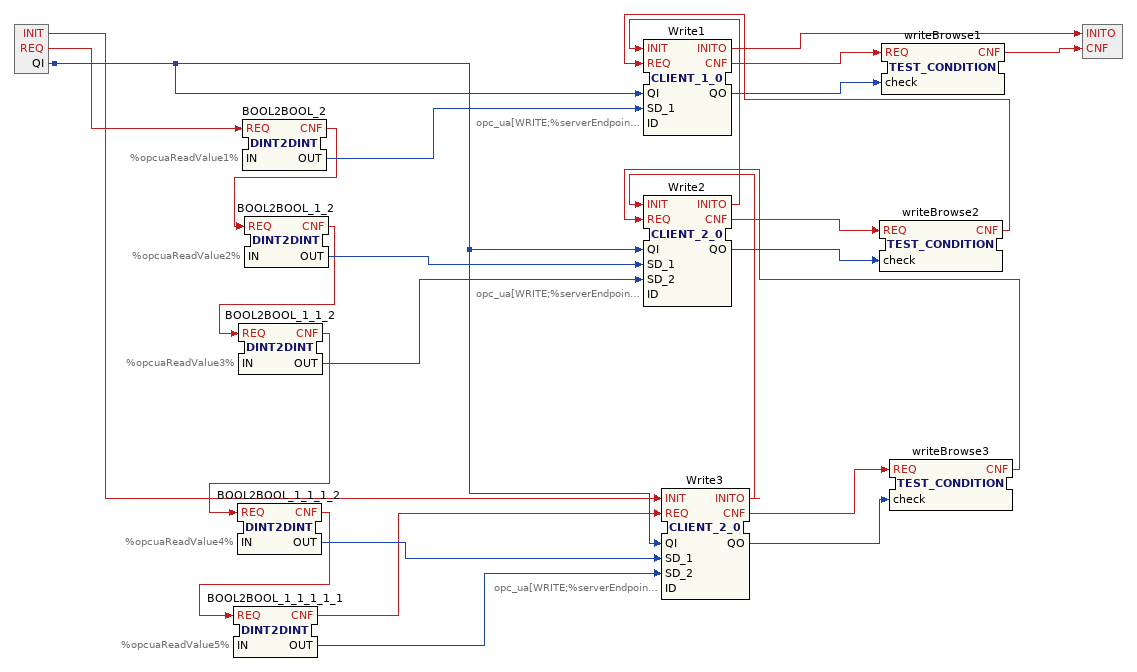
        FBS
          BOOL2BOOL_1_1_2 : DINT2DINT(IN := %opcuaReadValue3%);
          BOOL2BOOL_1_1_1_1_1 : DINT2DINT(IN := %opcuaReadValue5%);
          BOOL2BOOL_1_1_1_2 : DINT2DINT(IN := %opcuaReadValue4%);
          BOOL2BOOL_2 : DINT2DINT(IN := %opcuaReadValue1%);
          BOOL2BOOL_1_2 : DINT2DINT(IN := %opcuaReadValue2%);
          Write1 : CLIENT_1_0(ID := opc_ua[WRITE;%serverEndpoint%;%opcuaFolderTestOnlyBroseName1%]);
          Write3 : CLIENT_2_0(ID := opc_ua[WRITE;%serverEndpoint%;%opcuaFolderTestOnlyBroseName3%]);
          Write2 : CLIENT_2_0(ID := opc_ua[WRITE;%serverEndpoint%;%opcuaFolderTestOnlyBroseName2%]);
          writeBrowse1 : TEST_CONDITION;
          writeBrowse2 : TEST_CONDITION;
          writeBrowse3 : TEST_CONDITION;
        END_FBS
        EVENT_CONNECTIONS
          BOOL2BOOL_1_2.CNF TO BOOL2BOOL_1_1_2.REQ;
          BOOL2BOOL_1_1_2.CNF TO BOOL2BOOL_1_1_1_2.REQ;
          BOOL2BOOL_1_1_1_2.CNF TO BOOL2BOOL_1_1_1_1_1.REQ;
          BOOL2BOOL_2.CNF TO BOOL2BOOL_1_2.REQ;
          REQ TO BOOL2BOOL_2.REQ;
          Write1.INITO TO INITO;
          INIT TO Write3.INIT;
          BOOL2BOOL_1_1_1_1_1.CNF TO Write3.REQ;
          Write3.INITO TO Write2.INIT;
          Write2.INITO TO Write1.INIT;
          writeBrowse3.CNF TO Write2.REQ;
          Write3.CNF TO writeBrowse3.REQ;
          writeBrowse2.CNF TO Write1.REQ;
          Write2.CNF TO writeBrowse2.REQ;
          writeBrowse1.CNF TO CNF;
          Write1.CNF TO writeBrowse1.REQ;
        END_CONNECTIONS
        DATA_CONNECTIONS
          QI TO Write1.QI;
          BOOL2BOOL_2.OUT TO Write1.SD_1;
          QI TO Write3.QI;
          BOOL2BOOL_1_1_1_2.OUT TO Write3.SD_1;
          BOOL2BOOL_1_1_1_1_1.OUT TO Write3.SD_2;
          QI TO Write2.QI;
          BOOL2BOOL_1_2.OUT TO Write2.SD_1;
          BOOL2BOOL_1_1_2.OUT TO Write2.SD_2;
          Write1.QO TO writeBrowse1.check;
          Write2.QO TO writeBrowse2.check;
          Write3.QO TO writeBrowse3.check;
        END_CONNECTIONS
      END_SUBAPPLICATION
      SUBAPPLICATION ReadVars
        EVENT_INPUT
          INIT;
          REQ;
        END_EVENT
        EVENT_OUTPUT
          INITO;
          CNF;
        END_EVENT
        VAR_INPUT
          QI : BOOL;
        END_VAR
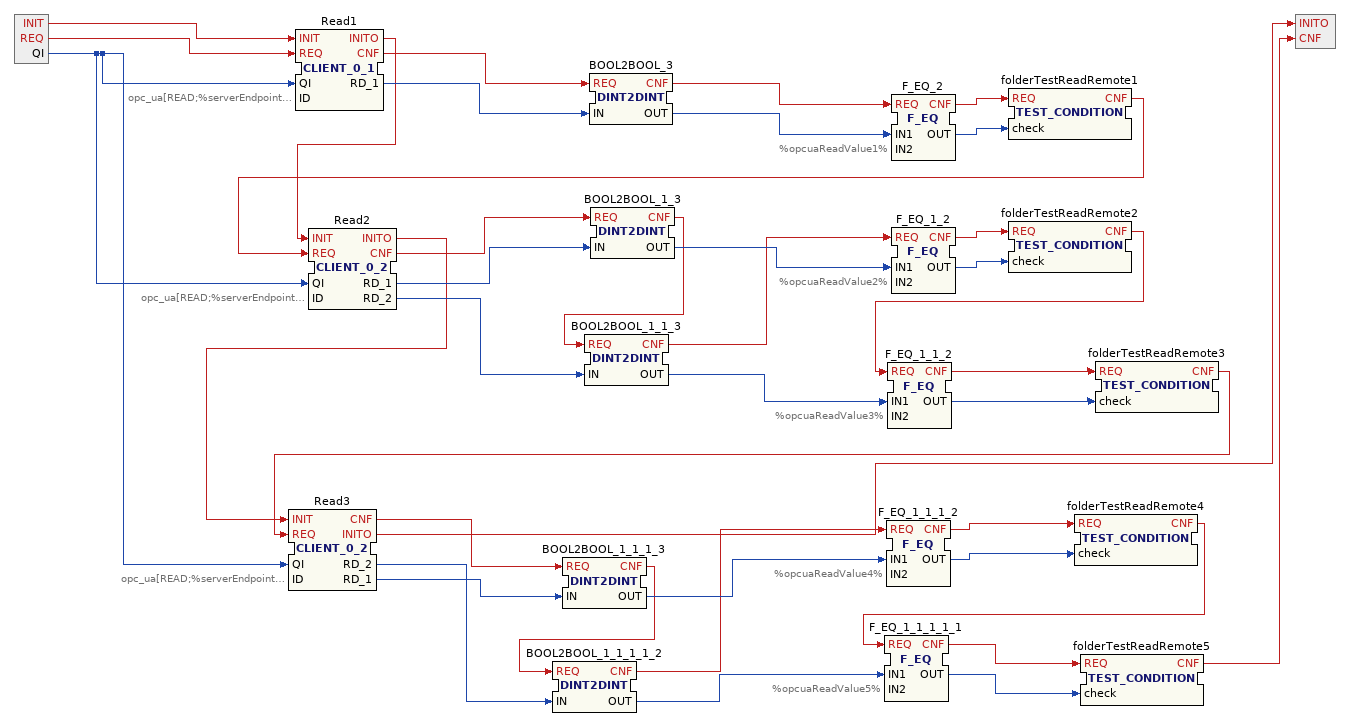
        FBS
          Read1 : CLIENT_0_1(ID := opc_ua[READ;%serverEndpoint%;%opcuaFolderTestOnlyBroseName1%]);
          Read2 : CLIENT_0_2(ID := opc_ua[READ;%serverEndpoint%;%opcuaFolderTestOnlyBroseName2%]);
          F_EQ_1_1_1_2 : F_EQ(IN2 := %opcuaReadValue4%);
          folderTestReadRemote4 : TEST_CONDITION;
          BOOL2BOOL_1_3 : DINT2DINT;
          F_EQ_1_1_1_1_1 : F_EQ(IN2 := %opcuaReadValue5%);
          folderTestReadRemote3 : TEST_CONDITION;
          BOOL2BOOL_1_1_3 : DINT2DINT;
          BOOL2BOOL_1_1_1_1_2 : DINT2DINT;
          BOOL2BOOL_1_1_1_3 : DINT2DINT;
          folderTestReadRemote2 : TEST_CONDITION;
          F_EQ_1_1_2 : F_EQ(IN2 := %opcuaReadValue3%);
          F_EQ_2 : F_EQ(IN2 := %opcuaReadValue1%);
          F_EQ_1_2 : F_EQ(IN2 := %opcuaReadValue2%);
          Read3 : CLIENT_0_2(ID := opc_ua[READ;%serverEndpoint%;%opcuaFolderTestOnlyBroseName3%]);
          folderTestReadRemote5 : TEST_CONDITION;
          folderTestReadRemote1 : TEST_CONDITION;
          BOOL2BOOL_3 : DINT2DINT;
        END_FBS
        EVENT_CONNECTIONS
          Read1.INITO TO Read2.INIT;
          Read1.CNF TO BOOL2BOOL_3.REQ;
          folderTestReadRemote1.CNF TO Read2.REQ;
          Read2.INITO TO Read3.INIT;
          Read2.CNF TO BOOL2BOOL_1_3.REQ;
          BOOL2BOOL_1_1_1_1_2.CNF TO F_EQ_1_1_1_2.REQ;
          F_EQ_1_1_1_2.CNF TO folderTestReadRemote4.REQ;
          folderTestReadRemote4.CNF TO F_EQ_1_1_1_1_1.REQ;
          BOOL2BOOL_1_3.CNF TO BOOL2BOOL_1_1_3.REQ;
          F_EQ_1_1_1_1_1.CNF TO folderTestReadRemote5.REQ;
          F_EQ_1_1_2.CNF TO folderTestReadRemote3.REQ;
          folderTestReadRemote3.CNF TO Read3.REQ;
          BOOL2BOOL_1_1_3.CNF TO F_EQ_1_2.REQ;
          BOOL2BOOL_1_1_1_3.CNF TO BOOL2BOOL_1_1_1_1_2.REQ;
          Read3.CNF TO BOOL2BOOL_1_1_1_3.REQ;
          F_EQ_1_2.CNF TO folderTestReadRemote2.REQ;
          folderTestReadRemote2.CNF TO F_EQ_1_1_2.REQ;
          BOOL2BOOL_3.CNF TO F_EQ_2.REQ;
          F_EQ_2.CNF TO folderTestReadRemote1.REQ;
          INIT TO Read1.INIT;
          REQ TO Read1.REQ;
          Read3.INITO TO INITO;
          folderTestReadRemote5.CNF TO CNF;
        END_CONNECTIONS
        DATA_CONNECTIONS
          Read1.RD_1 TO BOOL2BOOL_3.IN;
          Read2.RD_1 TO BOOL2BOOL_1_3.IN;
          Read2.RD_2 TO BOOL2BOOL_1_1_3.IN;
          BOOL2BOOL_1_1_1_3.OUT TO F_EQ_1_1_1_2.IN1;
          F_EQ_1_1_1_2.OUT TO folderTestReadRemote4.check;
          BOOL2BOOL_1_3.OUT TO F_EQ_1_2.IN1;
          BOOL2BOOL_1_1_1_1_2.OUT TO F_EQ_1_1_1_1_1.IN1;
          F_EQ_1_1_1_1_1.OUT TO folderTestReadRemote5.check;
          F_EQ_1_1_2.OUT TO folderTestReadRemote3.check;
          BOOL2BOOL_1_1_3.OUT TO F_EQ_1_1_2.IN1;
          Read3.RD_2 TO BOOL2BOOL_1_1_1_1_2.IN;
          Read3.RD_1 TO BOOL2BOOL_1_1_1_3.IN;
          F_EQ_1_2.OUT TO folderTestReadRemote2.check;
          BOOL2BOOL_3.OUT TO F_EQ_2.IN1;
          F_EQ_2.OUT TO folderTestReadRemote1.check;
          QI TO Read1.QI;
          QI TO Read2.QI;
          QI TO Read3.QI;
        END_CONNECTIONS
      END_SUBAPPLICATION
      EVENT_CONNECTIONS
        ReadVars.INITO TO SubscribeToVars.INIT;
        WriteToVars.INITO TO ReadVars.INIT;
        SubscribeToVars.INITO TO INITO;
        INIT TO WriteToVars.INIT;
        REQ TO WriteToVars.REQ;
        ReadVars.CNF TO CNF;
        WriteToVars.CNF TO ReadVars.REQ;
      END_CONNECTIONS
      DATA_CONNECTIONS
        QI TO SubscribeToVars.QI;
        QI TO ReadVars.QI;
        QI TO WriteToVars.QI;
      END_CONNECTIONS
    END_SUBAPPLICATION
    SUBAPPLICATION HandleInit
      EVENT_INPUT
        InitFinished;
      END_EVENT
      EVENT_OUTPUT
        Execute;
      END_EVENT
      VAR_INPUT
        QI : BOOL;
      END_VAR
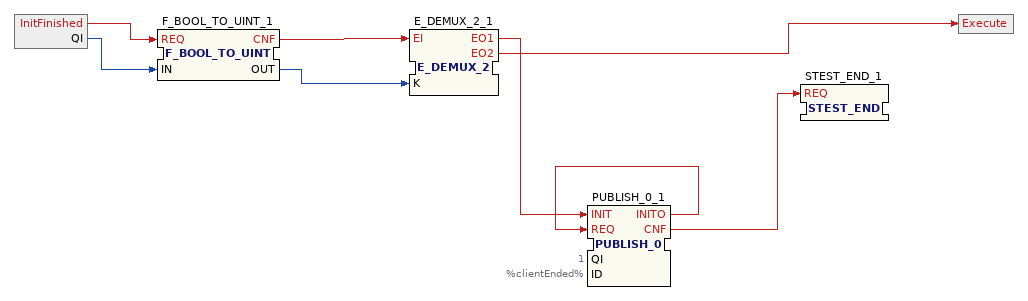
      FBS
        STEST_END_1 : STEST_END;
        E_DEMUX_2_1 : E_DEMUX_2;
        F_BOOL_TO_UINT_1 : F_BOOL_TO_UINT;
        PUBLISH_0_1 : PUBLISH_0(QI := 1, ID := %clientEnded%);
      END_FBS
      EVENT_CONNECTIONS
        F_BOOL_TO_UINT_1.CNF TO E_DEMUX_2_1.EI;
        E_DEMUX_2_1.EO1 TO PUBLISH_0_1.INIT;
        PUBLISH_0_1.INITO TO PUBLISH_0_1.REQ;
        E_DEMUX_2_1.EO2 TO Execute;
        InitFinished TO F_BOOL_TO_UINT_1.REQ;
        PUBLISH_0_1.CNF TO STEST_END_1.REQ;
      END_CONNECTIONS
      DATA_CONNECTIONS
        F_BOOL_TO_UINT_1.OUT TO E_DEMUX_2_1.K;
        QI TO F_BOOL_TO_UINT_1.IN;
      END_CONNECTIONS
    END_SUBAPPLICATION
    SUBAPPLICATION HandleInitLocal
      EVENT_INPUT
        InitFinished;
      END_EVENT
      VAR_INPUT
        QI : BOOL;
      END_VAR
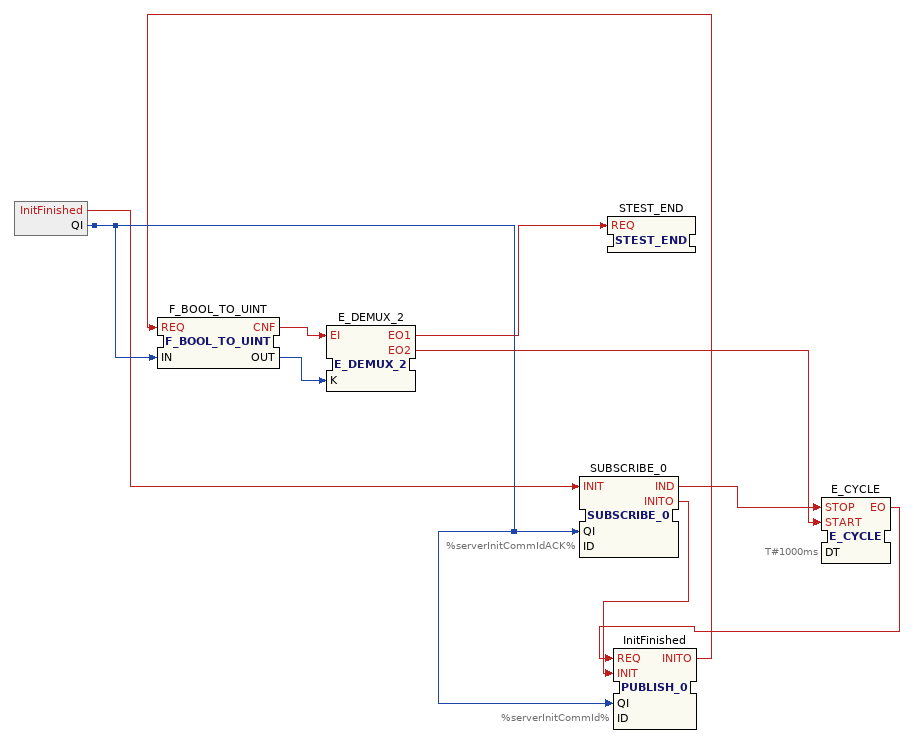
      FBS
        InitFinished : PUBLISH_0(ID := %serverInitCommId%);
        SUBSCRIBE_0 : SUBSCRIBE_0(ID := %serverInitCommIdACK%);
        E_CYCLE : E_CYCLE(DT := T#1000ms);
        E_DEMUX_2 : E_DEMUX_2;
        STEST_END : STEST_END;
        F_BOOL_TO_UINT : F_BOOL_TO_UINT;
      END_FBS
      EVENT_CONNECTIONS
        E_CYCLE.EO TO InitFinished.REQ;
        SUBSCRIBE_0.IND TO E_CYCLE.STOP;
        F_BOOL_TO_UINT.CNF TO E_DEMUX_2.EI;
        E_DEMUX_2.EO1 TO STEST_END.REQ;
        InitFinished TO SUBSCRIBE_0.INIT;
        SUBSCRIBE_0.INITO TO InitFinished.INIT;
        InitFinished.INITO TO F_BOOL_TO_UINT.REQ;
        E_DEMUX_2.EO2 TO E_CYCLE.START;
      END_CONNECTIONS
      DATA_CONNECTIONS
        F_BOOL_TO_UINT.OUT TO E_DEMUX_2.K;
        QI TO F_BOOL_TO_UINT.IN;
        QI TO SUBSCRIBE_0.QI;
        QI TO InitFinished.QI;
      END_CONNECTIONS
    END_SUBAPPLICATION
    SUBAPPLICATION numericNodeIdTestRemote
      EVENT_INPUT
        INIT;
        REQ;
      END_EVENT
      EVENT_OUTPUT
        INITO;
        CNF;
      END_EVENT
      VAR_INPUT
        QI : BOOL;
      END_VAR
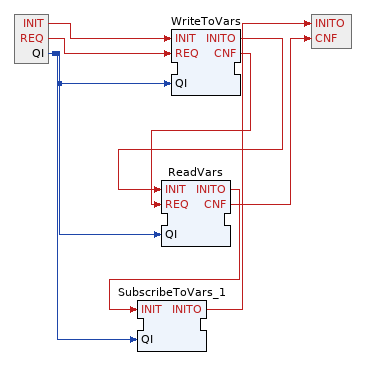
      SUBAPPLICATION WriteToVars
        EVENT_INPUT
          INIT;
          REQ;
        END_EVENT
        EVENT_OUTPUT
          INITO;
          CNF;
        END_EVENT
        VAR_INPUT
          QI : BOOL;
        END_VAR
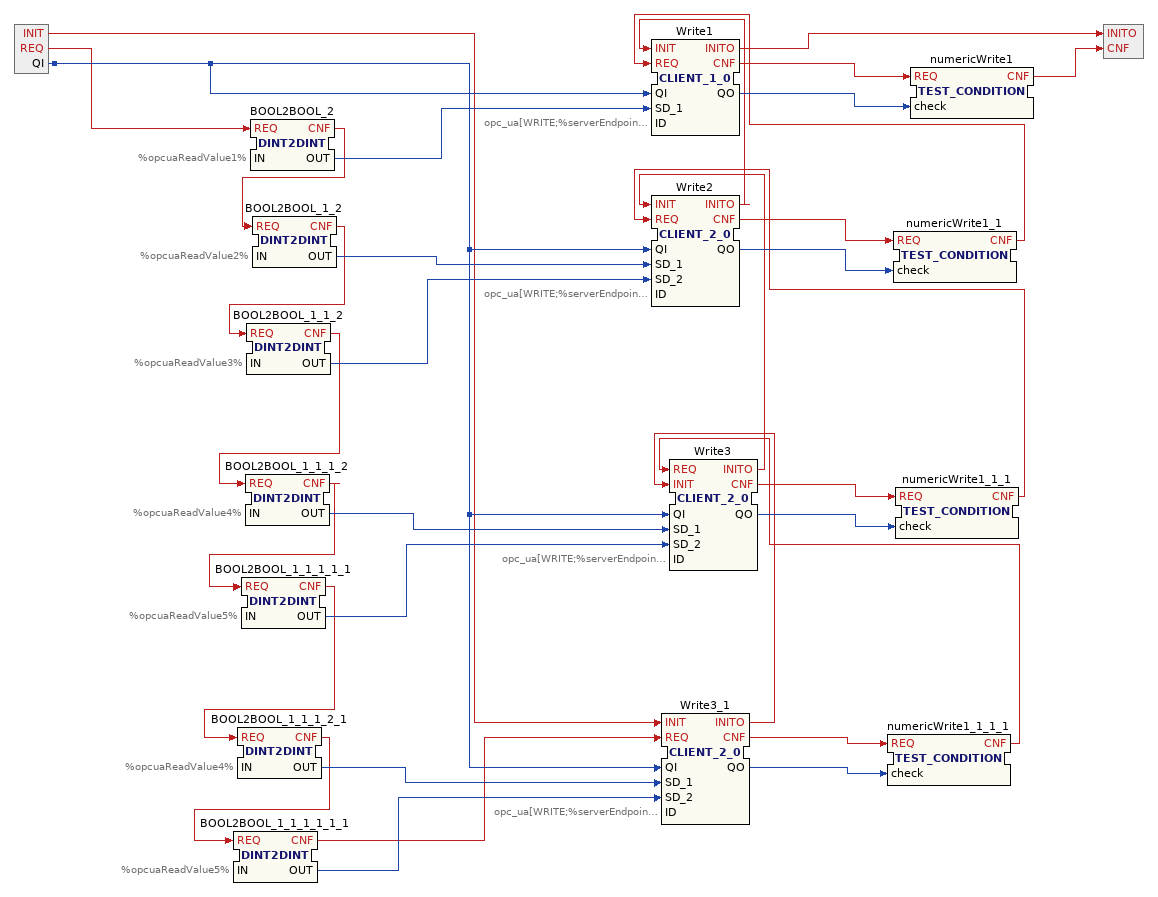
        FBS
          BOOL2BOOL_1_1_2 : DINT2DINT(IN := %opcuaReadValue3%);
          BOOL2BOOL_1_1_1_1_1 : DINT2DINT(IN := %opcuaReadValue5%);
          BOOL2BOOL_1_1_1_2 : DINT2DINT(IN := %opcuaReadValue4%);
          BOOL2BOOL_2 : DINT2DINT(IN := %opcuaReadValue1%);
          BOOL2BOOL_1_2 : DINT2DINT(IN := %opcuaReadValue2%);
          BOOL2BOOL_1_1_1_2_1 : DINT2DINT(IN := %opcuaReadValue4%);
          BOOL2BOOL_1_1_1_1_1_1 : DINT2DINT(IN := %opcuaReadValue5%);
          Write1 : CLIENT_1_0(ID := opc_ua[WRITE;%serverEndpoint%;%opcuaFolderTestWithNodeIdNumeric1%]);
          Write3 : CLIENT_2_0(ID := opc_ua[WRITE;%serverEndpoint%;%opcuaFolderTestWithNodeIdNumeric3%]);
          Write2 : CLIENT_2_0(ID := opc_ua[WRITE;%serverEndpoint%;%opcuaFolderTestWithNodeIdNumeric2%]);
          numericWrite1 : TEST_CONDITION;
          numericWrite1_1 : TEST_CONDITION;
          numericWrite1_1_1 : TEST_CONDITION;
          numericWrite1_1_1_1 : TEST_CONDITION;
          Write3_1 : CLIENT_2_0(ID := opc_ua[WRITE;%serverEndpoint%;,1:i=12348;,1:i=12349]);
        END_FBS
        EVENT_CONNECTIONS
          BOOL2BOOL_1_2.CNF TO BOOL2BOOL_1_1_2.REQ;
          BOOL2BOOL_1_1_2.CNF TO BOOL2BOOL_1_1_1_2.REQ;
          BOOL2BOOL_1_1_1_2.CNF TO BOOL2BOOL_1_1_1_1_1.REQ;
          BOOL2BOOL_2.CNF TO BOOL2BOOL_1_2.REQ;
          REQ TO BOOL2BOOL_2.REQ;
          BOOL2BOOL_1_1_1_2_1.CNF TO BOOL2BOOL_1_1_1_1_1_1.REQ;
          BOOL2BOOL_1_1_1_1_1.CNF TO BOOL2BOOL_1_1_1_2_1.REQ;
          Write1.INITO TO INITO;
          Write3.INITO TO Write2.INIT;
          Write2.INITO TO Write1.INIT;
          numericWrite1_1.CNF TO Write1.REQ;
          numericWrite1.CNF TO CNF;
          Write1.CNF TO numericWrite1.REQ;
          numericWrite1_1_1.CNF TO Write2.REQ;
          Write3.CNF TO numericWrite1_1_1.REQ;
          numericWrite1_1_1_1.CNF TO Write3.REQ;
          INIT TO Write3_1.INIT;
          BOOL2BOOL_1_1_1_1_1_1.CNF TO Write3_1.REQ;
          Write3_1.INITO TO Write3.INIT;
          Write3_1.CNF TO numericWrite1_1_1_1.REQ;
          Write2.CNF TO numericWrite1_1.REQ;
        END_CONNECTIONS
        DATA_CONNECTIONS
          QI TO Write1.QI;
          BOOL2BOOL_2.OUT TO Write1.SD_1;
          QI TO Write3.QI;
          BOOL2BOOL_1_1_1_2.OUT TO Write3.SD_1;
          BOOL2BOOL_1_1_1_1_1.OUT TO Write3.SD_2;
          QI TO Write2.QI;
          BOOL2BOOL_1_2.OUT TO Write2.SD_1;
          BOOL2BOOL_1_1_2.OUT TO Write2.SD_2;
          Write3.QO TO numericWrite1_1_1.check;
          Write1.QO TO numericWrite1.check;
          Write2.QO TO numericWrite1_1.check;
          QI TO Write3_1.QI;
          BOOL2BOOL_1_1_1_2_1.OUT TO Write3_1.SD_1;
          BOOL2BOOL_1_1_1_1_1_1.OUT TO Write3_1.SD_2;
          Write3_1.QO TO numericWrite1_1_1_1.check;
        END_CONNECTIONS
      END_SUBAPPLICATION
      SUBAPPLICATION ReadVars
        EVENT_INPUT
          INIT;
          REQ;
        END_EVENT
        EVENT_OUTPUT
          INITO;
          CNF;
        END_EVENT
        VAR_INPUT
          QI : BOOL;
        END_VAR
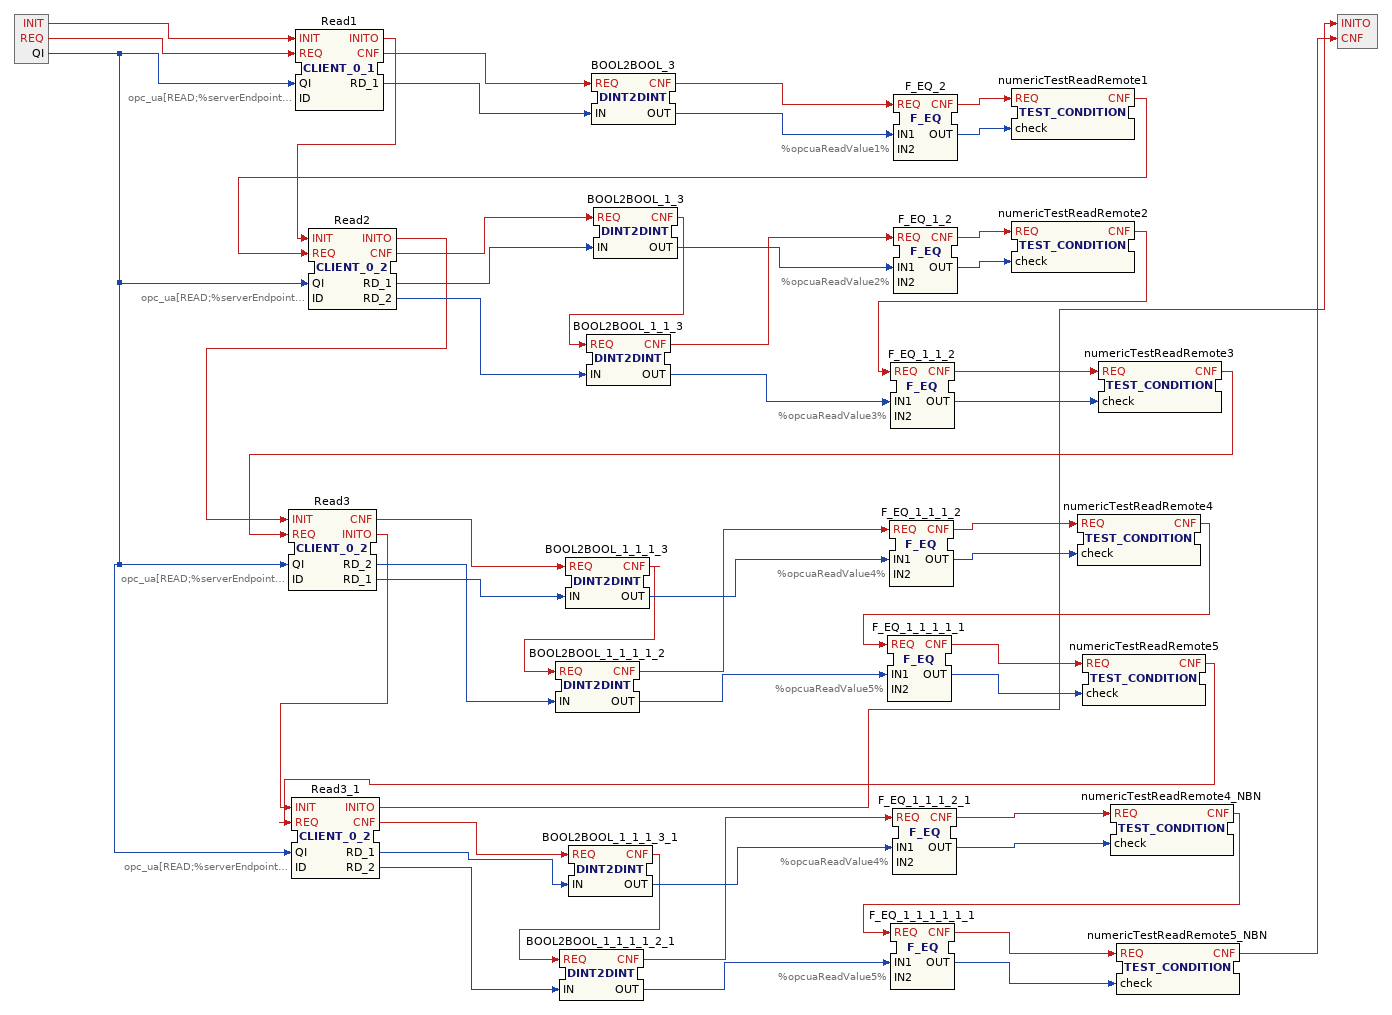
        FBS
          Read1 : CLIENT_0_1(ID := opc_ua[READ;%serverEndpoint%;%opcuaFolderTestWithNodeIdNumeric1%]);
          Read2 : CLIENT_0_2(ID := opc_ua[READ;%serverEndpoint%;%opcuaFolderTestWithNodeIdNumeric2%]);
          F_EQ_1_1_1_2 : F_EQ(IN2 := %opcuaReadValue4%);
          numericTestReadRemote4 : TEST_CONDITION;
          BOOL2BOOL_1_3 : DINT2DINT;
          F_EQ_1_1_1_1_1 : F_EQ(IN2 := %opcuaReadValue5%);
          numericTestReadRemote3 : TEST_CONDITION;
          BOOL2BOOL_1_1_3 : DINT2DINT;
          BOOL2BOOL_1_1_1_1_2 : DINT2DINT;
          BOOL2BOOL_1_1_1_3 : DINT2DINT;
          numericTestReadRemote2 : TEST_CONDITION;
          F_EQ_1_1_2 : F_EQ(IN2 := %opcuaReadValue3%);
          F_EQ_2 : F_EQ(IN2 := %opcuaReadValue1%);
          F_EQ_1_2 : F_EQ(IN2 := %opcuaReadValue2%);
          Read3 : CLIENT_0_2(ID := opc_ua[READ;%serverEndpoint%;%opcuaFolderTestWithNodeIdNumeric3%]);
          numericTestReadRemote5 : TEST_CONDITION;
          numericTestReadRemote1 : TEST_CONDITION;
          BOOL2BOOL_3 : DINT2DINT;
          F_EQ_1_1_1_2_1 : F_EQ(IN2 := %opcuaReadValue4%);
          Read3_1 : CLIENT_0_2(ID := opc_ua[READ;%serverEndpoint%;,1:i=12348;,1:i=12349]);
          F_EQ_1_1_1_1_1_1 : F_EQ(IN2 := %opcuaReadValue5%);
          BOOL2BOOL_1_1_1_1_2_1 : DINT2DINT;
          BOOL2BOOL_1_1_1_3_1 : DINT2DINT;
          numericTestReadRemote4_NBN : TEST_CONDITION;
          numericTestReadRemote5_NBN : TEST_CONDITION;
        END_FBS
        EVENT_CONNECTIONS
          Read1.INITO TO Read2.INIT;
          numericTestReadRemote1.CNF TO Read2.REQ;
          Read2.INITO TO Read3.INIT;
          Read2.CNF TO BOOL2BOOL_1_3.REQ;
          BOOL2BOOL_1_1_1_1_2.CNF TO F_EQ_1_1_1_2.REQ;
          F_EQ_1_1_1_2.CNF TO numericTestReadRemote4.REQ;
          numericTestReadRemote4.CNF TO F_EQ_1_1_1_1_1.REQ;
          BOOL2BOOL_1_3.CNF TO BOOL2BOOL_1_1_3.REQ;
          F_EQ_1_1_1_1_1.CNF TO numericTestReadRemote5.REQ;
          F_EQ_1_1_2.CNF TO numericTestReadRemote3.REQ;
          numericTestReadRemote3.CNF TO Read3.REQ;
          BOOL2BOOL_1_1_3.CNF TO F_EQ_1_2.REQ;
          BOOL2BOOL_1_1_1_3.CNF TO BOOL2BOOL_1_1_1_1_2.REQ;
          Read3.CNF TO BOOL2BOOL_1_1_1_3.REQ;
          F_EQ_1_2.CNF TO numericTestReadRemote2.REQ;
          INIT TO Read1.INIT;
          REQ TO Read1.REQ;
          Read1.CNF TO BOOL2BOOL_3.REQ;
          BOOL2BOOL_3.CNF TO F_EQ_2.REQ;
          F_EQ_2.CNF TO numericTestReadRemote1.REQ;
          numericTestReadRemote2.CNF TO F_EQ_1_1_2.REQ;
          Read3_1.INITO TO INITO;
          Read3.INITO TO Read3_1.INIT;
          Read3_1.CNF TO BOOL2BOOL_1_1_1_3_1.REQ;
          BOOL2BOOL_1_1_1_3_1.CNF TO BOOL2BOOL_1_1_1_1_2_1.REQ;
          BOOL2BOOL_1_1_1_1_2_1.CNF TO F_EQ_1_1_1_2_1.REQ;
          F_EQ_1_1_1_2_1.CNF TO numericTestReadRemote4_NBN.REQ;
          F_EQ_1_1_1_1_1_1.CNF TO numericTestReadRemote5_NBN.REQ;
          numericTestReadRemote4_NBN.CNF TO F_EQ_1_1_1_1_1_1.REQ;
          numericTestReadRemote5_NBN.CNF TO CNF;
          numericTestReadRemote5.CNF TO Read3_1.REQ;
        END_CONNECTIONS
        DATA_CONNECTIONS
          Read1.RD_1 TO BOOL2BOOL_3.IN;
          Read2.RD_1 TO BOOL2BOOL_1_3.IN;
          Read2.RD_2 TO BOOL2BOOL_1_1_3.IN;
          BOOL2BOOL_1_1_1_3.OUT TO F_EQ_1_1_1_2.IN1;
          F_EQ_1_1_1_2.OUT TO numericTestReadRemote4.check;
          BOOL2BOOL_1_3.OUT TO F_EQ_1_2.IN1;
          BOOL2BOOL_1_1_1_1_2.OUT TO F_EQ_1_1_1_1_1.IN1;
          F_EQ_1_1_1_1_1.OUT TO numericTestReadRemote5.check;
          F_EQ_1_1_2.OUT TO numericTestReadRemote3.check;
          BOOL2BOOL_1_1_3.OUT TO F_EQ_1_1_2.IN1;
          Read3.RD_2 TO BOOL2BOOL_1_1_1_1_2.IN;
          Read3.RD_1 TO BOOL2BOOL_1_1_1_3.IN;
          F_EQ_1_2.OUT TO numericTestReadRemote2.check;
          BOOL2BOOL_3.OUT TO F_EQ_2.IN1;
          F_EQ_2.OUT TO numericTestReadRemote1.check;
          QI TO Read1.QI;
          QI TO Read2.QI;
          QI TO Read3.QI;
          Read3_1.RD_1 TO BOOL2BOOL_1_1_1_3_1.IN;
          Read3_1.RD_2 TO BOOL2BOOL_1_1_1_1_2_1.IN;
          BOOL2BOOL_1_1_1_1_2_1.OUT TO F_EQ_1_1_1_1_1_1.IN1;
          BOOL2BOOL_1_1_1_3_1.OUT TO F_EQ_1_1_1_2_1.IN1;
          F_EQ_1_1_1_2_1.OUT TO numericTestReadRemote4_NBN.check;
          F_EQ_1_1_1_1_1_1.OUT TO numericTestReadRemote5_NBN.check;
          QI TO Read3_1.QI;
        END_CONNECTIONS
      END_SUBAPPLICATION
      SUBAPPLICATION SubscribeToVars_1
        EVENT_INPUT
          INIT;
        END_EVENT
        EVENT_OUTPUT
          INITO;
        END_EVENT
        VAR_INPUT
          QI : BOOL;
        END_VAR
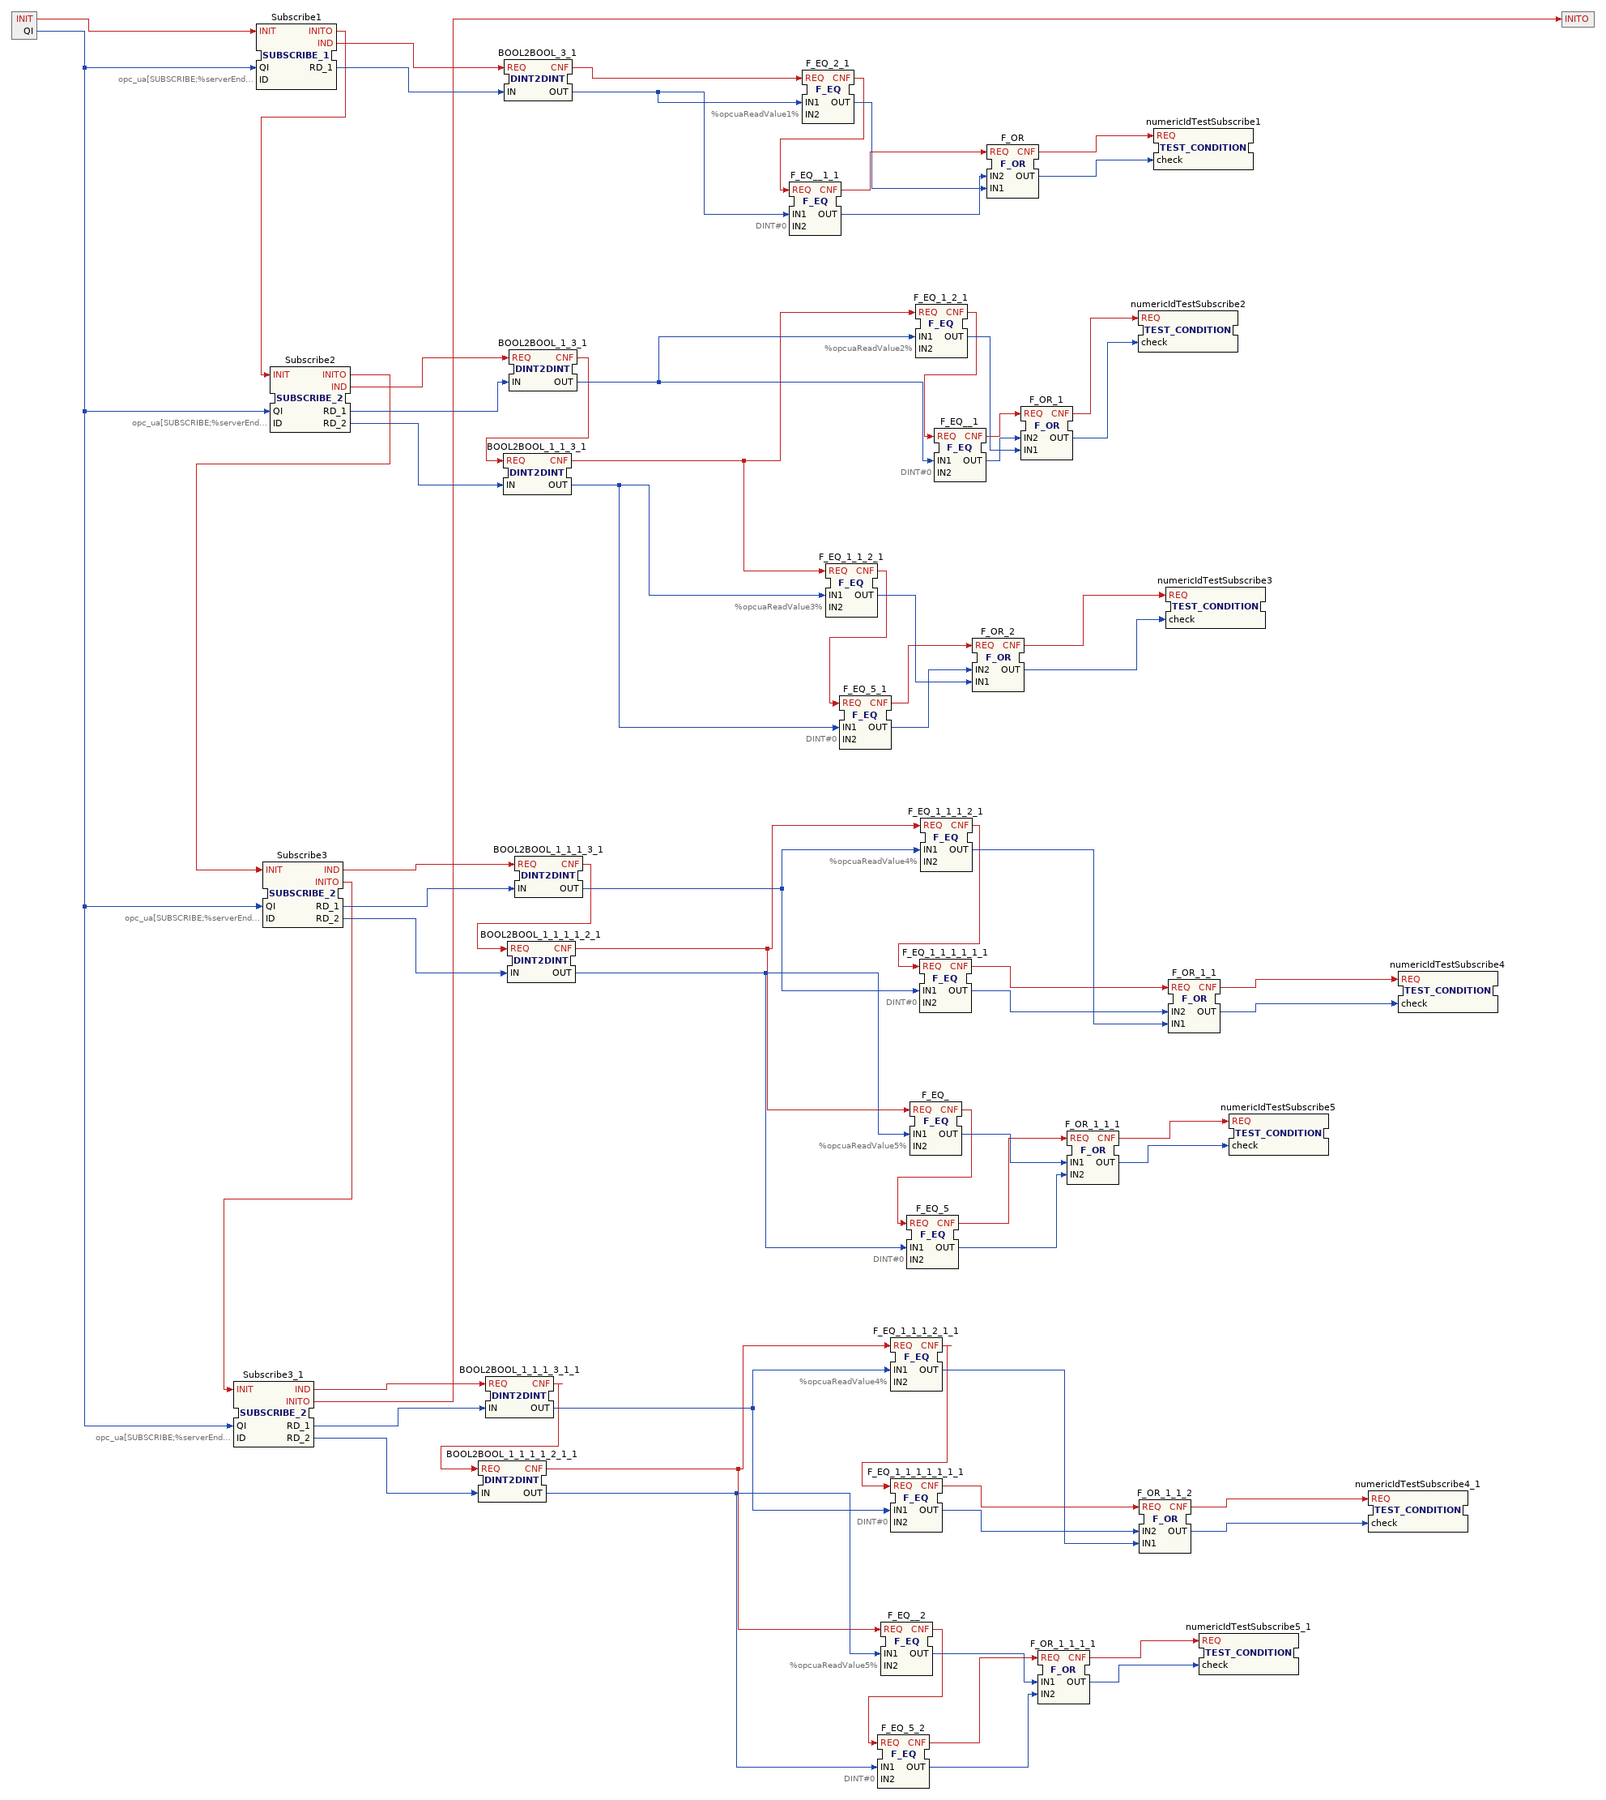
        FBS
          F_EQ_2_1 : F_EQ(IN2 := %opcuaReadValue1%);
          numericIdTestSubscribe4 : TEST_CONDITION;
          Subscribe3 : SUBSCRIBE_2(ID := opc_ua[SUBSCRIBE;%serverEndpoint%;%opcuaFolderTestWithNodeIdNumeric3%]);
          F_EQ_1_1_1_2_1 : F_EQ(IN2 := %opcuaReadValue4%);
          numericIdTestSubscribe3 : TEST_CONDITION;
          F_EQ_1_1_1_1_1_1 : F_EQ(IN2 := DINT#0);
          F_EQ_1_1_2_1 : F_EQ(IN2 := %opcuaReadValue3%);
          numericIdTestSubscribe1 : TEST_CONDITION;
          numericIdTestSubscribe2 : TEST_CONDITION;
          Subscribe1 : SUBSCRIBE_1(ID := opc_ua[SUBSCRIBE;%serverEndpoint%;%opcuaFolderTestWithNodeIdNumeric1%]);
          Subscribe2 : SUBSCRIBE_2(ID := opc_ua[SUBSCRIBE;%serverEndpoint%;%opcuaFolderTestWithNodeIdNumeric2%]);
          BOOL2BOOL_1_1_3_1 : DINT2DINT;
          F_EQ_1_2_1 : F_EQ(IN2 := %opcuaReadValue2%);
          BOOL2BOOL_3_1 : DINT2DINT;
          BOOL2BOOL_1_1_1_3_1 : DINT2DINT;
          BOOL2BOOL_1_1_1_1_2_1 : DINT2DINT;
          BOOL2BOOL_1_3_1 : DINT2DINT;
          F_EQ_ : F_EQ(IN2 := %opcuaReadValue5%);
          numericIdTestSubscribe5 : TEST_CONDITION;
          F_EQ_5 : F_EQ(IN2 := DINT#0);
          F_EQ_5_1 : F_EQ(IN2 := DINT#0);
          F_EQ__1 : F_EQ(IN2 := DINT#0);
          F_EQ__1_1 : F_EQ(IN2 := DINT#0);
          F_OR : F_OR;
          F_OR_1 : F_OR;
          F_OR_2 : F_OR;
          F_OR_1_1 : F_OR;
          F_OR_1_1_1 : F_OR;
          F_EQ_5_2 : F_EQ(IN2 := DINT#0);
          BOOL2BOOL_1_1_1_1_2_1_1 : DINT2DINT;
          Subscribe3_1 : SUBSCRIBE_2(ID := opc_ua[SUBSCRIBE;%serverEndpoint%;,1:i=12348;,1:i=12349]);
          F_EQ_1_1_1_1_1_1_1 : F_EQ(IN2 := DINT#0);
          F_OR_1_1_1_1 : F_OR;
          BOOL2BOOL_1_1_1_3_1_1 : DINT2DINT;
          F_OR_1_1_2 : F_OR;
          numericIdTestSubscribe4_1 : TEST_CONDITION;
          numericIdTestSubscribe5_1 : TEST_CONDITION;
          F_EQ__2 : F_EQ(IN2 := %opcuaReadValue5%);
          F_EQ_1_1_1_2_1_1 : F_EQ(IN2 := %opcuaReadValue4%);
        END_FBS
        EVENT_CONNECTIONS
          Subscribe2.INITO TO Subscribe3.INIT;
          Subscribe3.IND TO BOOL2BOOL_1_1_1_3_1.REQ;
          Subscribe1.INITO TO Subscribe2.INIT;
          Subscribe1.IND TO BOOL2BOOL_3_1.REQ;
          Subscribe2.IND TO BOOL2BOOL_1_3_1.REQ;
          BOOL2BOOL_1_3_1.CNF TO BOOL2BOOL_1_1_3_1.REQ;
          BOOL2BOOL_1_1_1_3_1.CNF TO BOOL2BOOL_1_1_1_1_2_1.REQ;
          INIT TO Subscribe1.INIT;
          F_EQ__1_1.CNF TO F_OR.REQ;
          BOOL2BOOL_3_1.CNF TO F_EQ_2_1.REQ;
          F_EQ_2_1.CNF TO F_EQ__1_1.REQ;
          F_OR.CNF TO numericIdTestSubscribe1.REQ;
          F_OR_2.CNF TO numericIdTestSubscribe3.REQ;
          F_OR_1.CNF TO numericIdTestSubscribe2.REQ;
          F_EQ__1.CNF TO F_OR_1.REQ;
          F_EQ_1_2_1.CNF TO F_EQ__1.REQ;
          BOOL2BOOL_1_1_3_1.CNF TO F_EQ_1_2_1.REQ;
          BOOL2BOOL_1_1_3_1.CNF TO F_EQ_1_1_2_1.REQ;
          F_EQ_1_1_2_1.CNF TO F_EQ_5_1.REQ;
          F_EQ_5_1.CNF TO F_OR_2.REQ;
          F_OR_1_1.CNF TO numericIdTestSubscribe4.REQ;
          F_EQ_1_1_1_1_1_1.CNF TO F_OR_1_1.REQ;
          F_EQ_1_1_1_2_1.CNF TO F_EQ_1_1_1_1_1_1.REQ;
          BOOL2BOOL_1_1_1_1_2_1.CNF TO F_EQ_1_1_1_2_1.REQ;
          F_OR_1_1_1.CNF TO numericIdTestSubscribe5.REQ;
          BOOL2BOOL_1_1_1_1_2_1.CNF TO F_EQ_.REQ;
          F_EQ_.CNF TO F_EQ_5.REQ;
          F_EQ_5.CNF TO F_OR_1_1_1.REQ;
          F_EQ_1_1_1_2_1_1.CNF TO F_EQ_1_1_1_1_1_1_1.REQ;
          F_EQ_1_1_1_1_1_1_1.CNF TO F_OR_1_1_2.REQ;
          BOOL2BOOL_1_1_1_1_2_1_1.CNF TO F_EQ_1_1_1_2_1_1.REQ;
          F_OR_1_1_2.CNF TO numericIdTestSubscribe4_1.REQ;
          Subscribe3_1.IND TO BOOL2BOOL_1_1_1_3_1_1.REQ;
          BOOL2BOOL_1_1_1_1_2_1_1.CNF TO F_EQ__2.REQ;
          F_OR_1_1_1_1.CNF TO numericIdTestSubscribe5_1.REQ;
          F_EQ__2.CNF TO F_EQ_5_2.REQ;
          F_EQ_5_2.CNF TO F_OR_1_1_1_1.REQ;
          BOOL2BOOL_1_1_1_3_1_1.CNF TO BOOL2BOOL_1_1_1_1_2_1_1.REQ;
          Subscribe3_1.INITO TO INITO;
          Subscribe3.INITO TO Subscribe3_1.INIT;
        END_CONNECTIONS
        DATA_CONNECTIONS
          BOOL2BOOL_3_1.OUT TO F_EQ_2_1.IN1;
          Subscribe3.RD_1 TO BOOL2BOOL_1_1_1_3_1.IN;
          Subscribe3.RD_2 TO BOOL2BOOL_1_1_1_1_2_1.IN;
          BOOL2BOOL_1_1_3_1.OUT TO F_EQ_1_1_2_1.IN1;
          Subscribe1.RD_1 TO BOOL2BOOL_3_1.IN;
          Subscribe2.RD_1 TO BOOL2BOOL_1_3_1.IN;
          Subscribe2.RD_2 TO BOOL2BOOL_1_1_3_1.IN;
          BOOL2BOOL_1_3_1.OUT TO F_EQ_1_2_1.IN1;
          QI TO Subscribe3.QI;
          QI TO Subscribe1.QI;
          QI TO Subscribe2.QI;
          BOOL2BOOL_1_1_1_1_2_1.OUT TO F_EQ_5.IN1;
          BOOL2BOOL_1_3_1.OUT TO F_EQ__1.IN1;
          BOOL2BOOL_1_1_3_1.OUT TO F_EQ_5_1.IN1;
          BOOL2BOOL_3_1.OUT TO F_EQ__1_1.IN1;
          BOOL2BOOL_1_1_1_3_1.OUT TO F_EQ_1_1_1_2_1.IN1;
          F_EQ__1_1.OUT TO F_OR.IN2;
          F_EQ_2_1.OUT TO F_OR.IN1;
          F_OR.OUT TO numericIdTestSubscribe1.check;
          F_EQ_5_1.OUT TO F_OR_2.IN2;
          F_EQ__1.OUT TO F_OR_1.IN2;
          F_EQ_1_2_1.OUT TO F_OR_1.IN1;
          F_OR_1.OUT TO numericIdTestSubscribe2.check;
          F_OR_2.OUT TO numericIdTestSubscribe3.check;
          F_OR_1_1.OUT TO numericIdTestSubscribe4.check;
          F_EQ_1_1_1_1_1_1.OUT TO F_OR_1_1.IN2;
          F_EQ_1_1_1_2_1.OUT TO F_OR_1_1.IN1;
          F_OR_1_1_1.OUT TO numericIdTestSubscribe5.check;
          F_EQ_.OUT TO F_OR_1_1_1.IN1;
          F_EQ_5.OUT TO F_OR_1_1_1.IN2;
          BOOL2BOOL_1_1_1_1_2_1.OUT TO F_EQ_.IN1;
          F_EQ_1_1_2_1.OUT TO F_OR_2.IN1;
          BOOL2BOOL_1_1_1_3_1.OUT TO F_EQ_1_1_1_1_1_1.IN1;
          F_EQ__2.OUT TO F_OR_1_1_1_1.IN1;
          F_EQ_1_1_1_1_1_1_1.OUT TO F_OR_1_1_2.IN2;
          BOOL2BOOL_1_1_1_1_2_1_1.OUT TO F_EQ__2.IN1;
          F_EQ_5_2.OUT TO F_OR_1_1_1_1.IN2;
          BOOL2BOOL_1_1_1_3_1_1.OUT TO F_EQ_1_1_1_1_1_1_1.IN1;
          Subscribe3_1.RD_1 TO BOOL2BOOL_1_1_1_3_1_1.IN;
          BOOL2BOOL_1_1_1_1_2_1_1.OUT TO F_EQ_5_2.IN1;
          Subscribe3_1.RD_2 TO BOOL2BOOL_1_1_1_1_2_1_1.IN;
          F_OR_1_1_2.OUT TO numericIdTestSubscribe4_1.check;
          F_EQ_1_1_1_2_1_1.OUT TO F_OR_1_1_2.IN1;
          BOOL2BOOL_1_1_1_3_1_1.OUT TO F_EQ_1_1_1_2_1_1.IN1;
          F_OR_1_1_1_1.OUT TO numericIdTestSubscribe5_1.check;
          QI TO Subscribe3_1.QI;
        END_CONNECTIONS
      END_SUBAPPLICATION
      EVENT_CONNECTIONS
        WriteToVars.INITO TO ReadVars.INIT;
        INIT TO WriteToVars.INIT;
        REQ TO WriteToVars.REQ;
        SubscribeToVars_1.INITO TO INITO;
        ReadVars.INITO TO SubscribeToVars_1.INIT;
        ReadVars.CNF TO CNF;
        WriteToVars.CNF TO ReadVars.REQ;
      END_CONNECTIONS
      DATA_CONNECTIONS
        QI TO ReadVars.QI;
        QI TO WriteToVars.QI;
        QI TO SubscribeToVars_1.QI;
      END_CONNECTIONS
    END_SUBAPPLICATION
    SUBAPPLICATION stringNodeIdTestRemote
      EVENT_INPUT
        INIT;
        REQ;
      END_EVENT
      EVENT_OUTPUT
        INITO;
        CNF;
      END_EVENT
      VAR_INPUT
        QI : BOOL;
      END_VAR
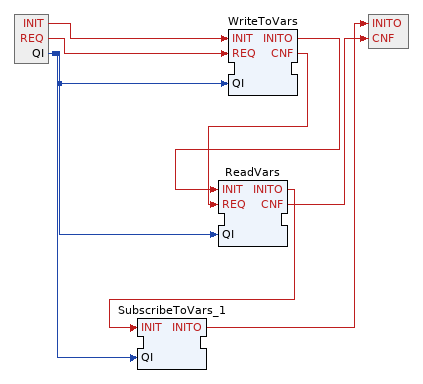
      SUBAPPLICATION WriteToVars
        EVENT_INPUT
          INIT;
          REQ;
        END_EVENT
        EVENT_OUTPUT
          INITO;
          CNF;
        END_EVENT
        VAR_INPUT
          QI : BOOL;
        END_VAR
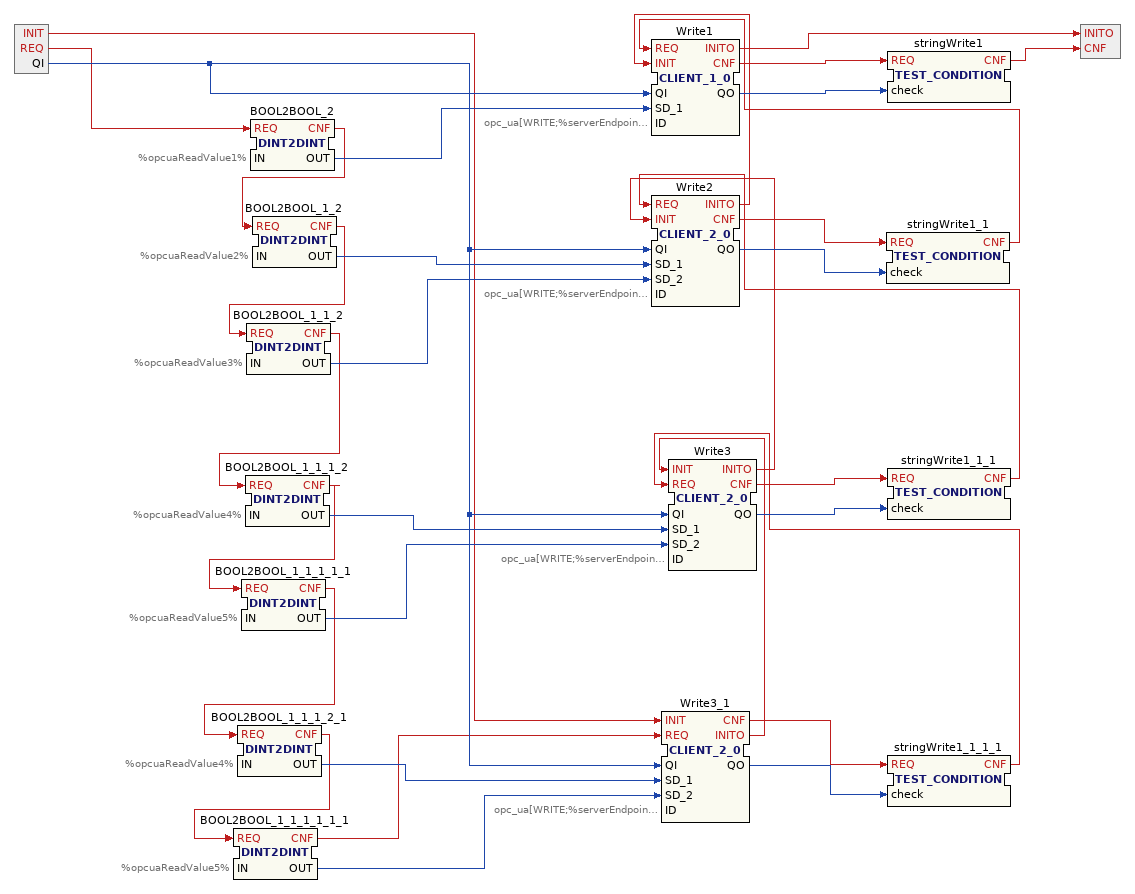
        FBS
          BOOL2BOOL_1_1_2 : DINT2DINT(IN := %opcuaReadValue3%);
          BOOL2BOOL_1_1_1_1_1 : DINT2DINT(IN := %opcuaReadValue5%);
          BOOL2BOOL_1_1_1_2 : DINT2DINT(IN := %opcuaReadValue4%);
          BOOL2BOOL_2 : DINT2DINT(IN := %opcuaReadValue1%);
          BOOL2BOOL_1_2 : DINT2DINT(IN := %opcuaReadValue2%);
          BOOL2BOOL_1_1_1_2_1 : DINT2DINT(IN := %opcuaReadValue4%);
          BOOL2BOOL_1_1_1_1_1_1 : DINT2DINT(IN := %opcuaReadValue5%);
          stringWrite1 : TEST_CONDITION;
          stringWrite1_1 : TEST_CONDITION;
          stringWrite1_1_1 : TEST_CONDITION;
          stringWrite1_1_1_1 : TEST_CONDITION;
          Write1 : CLIENT_1_0(ID := opc_ua[WRITE;%serverEndpoint%;%opcuaFolderTestWithNodeIdString1%]);
          Write2 : CLIENT_2_0(ID := opc_ua[WRITE;%serverEndpoint%;%opcuaFolderTestWithNodeIdString2%]);
          Write3_1 : CLIENT_2_0(ID := opc_ua[WRITE;%serverEndpoint%;,1:s=hello3;,1:s=hello4]);
          Write3 : CLIENT_2_0(ID := opc_ua[WRITE;%serverEndpoint%;%opcuaFolderTestWithNodeIdString3%]);
        END_FBS
        EVENT_CONNECTIONS
          BOOL2BOOL_1_2.CNF TO BOOL2BOOL_1_1_2.REQ;
          BOOL2BOOL_1_1_2.CNF TO BOOL2BOOL_1_1_1_2.REQ;
          BOOL2BOOL_1_1_1_2.CNF TO BOOL2BOOL_1_1_1_1_1.REQ;
          BOOL2BOOL_2.CNF TO BOOL2BOOL_1_2.REQ;
          REQ TO BOOL2BOOL_2.REQ;
          BOOL2BOOL_1_1_1_2_1.CNF TO BOOL2BOOL_1_1_1_1_1_1.REQ;
          BOOL2BOOL_1_1_1_1_1.CNF TO BOOL2BOOL_1_1_1_2_1.REQ;
          stringWrite1.CNF TO CNF;
          stringWrite1_1.CNF TO Write1.REQ;
          Write1.INITO TO INITO;
          Write1.CNF TO stringWrite1.REQ;
          stringWrite1_1_1.CNF TO Write2.REQ;
          Write2.INITO TO Write1.INIT;
          Write2.CNF TO stringWrite1_1.REQ;
          INIT TO Write3_1.INIT;
          BOOL2BOOL_1_1_1_1_1_1.CNF TO Write3_1.REQ;
          Write3_1.CNF TO stringWrite1_1_1_1.REQ;
          Write3_1.INITO TO Write3.INIT;
          stringWrite1_1_1_1.CNF TO Write3.REQ;
          Write3.INITO TO Write2.INIT;
          Write3.CNF TO stringWrite1_1_1.REQ;
        END_CONNECTIONS
        DATA_CONNECTIONS
          QI TO Write1.QI;
          BOOL2BOOL_2.OUT TO Write1.SD_1;
          Write1.QO TO stringWrite1.check;
          QI TO Write2.QI;
          BOOL2BOOL_1_2.OUT TO Write2.SD_1;
          BOOL2BOOL_1_1_2.OUT TO Write2.SD_2;
          Write2.QO TO stringWrite1_1.check;
          QI TO Write3_1.QI;
          BOOL2BOOL_1_1_1_2_1.OUT TO Write3_1.SD_1;
          BOOL2BOOL_1_1_1_1_1_1.OUT TO Write3_1.SD_2;
          Write3_1.QO TO stringWrite1_1_1_1.check;
          QI TO Write3.QI;
          BOOL2BOOL_1_1_1_2.OUT TO Write3.SD_1;
          BOOL2BOOL_1_1_1_1_1.OUT TO Write3.SD_2;
          Write3.QO TO stringWrite1_1_1.check;
        END_CONNECTIONS
      END_SUBAPPLICATION
      SUBAPPLICATION ReadVars
        EVENT_INPUT
          INIT;
          REQ;
        END_EVENT
        EVENT_OUTPUT
          INITO;
          CNF;
        END_EVENT
        VAR_INPUT
          QI : BOOL;
        END_VAR
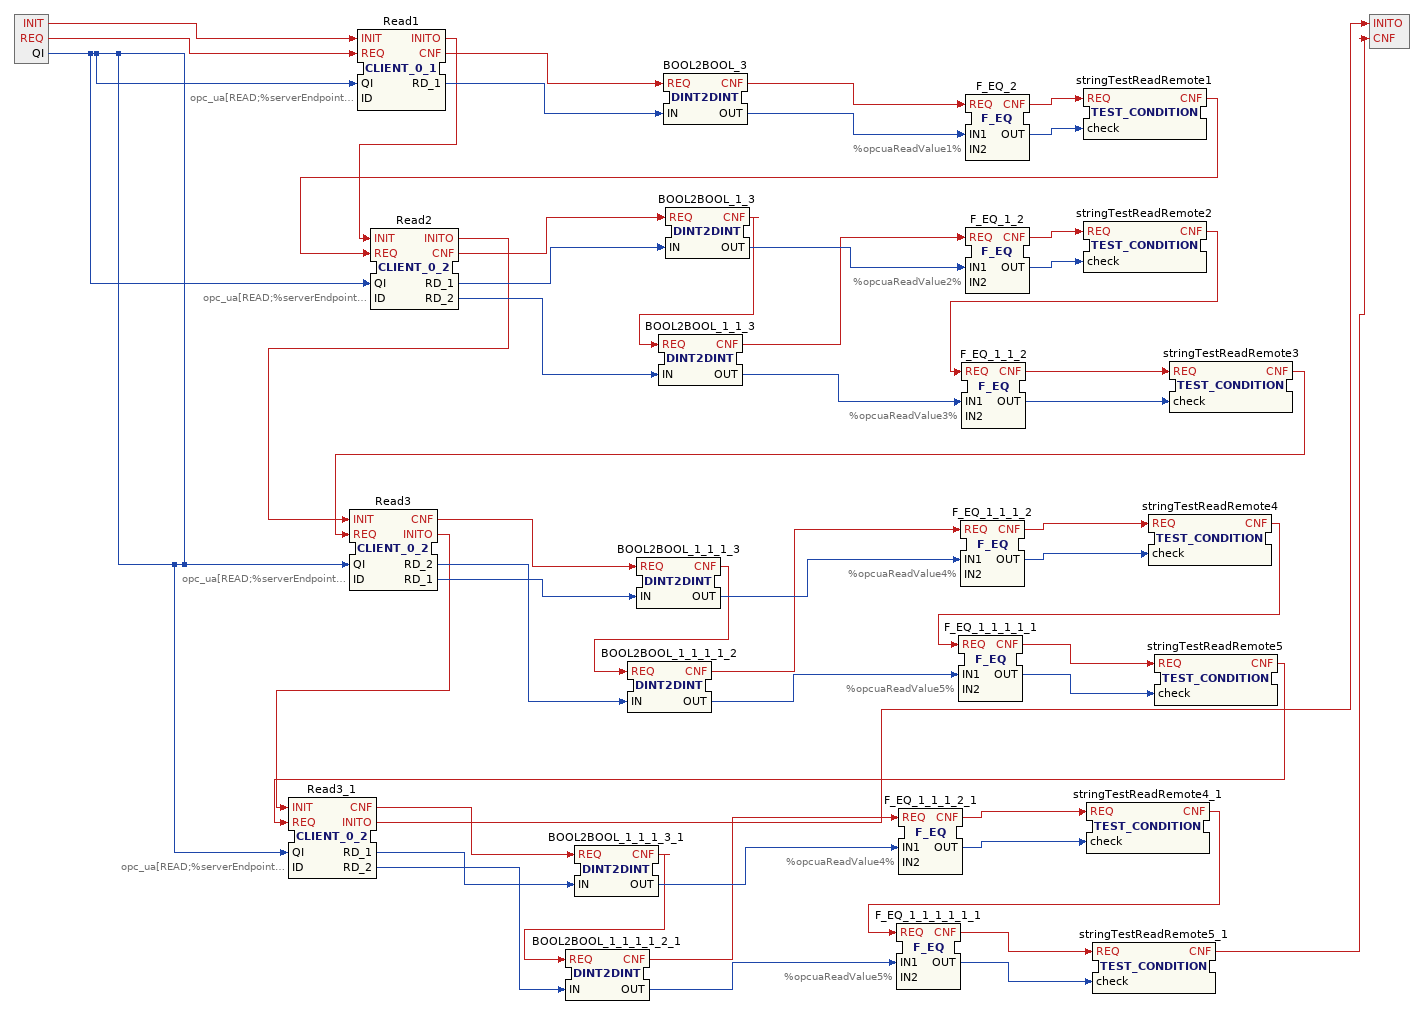
        FBS
          Read1 : CLIENT_0_1(ID := opc_ua[READ;%serverEndpoint%;%opcuaFolderTestWithNodeIdString1%]);
          Read2 : CLIENT_0_2(ID := opc_ua[READ;%serverEndpoint%;%opcuaFolderTestWithNodeIdString2%]);
          F_EQ_1_1_1_2 : F_EQ(IN2 := %opcuaReadValue4%);
          stringTestReadRemote4 : TEST_CONDITION;
          BOOL2BOOL_1_3 : DINT2DINT;
          F_EQ_1_1_1_1_1 : F_EQ(IN2 := %opcuaReadValue5%);
          stringTestReadRemote3 : TEST_CONDITION;
          BOOL2BOOL_1_1_3 : DINT2DINT;
          BOOL2BOOL_1_1_1_1_2 : DINT2DINT;
          BOOL2BOOL_1_1_1_3 : DINT2DINT;
          stringTestReadRemote2 : TEST_CONDITION;
          F_EQ_1_1_2 : F_EQ(IN2 := %opcuaReadValue3%);
          F_EQ_2 : F_EQ(IN2 := %opcuaReadValue1%);
          F_EQ_1_2 : F_EQ(IN2 := %opcuaReadValue2%);
          Read3 : CLIENT_0_2(ID := opc_ua[READ;%serverEndpoint%;%opcuaFolderTestWithNodeIdString3%]);
          stringTestReadRemote5 : TEST_CONDITION;
          stringTestReadRemote1 : TEST_CONDITION;
          BOOL2BOOL_3 : DINT2DINT;
          stringTestReadRemote5_1 : TEST_CONDITION;
          F_EQ_1_1_1_2_1 : F_EQ(IN2 := %opcuaReadValue4%);
          Read3_1 : CLIENT_0_2(ID := opc_ua[READ;%serverEndpoint%;,1:s=hello3;,1:s=hello4]);
          F_EQ_1_1_1_1_1_1 : F_EQ(IN2 := %opcuaReadValue5%);
          BOOL2BOOL_1_1_1_1_2_1 : DINT2DINT;
          BOOL2BOOL_1_1_1_3_1 : DINT2DINT;
          stringTestReadRemote4_1 : TEST_CONDITION;
        END_FBS
        EVENT_CONNECTIONS
          Read1.INITO TO Read2.INIT;
          Read1.CNF TO BOOL2BOOL_3.REQ;
          stringTestReadRemote1.CNF TO Read2.REQ;
          Read2.INITO TO Read3.INIT;
          Read2.CNF TO BOOL2BOOL_1_3.REQ;
          BOOL2BOOL_1_1_1_1_2.CNF TO F_EQ_1_1_1_2.REQ;
          F_EQ_1_1_1_2.CNF TO stringTestReadRemote4.REQ;
          stringTestReadRemote4.CNF TO F_EQ_1_1_1_1_1.REQ;
          BOOL2BOOL_1_3.CNF TO BOOL2BOOL_1_1_3.REQ;
          F_EQ_1_1_1_1_1.CNF TO stringTestReadRemote5.REQ;
          F_EQ_1_1_2.CNF TO stringTestReadRemote3.REQ;
          stringTestReadRemote3.CNF TO Read3.REQ;
          BOOL2BOOL_1_1_3.CNF TO F_EQ_1_2.REQ;
          BOOL2BOOL_1_1_1_3.CNF TO BOOL2BOOL_1_1_1_1_2.REQ;
          Read3.CNF TO BOOL2BOOL_1_1_1_3.REQ;
          F_EQ_1_2.CNF TO stringTestReadRemote2.REQ;
          stringTestReadRemote2.CNF TO F_EQ_1_1_2.REQ;
          BOOL2BOOL_3.CNF TO F_EQ_2.REQ;
          F_EQ_2.CNF TO stringTestReadRemote1.REQ;
          INIT TO Read1.INIT;
          REQ TO Read1.REQ;
          BOOL2BOOL_1_1_1_1_2_1.CNF TO F_EQ_1_1_1_2_1.REQ;
          BOOL2BOOL_1_1_1_3_1.CNF TO BOOL2BOOL_1_1_1_1_2_1.REQ;
          F_EQ_1_1_1_2_1.CNF TO stringTestReadRemote4_1.REQ;
          Read3_1.CNF TO BOOL2BOOL_1_1_1_3_1.REQ;
          F_EQ_1_1_1_1_1_1.CNF TO stringTestReadRemote5_1.REQ;
          stringTestReadRemote4_1.CNF TO F_EQ_1_1_1_1_1_1.REQ;
          Read3_1.INITO TO INITO;
          Read3.INITO TO Read3_1.INIT;
          stringTestReadRemote5_1.CNF TO CNF;
          stringTestReadRemote5.CNF TO Read3_1.REQ;
        END_CONNECTIONS
        DATA_CONNECTIONS
          Read1.RD_1 TO BOOL2BOOL_3.IN;
          Read2.RD_1 TO BOOL2BOOL_1_3.IN;
          Read2.RD_2 TO BOOL2BOOL_1_1_3.IN;
          BOOL2BOOL_1_1_1_3.OUT TO F_EQ_1_1_1_2.IN1;
          F_EQ_1_1_1_2.OUT TO stringTestReadRemote4.check;
          BOOL2BOOL_1_3.OUT TO F_EQ_1_2.IN1;
          BOOL2BOOL_1_1_1_1_2.OUT TO F_EQ_1_1_1_1_1.IN1;
          F_EQ_1_1_1_1_1.OUT TO stringTestReadRemote5.check;
          F_EQ_1_1_2.OUT TO stringTestReadRemote3.check;
          BOOL2BOOL_1_1_3.OUT TO F_EQ_1_1_2.IN1;
          Read3.RD_2 TO BOOL2BOOL_1_1_1_1_2.IN;
          Read3.RD_1 TO BOOL2BOOL_1_1_1_3.IN;
          F_EQ_1_2.OUT TO stringTestReadRemote2.check;
          BOOL2BOOL_3.OUT TO F_EQ_2.IN1;
          F_EQ_2.OUT TO stringTestReadRemote1.check;
          QI TO Read1.QI;
          QI TO Read2.QI;
          QI TO Read3.QI;
          Read3_1.RD_1 TO BOOL2BOOL_1_1_1_3_1.IN;
          Read3_1.RD_2 TO BOOL2BOOL_1_1_1_1_2_1.IN;
          F_EQ_1_1_1_2_1.OUT TO stringTestReadRemote4_1.check;
          F_EQ_1_1_1_1_1_1.OUT TO stringTestReadRemote5_1.check;
          BOOL2BOOL_1_1_1_3_1.OUT TO F_EQ_1_1_1_2_1.IN1;
          BOOL2BOOL_1_1_1_1_2_1.OUT TO F_EQ_1_1_1_1_1_1.IN1;
          QI TO Read3_1.QI;
        END_CONNECTIONS
      END_SUBAPPLICATION
      SUBAPPLICATION SubscribeToVars_1
        EVENT_INPUT
          INIT;
        END_EVENT
        EVENT_OUTPUT
          INITO;
        END_EVENT
        VAR_INPUT
          QI : BOOL;
        END_VAR
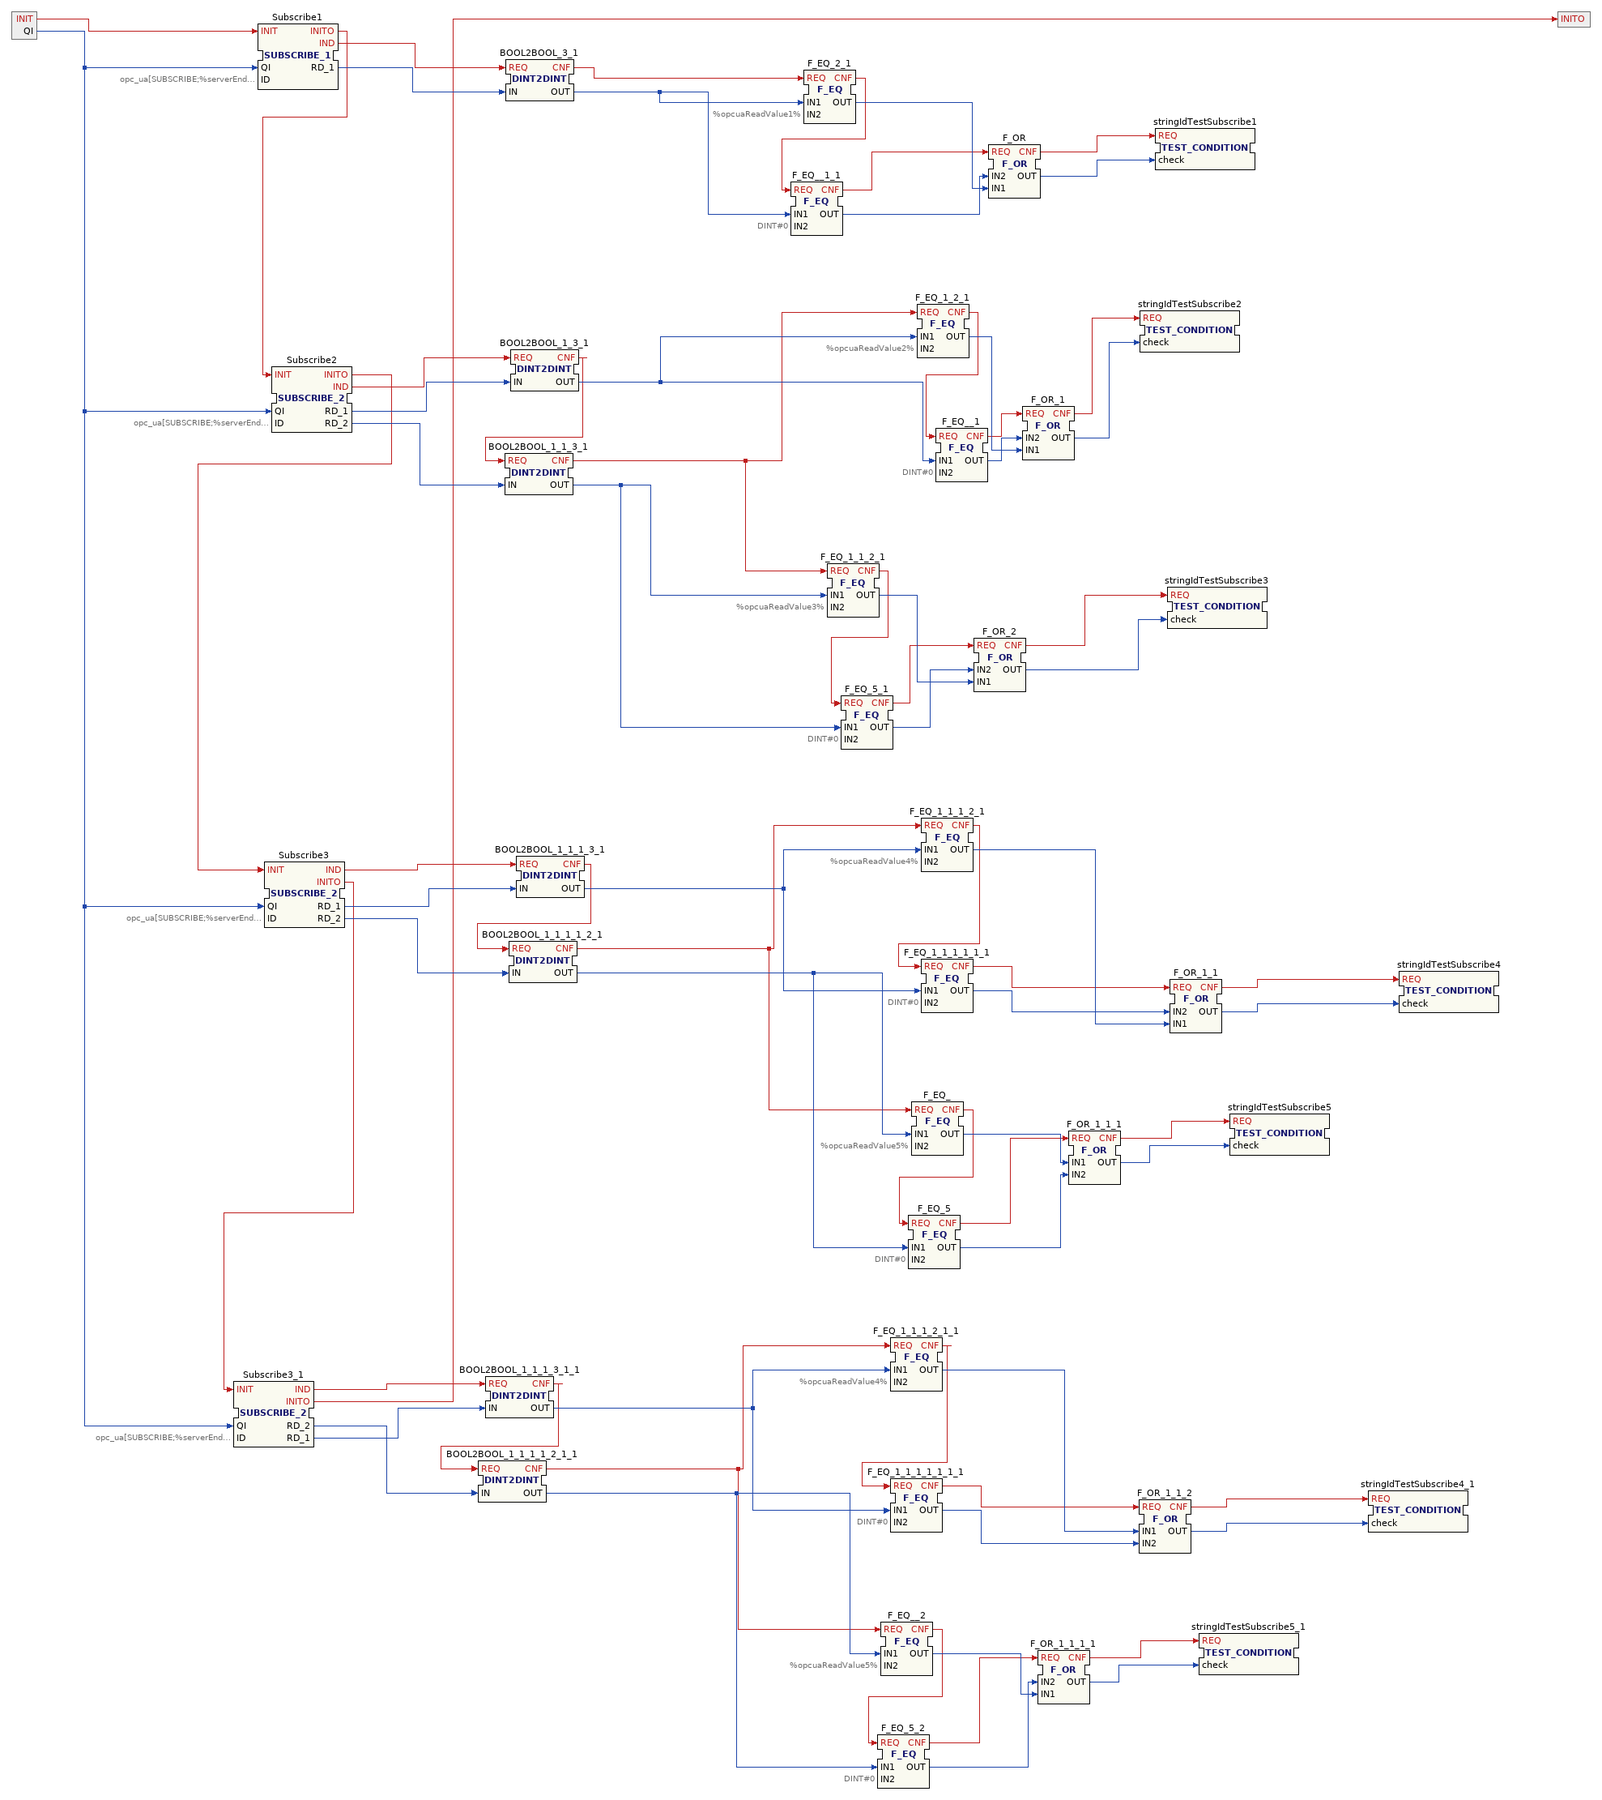
        FBS
          F_EQ_2_1 : F_EQ(IN2 := %opcuaReadValue1%);
          stringIdTestSubscribe4 : TEST_CONDITION;
          Subscribe3 : SUBSCRIBE_2(ID := opc_ua[SUBSCRIBE;%serverEndpoint%;%opcuaFolderTestWithNodeIdString3%]);
          F_EQ_1_1_1_2_1 : F_EQ(IN2 := %opcuaReadValue4%);
          stringIdTestSubscribe3 : TEST_CONDITION;
          F_EQ_1_1_1_1_1_1 : F_EQ(IN2 := DINT#0);
          F_EQ_1_1_2_1 : F_EQ(IN2 := %opcuaReadValue3%);
          stringIdTestSubscribe1 : TEST_CONDITION;
          stringIdTestSubscribe2 : TEST_CONDITION;
          Subscribe1 : SUBSCRIBE_1(ID := opc_ua[SUBSCRIBE;%serverEndpoint%;%opcuaFolderTestWithNodeIdString1%]);
          Subscribe2 : SUBSCRIBE_2(ID := opc_ua[SUBSCRIBE;%serverEndpoint%;%opcuaFolderTestWithNodeIdString2%]);
          BOOL2BOOL_1_1_3_1 : DINT2DINT;
          F_EQ_1_2_1 : F_EQ(IN2 := %opcuaReadValue2%);
          BOOL2BOOL_3_1 : DINT2DINT;
          BOOL2BOOL_1_1_1_3_1 : DINT2DINT;
          BOOL2BOOL_1_1_1_1_2_1 : DINT2DINT;
          BOOL2BOOL_1_3_1 : DINT2DINT;
          F_EQ_ : F_EQ(IN2 := %opcuaReadValue5%);
          stringIdTestSubscribe5 : TEST_CONDITION;
          F_EQ_5 : F_EQ(IN2 := DINT#0);
          F_EQ_5_1 : F_EQ(IN2 := DINT#0);
          F_EQ__1 : F_EQ(IN2 := DINT#0);
          F_EQ__1_1 : F_EQ(IN2 := DINT#0);
          F_OR : F_OR;
          F_OR_1 : F_OR;
          F_OR_2 : F_OR;
          F_OR_1_1 : F_OR;
          F_OR_1_1_1 : F_OR;
          BOOL2BOOL_1_1_1_1_2_1_1 : DINT2DINT;
          F_OR_1_1_2 : F_OR;
          BOOL2BOOL_1_1_1_3_1_1 : DINT2DINT;
          F_EQ__2 : F_EQ(IN2 := %opcuaReadValue5%);
          stringIdTestSubscribe5_1 : TEST_CONDITION;
          stringIdTestSubscribe4_1 : TEST_CONDITION;
          F_OR_1_1_1_1 : F_OR;
          Subscribe3_1 : SUBSCRIBE_2(ID := opc_ua[SUBSCRIBE;%serverEndpoint%;,1:s=hello3;,1:s=hello4]);
          F_EQ_1_1_1_1_1_1_1 : F_EQ(IN2 := DINT#0);
          F_EQ_5_2 : F_EQ(IN2 := DINT#0);
          F_EQ_1_1_1_2_1_1 : F_EQ(IN2 := %opcuaReadValue4%);
        END_FBS
        EVENT_CONNECTIONS
          Subscribe2.INITO TO Subscribe3.INIT;
          Subscribe3.IND TO BOOL2BOOL_1_1_1_3_1.REQ;
          Subscribe1.INITO TO Subscribe2.INIT;
          Subscribe1.IND TO BOOL2BOOL_3_1.REQ;
          Subscribe2.IND TO BOOL2BOOL_1_3_1.REQ;
          BOOL2BOOL_1_3_1.CNF TO BOOL2BOOL_1_1_3_1.REQ;
          BOOL2BOOL_1_1_1_3_1.CNF TO BOOL2BOOL_1_1_1_1_2_1.REQ;
          INIT TO Subscribe1.INIT;
          F_EQ__1_1.CNF TO F_OR.REQ;
          BOOL2BOOL_3_1.CNF TO F_EQ_2_1.REQ;
          F_EQ_2_1.CNF TO F_EQ__1_1.REQ;
          F_OR.CNF TO stringIdTestSubscribe1.REQ;
          F_OR_2.CNF TO stringIdTestSubscribe3.REQ;
          F_OR_1.CNF TO stringIdTestSubscribe2.REQ;
          F_EQ__1.CNF TO F_OR_1.REQ;
          F_EQ_1_2_1.CNF TO F_EQ__1.REQ;
          BOOL2BOOL_1_1_3_1.CNF TO F_EQ_1_2_1.REQ;
          BOOL2BOOL_1_1_3_1.CNF TO F_EQ_1_1_2_1.REQ;
          F_EQ_1_1_2_1.CNF TO F_EQ_5_1.REQ;
          F_EQ_5_1.CNF TO F_OR_2.REQ;
          F_OR_1_1.CNF TO stringIdTestSubscribe4.REQ;
          F_EQ_1_1_1_1_1_1.CNF TO F_OR_1_1.REQ;
          F_EQ_1_1_1_2_1.CNF TO F_EQ_1_1_1_1_1_1.REQ;
          BOOL2BOOL_1_1_1_1_2_1.CNF TO F_EQ_1_1_1_2_1.REQ;
          F_OR_1_1_1.CNF TO stringIdTestSubscribe5.REQ;
          BOOL2BOOL_1_1_1_1_2_1.CNF TO F_EQ_.REQ;
          F_EQ_.CNF TO F_EQ_5.REQ;
          F_EQ_5.CNF TO F_OR_1_1_1.REQ;
          F_EQ_1_1_1_2_1_1.CNF TO F_EQ_1_1_1_1_1_1_1.REQ;
          Subscribe3_1.IND TO BOOL2BOOL_1_1_1_3_1_1.REQ;
          BOOL2BOOL_1_1_1_1_2_1_1.CNF TO F_EQ__2.REQ;
          F_OR_1_1_1_1.CNF TO stringIdTestSubscribe5_1.REQ;
          BOOL2BOOL_1_1_1_1_2_1_1.CNF TO F_EQ_1_1_1_2_1_1.REQ;
          BOOL2BOOL_1_1_1_3_1_1.CNF TO BOOL2BOOL_1_1_1_1_2_1_1.REQ;
          F_EQ_1_1_1_1_1_1_1.CNF TO F_OR_1_1_2.REQ;
          F_EQ__2.CNF TO F_EQ_5_2.REQ;
          F_OR_1_1_2.CNF TO stringIdTestSubscribe4_1.REQ;
          F_EQ_5_2.CNF TO F_OR_1_1_1_1.REQ;
          Subscribe3_1.INITO TO INITO;
          Subscribe3.INITO TO Subscribe3_1.INIT;
        END_CONNECTIONS
        DATA_CONNECTIONS
          BOOL2BOOL_3_1.OUT TO F_EQ_2_1.IN1;
          Subscribe3.RD_1 TO BOOL2BOOL_1_1_1_3_1.IN;
          Subscribe3.RD_2 TO BOOL2BOOL_1_1_1_1_2_1.IN;
          BOOL2BOOL_1_1_3_1.OUT TO F_EQ_1_1_2_1.IN1;
          Subscribe1.RD_1 TO BOOL2BOOL_3_1.IN;
          Subscribe2.RD_1 TO BOOL2BOOL_1_3_1.IN;
          Subscribe2.RD_2 TO BOOL2BOOL_1_1_3_1.IN;
          BOOL2BOOL_1_3_1.OUT TO F_EQ_1_2_1.IN1;
          QI TO Subscribe3.QI;
          QI TO Subscribe1.QI;
          QI TO Subscribe2.QI;
          BOOL2BOOL_1_1_1_1_2_1.OUT TO F_EQ_5.IN1;
          BOOL2BOOL_1_3_1.OUT TO F_EQ__1.IN1;
          BOOL2BOOL_1_1_3_1.OUT TO F_EQ_5_1.IN1;
          BOOL2BOOL_3_1.OUT TO F_EQ__1_1.IN1;
          BOOL2BOOL_1_1_1_3_1.OUT TO F_EQ_1_1_1_2_1.IN1;
          F_EQ__1_1.OUT TO F_OR.IN2;
          F_EQ_2_1.OUT TO F_OR.IN1;
          F_OR.OUT TO stringIdTestSubscribe1.check;
          F_EQ_5_1.OUT TO F_OR_2.IN2;
          F_EQ__1.OUT TO F_OR_1.IN2;
          F_EQ_1_2_1.OUT TO F_OR_1.IN1;
          F_OR_1.OUT TO stringIdTestSubscribe2.check;
          F_OR_2.OUT TO stringIdTestSubscribe3.check;
          F_OR_1_1.OUT TO stringIdTestSubscribe4.check;
          F_EQ_1_1_1_1_1_1.OUT TO F_OR_1_1.IN2;
          F_EQ_1_1_1_2_1.OUT TO F_OR_1_1.IN1;
          F_OR_1_1_1.OUT TO stringIdTestSubscribe5.check;
          F_EQ_.OUT TO F_OR_1_1_1.IN1;
          F_EQ_5.OUT TO F_OR_1_1_1.IN2;
          BOOL2BOOL_1_1_1_1_2_1.OUT TO F_EQ_.IN1;
          F_EQ_1_1_2_1.OUT TO F_OR_2.IN1;
          BOOL2BOOL_1_1_1_3_1.OUT TO F_EQ_1_1_1_1_1_1.IN1;
          BOOL2BOOL_1_1_1_3_1_1.OUT TO F_EQ_1_1_1_1_1_1_1.IN1;
          F_EQ_5_2.OUT TO F_OR_1_1_1_1.IN2;
          F_EQ_1_1_1_2_1_1.OUT TO F_OR_1_1_2.IN1;
          F_EQ__2.OUT TO F_OR_1_1_1_1.IN1;
          F_OR_1_1_1_1.OUT TO stringIdTestSubscribe5_1.check;
          Subscribe3_1.RD_2 TO BOOL2BOOL_1_1_1_1_2_1_1.IN;
          BOOL2BOOL_1_1_1_1_2_1_1.OUT TO F_EQ__2.IN1;
          Subscribe3_1.RD_1 TO BOOL2BOOL_1_1_1_3_1_1.IN;
          BOOL2BOOL_1_1_1_3_1_1.OUT TO F_EQ_1_1_1_2_1_1.IN1;
          F_OR_1_1_2.OUT TO stringIdTestSubscribe4_1.check;
          F_EQ_1_1_1_1_1_1_1.OUT TO F_OR_1_1_2.IN2;
          BOOL2BOOL_1_1_1_1_2_1_1.OUT TO F_EQ_5_2.IN1;
          QI TO Subscribe3_1.QI;
        END_CONNECTIONS
      END_SUBAPPLICATION
      EVENT_CONNECTIONS
        WriteToVars.INITO TO ReadVars.INIT;
        INIT TO WriteToVars.INIT;
        REQ TO WriteToVars.REQ;
        SubscribeToVars_1.INITO TO INITO;
        ReadVars.INITO TO SubscribeToVars_1.INIT;
        WriteToVars.CNF TO ReadVars.REQ;
        ReadVars.CNF TO CNF;
      END_CONNECTIONS
      DATA_CONNECTIONS
        QI TO ReadVars.QI;
        QI TO WriteToVars.QI;
        QI TO SubscribeToVars_1.QI;
      END_CONNECTIONS
    END_SUBAPPLICATION
    SUBAPPLICATION bytestringNodeIdTestRemote
      EVENT_INPUT
        INIT;
        REQ;
      END_EVENT
      EVENT_OUTPUT
        INITO;
        CNF;
      END_EVENT
      VAR_INPUT
        QI : BOOL;
      END_VAR
